REGION Network 80: IMMEDIATE STOP ALARMS
   RUNG wire#powerrail
      Contact( "M_ONE" )
      wire#w1
      I_Contact( #oALARM_POWDER_LINE_1_CLOGGED )
      I_Contact( #oALARM_GAS_FLOW_BELOW_LOW_LIMIT_LN_1 )
      I_Contact( #oALARM_DISK_SPEED_BELOW_LOW_LIMIT_LN_1 )
      I_Contact( #oALARM_STIRRER_SPEED_BELOW_LOW_LIMIT_LN_1 )
      I_Contact( #oALARM_GAS_FLOW_ABOVE_HIGH_LIMIT_LN_1 )
      I_Contact( #oALARM_CARRIER_GAS_INLET_PRESSURE_TOO_LOW_LN_1 )
      Not()
      Coil( #DATA.FAULT )
   END_RUNG
   RUNG wire#w1
      I_Contact( #DATA.FAULT )
      I_Contact( #oALARM_DISK_SPEED_ABOVE_HIGH_LIMIT_LN_1 )
      I_Contact( #oALARM_STIRRER_SPEED_ABOVE_HIGH_LIMIT_LN_1 )
      I_Contact( #oALARM_DISK_MOTOR_PLUGGED_IN_AND_READY_LN_1 )
      I_Contact( #oALARM_STIRRER_PLUGGED_IN_AND_READY_LN_1 )
      I_Contact( #oALARM_COMMUNICATION_RUNNING_LN_1 )
      I_Contact( #oALARM_FEEDER_NOT_READY_LN_1 )
      Not()
      Coil( #DATA.FAULT )
   END_RUNG
   RUNG wire#w1
      I_Contact( #DATA.FAULT )
      I_Contact( #oALARM_POWDER_LINE_2_CLOGGED )
      I_Contact( #oALARM_GAS_FLOW_BELOW_LOW_LIMIT_LN_2 )
      I_Contact( #oALARM_DISK_SPEED_BELOW_LOW_LIMIT_LN_2 )
      I_Contact( #oALARM_STIRRER_SPEED_BELOW_LOW_LIMIT_LN_2 )
      I_Contact( #oALARM_GAS_FLOW_ABOVE_HIGH_LIMIT_LN_2 )
      I_Contact( #oALARM_CARRIER_GAS_INLET_PRESSURE_TOO_LOW_LN_2 )
      Not()
      Coil( #DATA.FAULT )
   END_RUNG
   RUNG wire#w1
      I_Contact( #DATA.FAULT )
      I_Contact( #oALARM_DISK_SPEED_ABOVE_HIGH_LIMIT_LN_2 )
      I_Contact( #oALARM_STIRRER_SPEED_ABOVE_HIGH_LIMIT_LN_2 )
      I_Contact( #oALARM_DISK_MOTOR_PLUGGED_IN_AND_READY_LN_2 )
      I_Contact( #oALARM_STIRRER_PLUGGED_IN_AND_READY_LN_2 )
      I_Contact( #oALARM_COMMUNICATION_RUNNING_LN_2 )
      I_Contact( #oALARM_FEEDER_NOT_READY_LN_2 )
      Not()
      Move(in := #DB_NUMBER, out1 => "DB441_POWDER_FEEDERS_ALARM_DECODING".GLOBAL_ALARMS_MACHINE.ALARM_DECODING)
      wire#w2
      { S7_Templates := "SrcType := Int" } EQ_Contact(in1 := #INPUT_SETTINGS.UNIT_NUMBER, in2 := 1)
      S_Coil( "DB441_POWDER_FEEDERS_ALARM_DECODING".ALARMS_UNIT_01.POWDER_FEEDER[#INPUT_SETTINGS.FEEDER_NUMBER].IS_ALARMS )
   END_RUNG
   RUNG wire#w2
      { S7_Templates := "SrcType := Int" } EQ_Contact(in1 := #INPUT_SETTINGS.UNIT_NUMBER, in2 := 2)
      S_Coil( "DB441_POWDER_FEEDERS_ALARM_DECODING".ALARMS_UNIT_02.POWDER_FEEDER[#INPUT_SETTINGS.FEEDER_NUMBER].IS_ALARMS )
   END_RUNG
   // the same network as SCL:
   #DATA.FAULT := NOT ("M_ONE" AND NOT #oALARM_POWDER_LINE_1_CLOGGED AND NOT #oALARM_GAS_FLOW_BELOW_LOW_LIMIT_LN_1 AND NOT #oALARM_DISK_SPEED_BELOW_LOW_LIMIT_LN_1 AND NOT #oALARM_STIRRER_SPEED_BELOW_LOW_LIMIT_LN_1 AND NOT #oALARM_GAS_FLOW_ABOVE_HIGH_LIMIT_LN_1 AND NOT #oALARM_CARRIER_GAS_INLET_PRESSURE_TOO_LOW_LN_1);
   #DATA.FAULT := NOT ("M_ONE" AND NOT #DATA.FAULT AND NOT #oALARM_DISK_SPEED_ABOVE_HIGH_LIMIT_LN_1 AND NOT #oALARM_STIRRER_SPEED_ABOVE_HIGH_LIMIT_LN_1 AND NOT #oALARM_DISK_MOTOR_PLUGGED_IN_AND_READY_LN_1 AND NOT #oALARM_STIRRER_PLUGGED_IN_AND_READY_LN_1 AND NOT #oALARM_COMMUNICATION_RUNNING_LN_1 AND NOT #oALARM_FEEDER_NOT_READY_LN_1);
   #DATA.FAULT := NOT ("M_ONE" AND NOT #DATA.FAULT AND NOT #oALARM_POWDER_LINE_2_CLOGGED AND NOT #oALARM_GAS_FLOW_BELOW_LOW_LIMIT_LN_2 AND NOT #oALARM_DISK_SPEED_BELOW_LOW_LIMIT_LN_2 AND NOT #oALARM_STIRRER_SPEED_BELOW_LOW_LIMIT_LN_2 AND NOT #oALARM_GAS_FLOW_ABOVE_HIGH_LIMIT_LN_2 AND NOT #oALARM_CARRIER_GAS_INLET_PRESSURE_TOO_LOW_LN_2);
   #_w1 := NOT ("M_ONE" AND NOT #DATA.FAULT AND NOT #oALARM_DISK_SPEED_ABOVE_HIGH_LIMIT_LN_2 AND NOT #oALARM_STIRRER_SPEED_ABOVE_HIGH_LIMIT_LN_2 AND NOT #oALARM_DISK_MOTOR_PLUGGED_IN_AND_READY_LN_2 AND NOT #oALARM_STIRRER_PLUGGED_IN_AND_READY_LN_2 AND NOT #oALARM_COMMUNICATION_RUNNING_LN_2 AND NOT #oALARM_FEEDER_NOT_READY_LN_2);
   IF #_w1 THEN
       "DB441_POWDER_FEEDERS_ALARM_DECODING".GLOBAL_ALARMS_MACHINE.ALARM_DECODING := #DB_NUMBER;
   END_IF;
   IF #_w1 AND (#INPUT_SETTINGS.UNIT_NUMBER = 1) THEN
       "DB441_POWDER_FEEDERS_ALARM_DECODING".ALARMS_UNIT_01.POWDER_FEEDER[#INPUT_SETTINGS.FEEDER_NUMBER].IS_ALARMS := TRUE;
   END_IF;
   IF #_w1 AND (#INPUT_SETTINGS.UNIT_NUMBER = 2) THEN
       "DB441_POWDER_FEEDERS_ALARM_DECODING".ALARMS_UNIT_02.POWDER_FEEDER[#INPUT_SETTINGS.FEEDER_NUMBER].IS_ALARMS := TRUE;
   END_IF;
END_REGION

REGION Network 81: WARNINGS
   RUNG wire#powerrail
      Contact( "M_ONE" )
      wire#w1
      I_Contact( #oWARNING_GAS_FLOW_UNDER_LIMIT_LN_1 )
      I_Contact( #oWARNING_DISK_SPEED_UNDER_LIMIT_LN_1 )
      I_Contact( #oWARNING_STIRRER_SPEED_UNDER_LIMIT_LN_1 )
      I_Contact( #oWARNING_GAS_FLOW_OVER_LIMIT_LN_1 )
      I_Contact( #oWARNING_DISK_SPEED_OVER_LIMIT_LN_1 )
      I_Contact( #oWARNING_STIRRER_SPEED_OVER_LIMIT_LN_1 )
      Not()
      Coil( #oSTATION_WARNINGS )
   END_RUNG
   RUNG wire#w1
      I_Contact( #oSTATION_WARNINGS )
      I_Contact( #oWARNING_GAS_FLOW_UNDER_LIMIT_LN_2 )
      I_Contact( #oWARNING_DISK_SPEED_UNDER_LIMIT_LN_2 )
      I_Contact( #oWARNING_STIRRER_SPEED_UNDER_LIMIT_LN_2 )
      I_Contact( #oWARNING_GAS_FLOW_OVER_LIMIT_LN_2 )
      I_Contact( #oWARNING_DISK_SPEED_OVER_LIMIT_LN_2 )
      I_Contact( #oWARNING_STIRRER_SPEED_OVER_LIMIT_LN_2 )
      Not()
      Move(in := #DB_NUMBER, out1 => "DB441_POWDER_FEEDERS_ALARM_DECODING".GLOBAL_ALARMS_MACHINE.HELP_DECODING)
      wire#w2
      { S7_Templates := "SrcType := Int" } EQ_Contact(in1 := #INPUT_SETTINGS.UNIT_NUMBER, in2 := 1)
      S_Coil( "DB441_POWDER_FEEDERS_ALARM_DECODING".ALARMS_UNIT_01.POWDER_FEEDER[#INPUT_SETTINGS.FEEDER_NUMBER].WARNING )
   END_RUNG
   RUNG wire#w2
      { S7_Templates := "SrcType := Int" } EQ_Contact(in1 := #INPUT_SETTINGS.UNIT_NUMBER, in2 := 2)
      S_Coil( "DB441_POWDER_FEEDERS_ALARM_DECODING".ALARMS_UNIT_02.POWDER_FEEDER[#INPUT_SETTINGS.FEEDER_NUMBER].WARNING )
   END_RUNG
   // the same network as SCL:
   #oSTATION_WARNINGS := NOT ("M_ONE" AND NOT #oWARNING_GAS_FLOW_UNDER_LIMIT_LN_1 AND NOT #oWARNING_DISK_SPEED_UNDER_LIMIT_LN_1 AND NOT #oWARNING_STIRRER_SPEED_UNDER_LIMIT_LN_1 AND NOT #oWARNING_GAS_FLOW_OVER_LIMIT_LN_1 AND NOT #oWARNING_DISK_SPEED_OVER_LIMIT_LN_1 AND NOT #oWARNING_STIRRER_SPEED_OVER_LIMIT_LN_1);
   #_w1 := NOT ("M_ONE" AND NOT #oSTATION_WARNINGS AND NOT #oWARNING_GAS_FLOW_UNDER_LIMIT_LN_2 AND NOT #oWARNING_DISK_SPEED_UNDER_LIMIT_LN_2 AND NOT #oWARNING_STIRRER_SPEED_UNDER_LIMIT_LN_2 AND NOT #oWARNING_GAS_FLOW_OVER_LIMIT_LN_2 AND NOT #oWARNING_DISK_SPEED_OVER_LIMIT_LN_2 AND NOT #oWARNING_STIRRER_SPEED_OVER_LIMIT_LN_2);
   IF #_w1 THEN
       "DB441_POWDER_FEEDERS_ALARM_DECODING".GLOBAL_ALARMS_MACHINE.HELP_DECODING := #DB_NUMBER;
   END_IF;
   IF #_w1 AND (#INPUT_SETTINGS.UNIT_NUMBER = 1) THEN
       "DB441_POWDER_FEEDERS_ALARM_DECODING".ALARMS_UNIT_01.POWDER_FEEDER[#INPUT_SETTINGS.FEEDER_NUMBER].WARNING := TRUE;
   END_IF;
   IF #_w1 AND (#INPUT_SETTINGS.UNIT_NUMBER = 2) THEN
       "DB441_POWDER_FEEDERS_ALARM_DECODING".ALARMS_UNIT_02.POWDER_FEEDER[#INPUT_SETTINGS.FEEDER_NUMBER].WARNING := TRUE;
   END_IF;
END_REGION

REGION Network 82: FAULT RESET
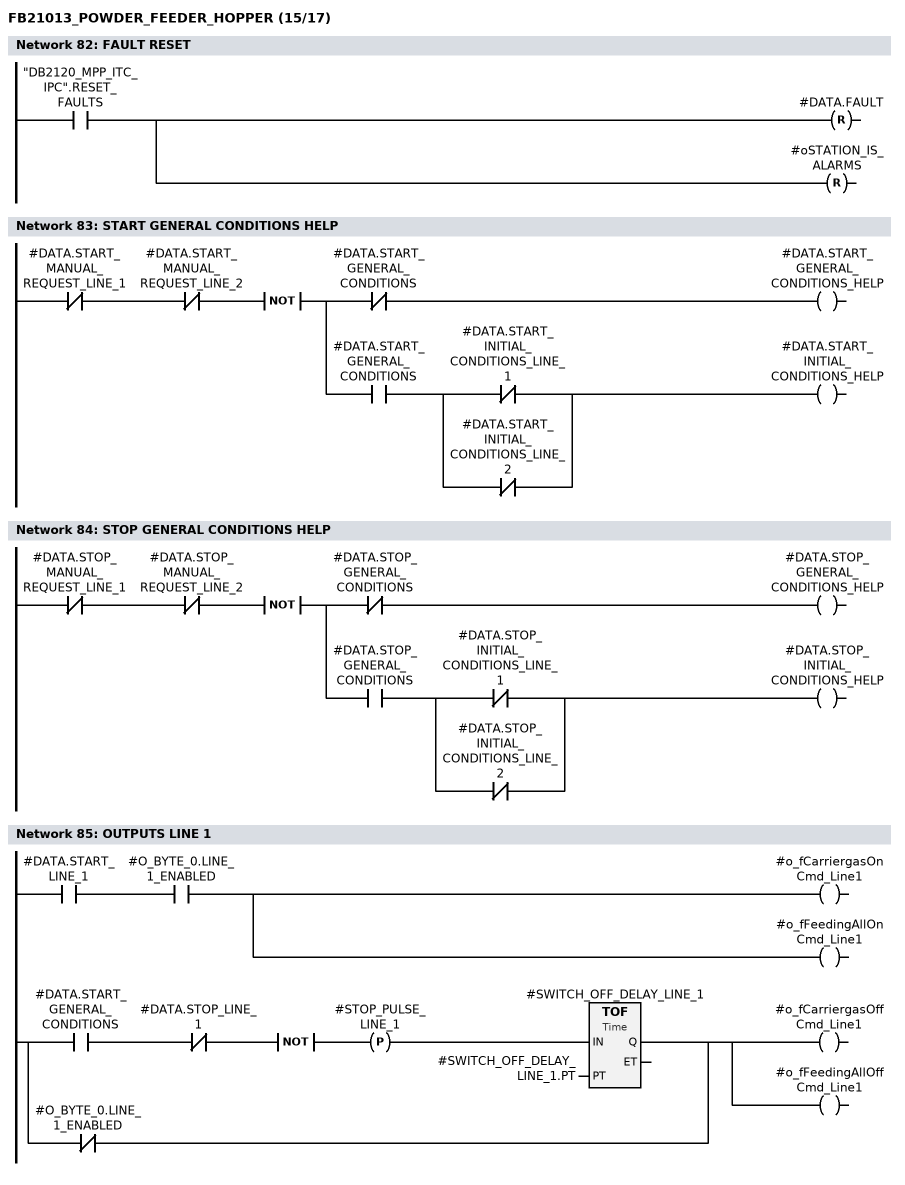
   RUNG wire#powerrail
      Contact( "DB2120_MPP_ITC_IPC".RESET_FAULTS )
      wire#w1
      R_Coil( #DATA.FAULT )
   END_RUNG
   RUNG wire#w1
      R_Coil( #oSTATION_IS_ALARMS )
   END_RUNG
   // the same network as SCL:
   IF "DB2120_MPP_ITC_IPC".RESET_FAULTS THEN
       #DATA.FAULT := FALSE;
       #oSTATION_IS_ALARMS := FALSE;
   END_IF;
END_REGION

REGION Network 83: START GENERAL CONDITIONS HELP
   RUNG wire#powerrail
      I_Contact( #DATA.START_MANUAL_REQUEST_LINE_1 )
      I_Contact( #DATA.START_MANUAL_REQUEST_LINE_2 )
      Not()
      wire#w1
      I_Contact( #DATA.START_GENERAL_CONDITIONS )
      Coil( #DATA.START_GENERAL_CONDITIONS_HELP )
   END_RUNG
   RUNG wire#w1
      Contact( #DATA.START_GENERAL_CONDITIONS )
      wire#w2
      I_Contact( #DATA.START_INITIAL_CONDITIONS_LINE_1 )
      wire#w3
      Coil( #DATA.START_INITIAL_CONDITIONS_HELP )
   END_RUNG
   RUNG wire#w2
      I_Contact( #DATA.START_INITIAL_CONDITIONS_LINE_2 )
   END_RUNG wire#w3
   // the same network as SCL:
   #_w1 := NOT (NOT #DATA.START_MANUAL_REQUEST_LINE_1 AND NOT #DATA.START_MANUAL_REQUEST_LINE_2);
   #DATA.START_GENERAL_CONDITIONS_HELP := #_w1 AND NOT #DATA.START_GENERAL_CONDITIONS;
   #DATA.START_INITIAL_CONDITIONS_HELP := #_w1 AND #DATA.START_GENERAL_CONDITIONS AND (NOT #DATA.START_INITIAL_CONDITIONS_LINE_1 OR NOT #DATA.START_INITIAL_CONDITIONS_LINE_2);
END_REGION

REGION Network 84: STOP GENERAL CONDITIONS HELP
   RUNG wire#powerrail
      I_Contact( #DATA.STOP_MANUAL_REQUEST_LINE_1 )
      I_Contact( #DATA.STOP_MANUAL_REQUEST_LINE_2 )
      Not()
      wire#w1
      I_Contact( #DATA.STOP_GENERAL_CONDITIONS )
      Coil( #DATA.STOP_GENERAL_CONDITIONS_HELP )
   END_RUNG
   RUNG wire#w1
      Contact( #DATA.STOP_GENERAL_CONDITIONS )
      wire#w2
      I_Contact( #DATA.STOP_INITIAL_CONDITIONS_LINE_1 )
      wire#w3
      Coil( #DATA.STOP_INITIAL_CONDITIONS_HELP )
   END_RUNG
   RUNG wire#w2
      I_Contact( #DATA.STOP_INITIAL_CONDITIONS_LINE_2 )
   END_RUNG wire#w3
   // the same network as SCL:
   #_w1 := NOT (NOT #DATA.STOP_MANUAL_REQUEST_LINE_1 AND NOT #DATA.STOP_MANUAL_REQUEST_LINE_2);
   #DATA.STOP_GENERAL_CONDITIONS_HELP := #_w1 AND NOT #DATA.STOP_GENERAL_CONDITIONS;
   #DATA.STOP_INITIAL_CONDITIONS_HELP := #_w1 AND #DATA.STOP_GENERAL_CONDITIONS AND (NOT #DATA.STOP_INITIAL_CONDITIONS_LINE_1 OR NOT #DATA.STOP_INITIAL_CONDITIONS_LINE_2);
END_REGION

REGION Network 85: OUTPUTS LINE 1
   RUNG wire#powerrail
      Contact( #DATA.START_LINE_1 )
      Contact( #O_BYTE_0.LINE_1_ENABLED )
      wire#w1
      Coil( #o_fCarriergasOnCmd_Line1 )
   END_RUNG
   RUNG wire#w1
      Coil( #o_fFeedingAllOnCmd_Line1 )
   END_RUNG
   RUNG wire#powerrail
      Contact( #DATA.START_GENERAL_CONDITIONS )
      I_Contact( #DATA.STOP_LINE_1 )
      Not()
      P_Trig( #STOP_PULSE_LINE_1 )
      { S7_Templates := "time_type := Time" } #SWITCH_OFF_DELAY_LINE_1.TOF(pt := #SWITCH_OFF_DELAY_LINE_1.PT, et =>)
      wire#w2
      Coil( #o_fCarriergasOffCmd_Line1 )
   END_RUNG
   RUNG wire#powerrail
      I_Contact( #O_BYTE_0.LINE_1_ENABLED )
   END_RUNG wire#w2
   RUNG wire#w2
      Coil( #o_fFeedingAllOffCmd_Line1 )
   END_RUNG
   // the same network as SCL:
   #o_fCarriergasOnCmd_Line1 := #DATA.START_LINE_1 AND #O_BYTE_0.LINE_1_ENABLED;
   #o_fFeedingAllOnCmd_Line1 := #o_fCarriergasOnCmd_Line1;
   #_w1 := NOT (#DATA.START_GENERAL_CONDITIONS AND NOT #DATA.STOP_LINE_1);
   #_w2 := #_w1 AND NOT #STOP_PULSE_LINE_1;   // rising edge
   #STOP_PULSE_LINE_1 := #_w1;
   #SWITCH_OFF_DELAY_LINE_1(IN := #_w2, PT := #SWITCH_OFF_DELAY_LINE_1.PT);   // TOF
   #o_fCarriergasOffCmd_Line1 := #SWITCH_OFF_DELAY_LINE_1.Q OR NOT #O_BYTE_0.LINE_1_ENABLED;
   #o_fFeedingAllOffCmd_Line1 := #o_fCarriergasOffCmd_Line1;
END_REGION

REGION Network 86: OUTPUTS LINE 2
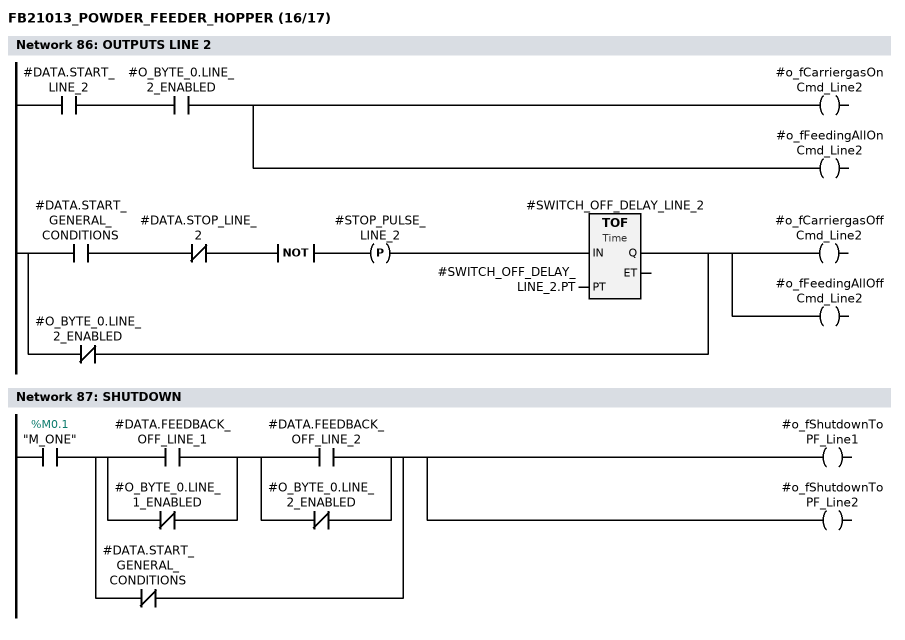
   RUNG wire#powerrail
      Contact( #DATA.START_LINE_2 )
      Contact( #O_BYTE_0.LINE_2_ENABLED )
      wire#w1
      Coil( #o_fCarriergasOnCmd_Line2 )
   END_RUNG
   RUNG wire#w1
      Coil( #o_fFeedingAllOnCmd_Line2 )
   END_RUNG
   RUNG wire#powerrail
      Contact( #DATA.START_GENERAL_CONDITIONS )
      I_Contact( #DATA.STOP_LINE_2 )
      Not()
      P_Trig( #STOP_PULSE_LINE_2 )
      { S7_Templates := "time_type := Time" } #SWITCH_OFF_DELAY_LINE_2.TOF(pt := #SWITCH_OFF_DELAY_LINE_2.PT, et =>)
      wire#w2
      Coil( #o_fCarriergasOffCmd_Line2 )
   END_RUNG
   RUNG wire#powerrail
      I_Contact( #O_BYTE_0.LINE_2_ENABLED )
   END_RUNG wire#w2
   RUNG wire#w2
      Coil( #o_fFeedingAllOffCmd_Line2 )
   END_RUNG
   // the same network as SCL:
   #o_fCarriergasOnCmd_Line2 := #DATA.START_LINE_2 AND #O_BYTE_0.LINE_2_ENABLED;
   #o_fFeedingAllOnCmd_Line2 := #o_fCarriergasOnCmd_Line2;
   #_w1 := NOT (#DATA.START_GENERAL_CONDITIONS AND NOT #DATA.STOP_LINE_2);
   #_w2 := #_w1 AND NOT #STOP_PULSE_LINE_2;   // rising edge
   #STOP_PULSE_LINE_2 := #_w1;
   #SWITCH_OFF_DELAY_LINE_2(IN := #_w2, PT := #SWITCH_OFF_DELAY_LINE_2.PT);   // TOF
   #o_fCarriergasOffCmd_Line2 := #SWITCH_OFF_DELAY_LINE_2.Q OR NOT #O_BYTE_0.LINE_2_ENABLED;
   #o_fFeedingAllOffCmd_Line2 := #o_fCarriergasOffCmd_Line2;
END_REGION

REGION Network 87: SHUTDOWN
   RUNG wire#powerrail
      Contact( "M_ONE" )
      wire#w1
      Contact( #DATA.FEEDBACK_OFF_LINE_1 )
      wire#w2
      Contact( #DATA.FEEDBACK_OFF_LINE_2 )
      wire#w3
      Coil( #o_fShutdownToPF_Line1 )
   END_RUNG
   RUNG wire#w1
      I_Contact( #O_BYTE_0.LINE_1_ENABLED )
   END_RUNG wire#w2
   RUNG wire#w2
      I_Contact( #O_BYTE_0.LINE_2_ENABLED )
   END_RUNG wire#w3
   RUNG wire#w1
      I_Contact( #DATA.START_GENERAL_CONDITIONS )
   END_RUNG wire#w3
   RUNG wire#w3
      Coil( #o_fShutdownToPF_Line2 )
   END_RUNG
   // the same network as SCL:
   #o_fShutdownToPF_Line1 := "M_ONE" AND (((#DATA.FEEDBACK_OFF_LINE_1 OR NOT #O_BYTE_0.LINE_1_ENABLED) AND (#DATA.FEEDBACK_OFF_LINE_2 OR NOT #O_BYTE_0.LINE_2_ENABLED)) OR NOT #DATA.START_GENERAL_CONDITIONS);
   #o_fShutdownToPF_Line2 := #o_fShutdownToPF_Line1;
END_REGION

REGION Network 88: HOPPER STATUS
   // STATUS:
   // 0: OFF WITH NO CONDITIONS
   // 1: ON
   // 2: OFF WITH CONDITIONS TO SWITCH ON
   // 3: SWITCH ON SEQUENCE RUNNING
   // 4: SWITCH OFF SEQUENCE RUNNING
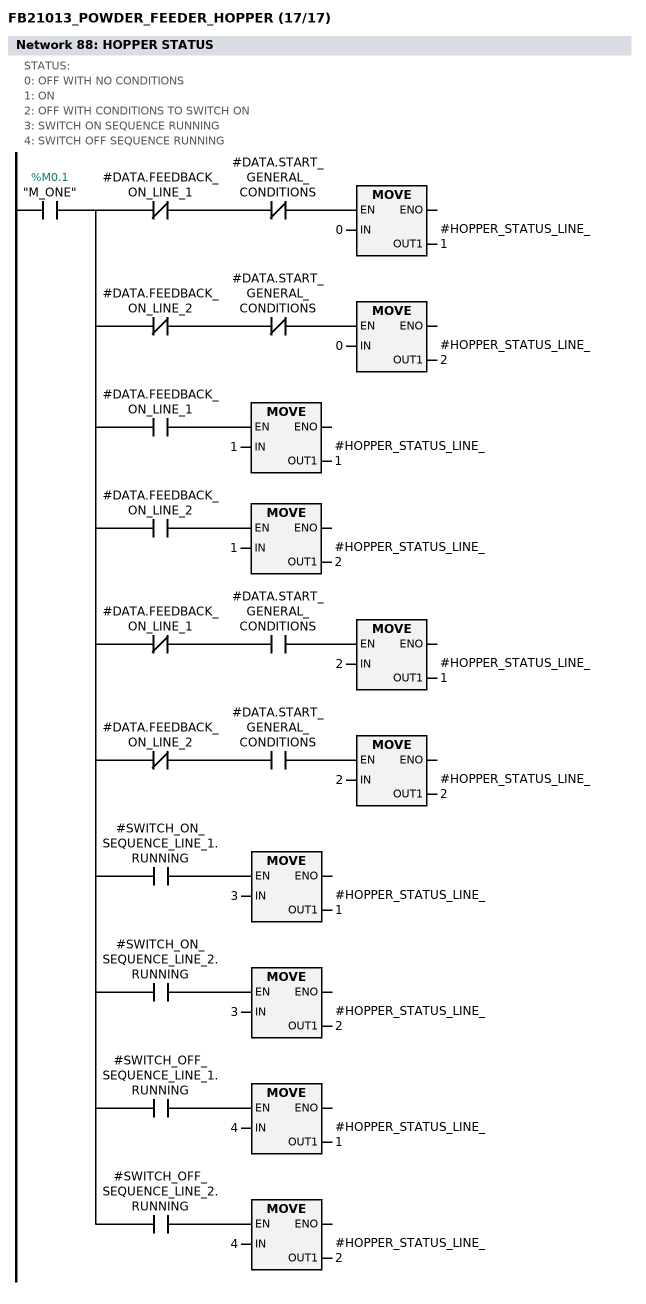
   RUNG wire#powerrail
      Contact( "M_ONE" )
      wire#w1
      I_Contact( #DATA.FEEDBACK_ON_LINE_1 )
      I_Contact( #DATA.START_GENERAL_CONDITIONS )
      Move(in := 0, out1 => #HOPPER_STATUS_LINE_1)
   END_RUNG
   RUNG wire#w1
      I_Contact( #DATA.FEEDBACK_ON_LINE_2 )
      I_Contact( #DATA.START_GENERAL_CONDITIONS )
      Move(in := 0, out1 => #HOPPER_STATUS_LINE_2)
   END_RUNG
   RUNG wire#w1
      Contact( #DATA.FEEDBACK_ON_LINE_1 )
      Move(in := 1, out1 => #HOPPER_STATUS_LINE_1)
   END_RUNG
   RUNG wire#w1
      Contact( #DATA.FEEDBACK_ON_LINE_2 )
      Move(in := 1, out1 => #HOPPER_STATUS_LINE_2)
   END_RUNG
   RUNG wire#w1
      I_Contact( #DATA.FEEDBACK_ON_LINE_1 )
      Contact( #DATA.START_GENERAL_CONDITIONS )
      Move(in := 2, out1 => #HOPPER_STATUS_LINE_1)
   END_RUNG
   RUNG wire#w1
      I_Contact( #DATA.FEEDBACK_ON_LINE_2 )
      Contact( #DATA.START_GENERAL_CONDITIONS )
      Move(in := 2, out1 => #HOPPER_STATUS_LINE_2)
   END_RUNG
   RUNG wire#w1
      Contact( #SWITCH_ON_SEQUENCE_LINE_1.RUNNING )
      Move(in := 3, out1 => #HOPPER_STATUS_LINE_1)
   END_RUNG
   RUNG wire#w1
      Contact( #SWITCH_ON_SEQUENCE_LINE_2.RUNNING )
      Move(in := 3, out1 => #HOPPER_STATUS_LINE_2)
   END_RUNG
   RUNG wire#w1
      Contact( #SWITCH_OFF_SEQUENCE_LINE_1.RUNNING )
      Move(in := 4, out1 => #HOPPER_STATUS_LINE_1)
   END_RUNG
   RUNG wire#w1
      Contact( #SWITCH_OFF_SEQUENCE_LINE_2.RUNNING )
      Move(in := 4, out1 => #HOPPER_STATUS_LINE_2)
   END_RUNG
   // the same network as SCL:
   IF "M_ONE" AND NOT #DATA.FEEDBACK_ON_LINE_1 AND NOT #DATA.START_GENERAL_CONDITIONS THEN
       #HOPPER_STATUS_LINE_1 := 0;
   END_IF;
   IF "M_ONE" AND NOT #DATA.FEEDBACK_ON_LINE_2 AND NOT #DATA.START_GENERAL_CONDITIONS THEN
       #HOPPER_STATUS_LINE_2 := 0;
   END_IF;
   IF "M_ONE" AND #DATA.FEEDBACK_ON_LINE_1 THEN #HOPPER_STATUS_LINE_1 := 1; END_IF;
   IF "M_ONE" AND #DATA.FEEDBACK_ON_LINE_2 THEN #HOPPER_STATUS_LINE_2 := 1; END_IF;
   IF "M_ONE" AND NOT #DATA.FEEDBACK_ON_LINE_1 AND #DATA.START_GENERAL_CONDITIONS THEN
       #HOPPER_STATUS_LINE_1 := 2;
   END_IF;
   IF "M_ONE" AND NOT #DATA.FEEDBACK_ON_LINE_2 AND #DATA.START_GENERAL_CONDITIONS THEN
       #HOPPER_STATUS_LINE_2 := 2;
   END_IF;
   IF "M_ONE" AND #SWITCH_ON_SEQUENCE_LINE_1.RUNNING THEN #HOPPER_STATUS_LINE_1 := 3; END_IF;
   IF "M_ONE" AND #SWITCH_ON_SEQUENCE_LINE_2.RUNNING THEN #HOPPER_STATUS_LINE_2 := 3; END_IF;
   IF "M_ONE" AND #SWITCH_OFF_SEQUENCE_LINE_1.RUNNING THEN #HOPPER_STATUS_LINE_1 := 4; END_IF;
   IF "M_ONE" AND #SWITCH_OFF_SEQUENCE_LINE_2.RUNNING THEN #HOPPER_STATUS_LINE_2 := 4; END_IF;
END_REGION
END_FUNCTION_BLOCK

FUNCTION_BLOCK "FB21250_POWDER_ON_OFF_SEQUENCE"   // FB21250, LAD
{ S7_Optimized_Access := 'FALSE' }
VERSION : 0.1
// stored: AutoNumber false, IsIECCheckEnabled false, SetENOAutomatically false, UDAEnableTagReadback false
   VAR_INPUT
      OPTIONS_0 : Byte := 2#0000_0000;   // OPTIONS 0
      REQUEST_INPUT : Bool;   // REQUEST
      GENERAL_CONDITIONS_INPUT : Bool;   // GENERAL CONDITIONS INPUT
      INITIAL_CONDITIONS_INPUT : Bool;   // INITIAL CONDITIONS INPUT
      GAS_FLOW_ACTUAL : Real;   // GAS FLOW ACTUAL
      DISK_SPEED_ACTUAL : Real;   // DISK SPEED ACTUAL
      GAS_SETPOINT : Real;   // GAS SETPOINT
      DISK_SETPOINT : Real;   // DISK SETPOINT
   END_VAR
   VAR_OUTPUT
      DONE : Bool;   // SEQUENCE DONE
   END_VAR
   VAR DB_SPECIFIC
      GENERAL_CONDITIONS : Bool;   // GENERAL CONDITIONS
      INITIAL_CONDITIONS : Bool;   // INITIAL CONDITIONS
      REQUEST_START : Bool;   // REQUEST START
      START_COMMAND : Bool;   // START COMMAND
      RUNNING : Bool := false;   // SEQUENCE RUNNING
      ACTUAL_STEP_GAS : Int := 1;   // ACTUAL STEP GAS
      ACTUAL_STEP_DISK : Int := 1;   // ACTUAL STEP DISK
      MAX_STEPS_GAS : Int := 10;   // MAXIMUM NUMBER OF STEPS FOR GAS
      MAX_STEPS_DISK { ExternalAccessible := 'False'; ExternalVisible := 'False'; ExternalWritable := 'False'} : Int := 10;   // MAXIMUM NUMBER OF STEPS FOR DISK
      GAS_WAIT_STEP : Int;   // GAS PAUSE STEP
      GAS_FLOW_OFFSET { ExternalAccessible := 'False'; ExternalVisible := 'False'; ExternalWritable := 'False'} : Real := 10.0;   // GAS FLOW STEP OFFSET
      DISK_SPEED_OFFSET { ExternalAccessible := 'False'; ExternalVisible := 'False'; ExternalWritable := 'False'} : Real := 10.0;   // DISK SPEED STEP OFFSET
      START_GAS_FLOW { ExternalAccessible := 'False'; ExternalVisible := 'False'; ExternalWritable := 'False'} : Real := 0.0;   // START GAS FLOW
      START_DISK_SPEED : Real := 0.0;   // START DISK SPEED
      GAS_FLOW_MIN : Real := 0.0;   // GAS FLOW MIN
      GAS_FLOW_MAX : Real := 0.0;   // GAS FLOW MAX
      DISK_SPEED_MIN : Real := 0.0;   // DISK SPEED MIN
      DISK_SPEED_MAX : Real := 0.0;   // DISK SPEED MAX
      AUX_SETPOINT_VALUES : Struct
         GAS_FLOW_SETPOINT : Real;   // GAS FLOW SETPOINT
         DISK_SPEED_SETPOINT : Real;   // DISK SPEED SETPOINT
      END_STRUCT;
      STEP_CHANGE_DELAY_GAS : TON_TIME;
      STEP_CHANGE_DELAY_DISK : TON_TIME;
      DONE_DELAY : TON_TIME;
      AUX_1 : Bool;   // AUX PULSE
      AUX_2 : Bool;   // AUX PULSE
      AUX_3 : Bool;   // AUX PULSE
      AUX_4 : Bool;   // AUX PULSE
      AUX_5 : Bool;   // AUX PULSE
   END_VAR
   VAR_TEMP
      DB_NUMBER : DInt;   // DB NUMBER FOR ALARM DECODING
      INPUTS_MASK : Byte;   // INPUTS MASK
      O_BYTE_0 : Struct   // OPTIONS BYTE 0
         ON_SEQUENCE : Bool;   // ON SEQUENCE OPTION
         OFF_SEQUENCE : Bool;   // OFF SEQUENCE OPTION
         SPARE_2 : Bool;
         SPARE_3 : Bool;
         SPARE_4 : Bool;
         SPARE_5 : Bool;
         SPARE_6 : Bool;
         SPARE_7 : Bool;
      END_STRUCT;
   END_VAR
   // STEP_CHANGE_DELAY_GAS.PT := T#200ms;
   // STEP_CHANGE_DELAY_DISK.PT := T#200ms;
   // DONE_DELAY.PT := T#2s;
   VAR_TEMP   // added for the SCL form of the ladder/FBD networks
      _w1 : Bool;
   END_VAR
BEGIN

NETWORK
TITLE = READ INSTANCE DB
      L     DINO;
      +     10#800000;
      T     #DB_NUMBER;


REGION Network 2: OPTIONS
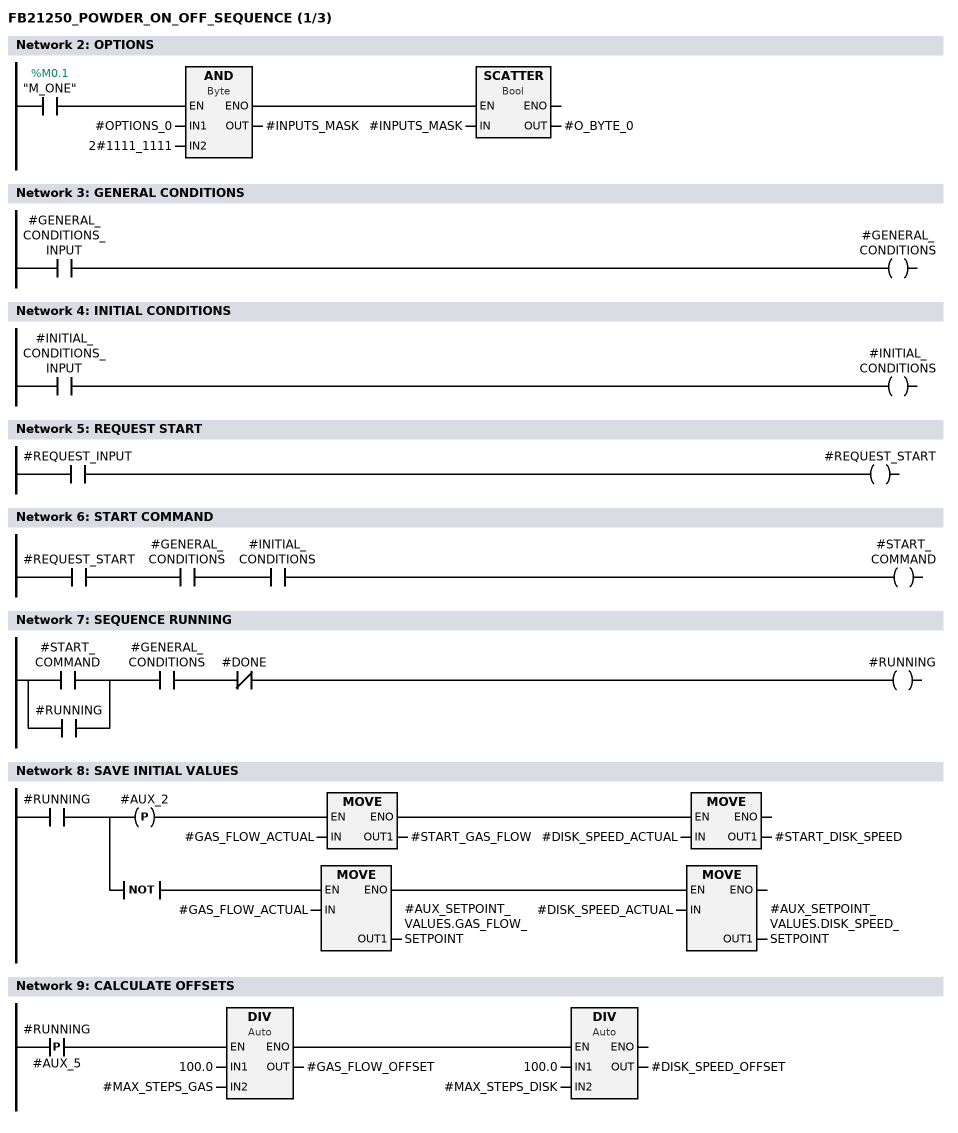
   RUNG wire#powerrail
      Contact( "M_ONE" )
      { S7_Templates := "SrcType := Byte"; S7_GenerateENO := "TRUE" } And(in1 := #OPTIONS_0, in2 := 2#1111_1111, out => #INPUTS_MASK)
      { S7_Templates := "[dest_type := Bool, src_type := Byte]" } SCATTER(IN := #INPUTS_MASK, OUT => #O_BYTE_0)
   END_RUNG
   // the same network as SCL:
   IF "M_ONE" THEN
       #INPUTS_MASK := #OPTIONS_0 AND 2#1111_1111;
       SCATTER(IN := #INPUTS_MASK, OUT => #O_BYTE_0);
   END_IF;
END_REGION

REGION Network 3: GENERAL CONDITIONS
   RUNG wire#powerrail
      Contact( #GENERAL_CONDITIONS_INPUT )
      Coil( #GENERAL_CONDITIONS )
   END_RUNG
   // the same network as SCL:
   #GENERAL_CONDITIONS := #GENERAL_CONDITIONS_INPUT;
END_REGION

REGION Network 4: INITIAL CONDITIONS
   RUNG wire#powerrail
      Contact( #INITIAL_CONDITIONS_INPUT )
      Coil( #INITIAL_CONDITIONS )
   END_RUNG
   // the same network as SCL:
   #INITIAL_CONDITIONS := #INITIAL_CONDITIONS_INPUT;
END_REGION

REGION Network 5: REQUEST START
   RUNG wire#powerrail
      Contact( #REQUEST_INPUT )
      Coil( #REQUEST_START )
   END_RUNG
   // the same network as SCL:
   #REQUEST_START := #REQUEST_INPUT;
END_REGION

REGION Network 6: START COMMAND
   RUNG wire#powerrail
      Contact( #REQUEST_START )
      Contact( #GENERAL_CONDITIONS )
      Contact( #INITIAL_CONDITIONS )
      Coil( #START_COMMAND )
   END_RUNG
   // the same network as SCL:
   #START_COMMAND := #REQUEST_START AND #GENERAL_CONDITIONS AND #INITIAL_CONDITIONS;
END_REGION

REGION Network 7: SEQUENCE RUNNING
   RUNG wire#powerrail
      Contact( #START_COMMAND )
      wire#w1
      Contact( #GENERAL_CONDITIONS )
      I_Contact( #DONE )
      Coil( #RUNNING )
   END_RUNG
   RUNG wire#powerrail
      Contact( #RUNNING )
   END_RUNG wire#w1
   // the same network as SCL:
   #RUNNING := (#START_COMMAND OR #RUNNING) AND #GENERAL_CONDITIONS AND NOT #DONE;
END_REGION

REGION Network 8: SAVE INITIAL VALUES
   RUNG wire#powerrail
      Contact( #RUNNING )
      wire#w1
      P_Trig( #AUX_2 )
      Move(in := #GAS_FLOW_ACTUAL, out1 => #START_GAS_FLOW)
      Move(in := #DISK_SPEED_ACTUAL, out1 => #START_DISK_SPEED)
   END_RUNG
   RUNG wire#w1
      Not()
      Move(in := #GAS_FLOW_ACTUAL, out1 => #AUX_SETPOINT_VALUES.GAS_FLOW_SETPOINT)
      Move(in := #DISK_SPEED_ACTUAL, out1 => #AUX_SETPOINT_VALUES.DISK_SPEED_SETPOINT)
   END_RUNG
   // the same network as SCL:
   #_w1 := #RUNNING AND NOT #AUX_2;   // rising edge
   #AUX_2 := #RUNNING;
   IF #_w1 THEN
       #START_GAS_FLOW := #GAS_FLOW_ACTUAL;
       #START_DISK_SPEED := #DISK_SPEED_ACTUAL;
   END_IF;
   IF NOT #RUNNING THEN
       #AUX_SETPOINT_VALUES.GAS_FLOW_SETPOINT := #GAS_FLOW_ACTUAL;
       #AUX_SETPOINT_VALUES.DISK_SPEED_SETPOINT := #DISK_SPEED_ACTUAL;
   END_IF;
END_REGION

REGION Network 9: CALCULATE OFFSETS
   RUNG wire#powerrail
      P_Contact(operand := #RUNNING, bit := #AUX_5)
      Div(in1 := 100.0, in2 := #MAX_STEPS_GAS, out => #GAS_FLOW_OFFSET)
      Div(in1 := 100.0, in2 := #MAX_STEPS_DISK, out => #DISK_SPEED_OFFSET)
   END_RUNG
   // the same network as SCL:
   #_w1 := #RUNNING AND NOT #AUX_5;   // rising edge of #RUNNING
   #AUX_5 := #RUNNING;
   IF #_w1 THEN
       #GAS_FLOW_OFFSET := 100.0 / #MAX_STEPS_GAS;
       #DISK_SPEED_OFFSET := 100.0 / #MAX_STEPS_DISK;
   END_IF;
END_REGION

REGION Network 10: CALCULATE VALUES DISK
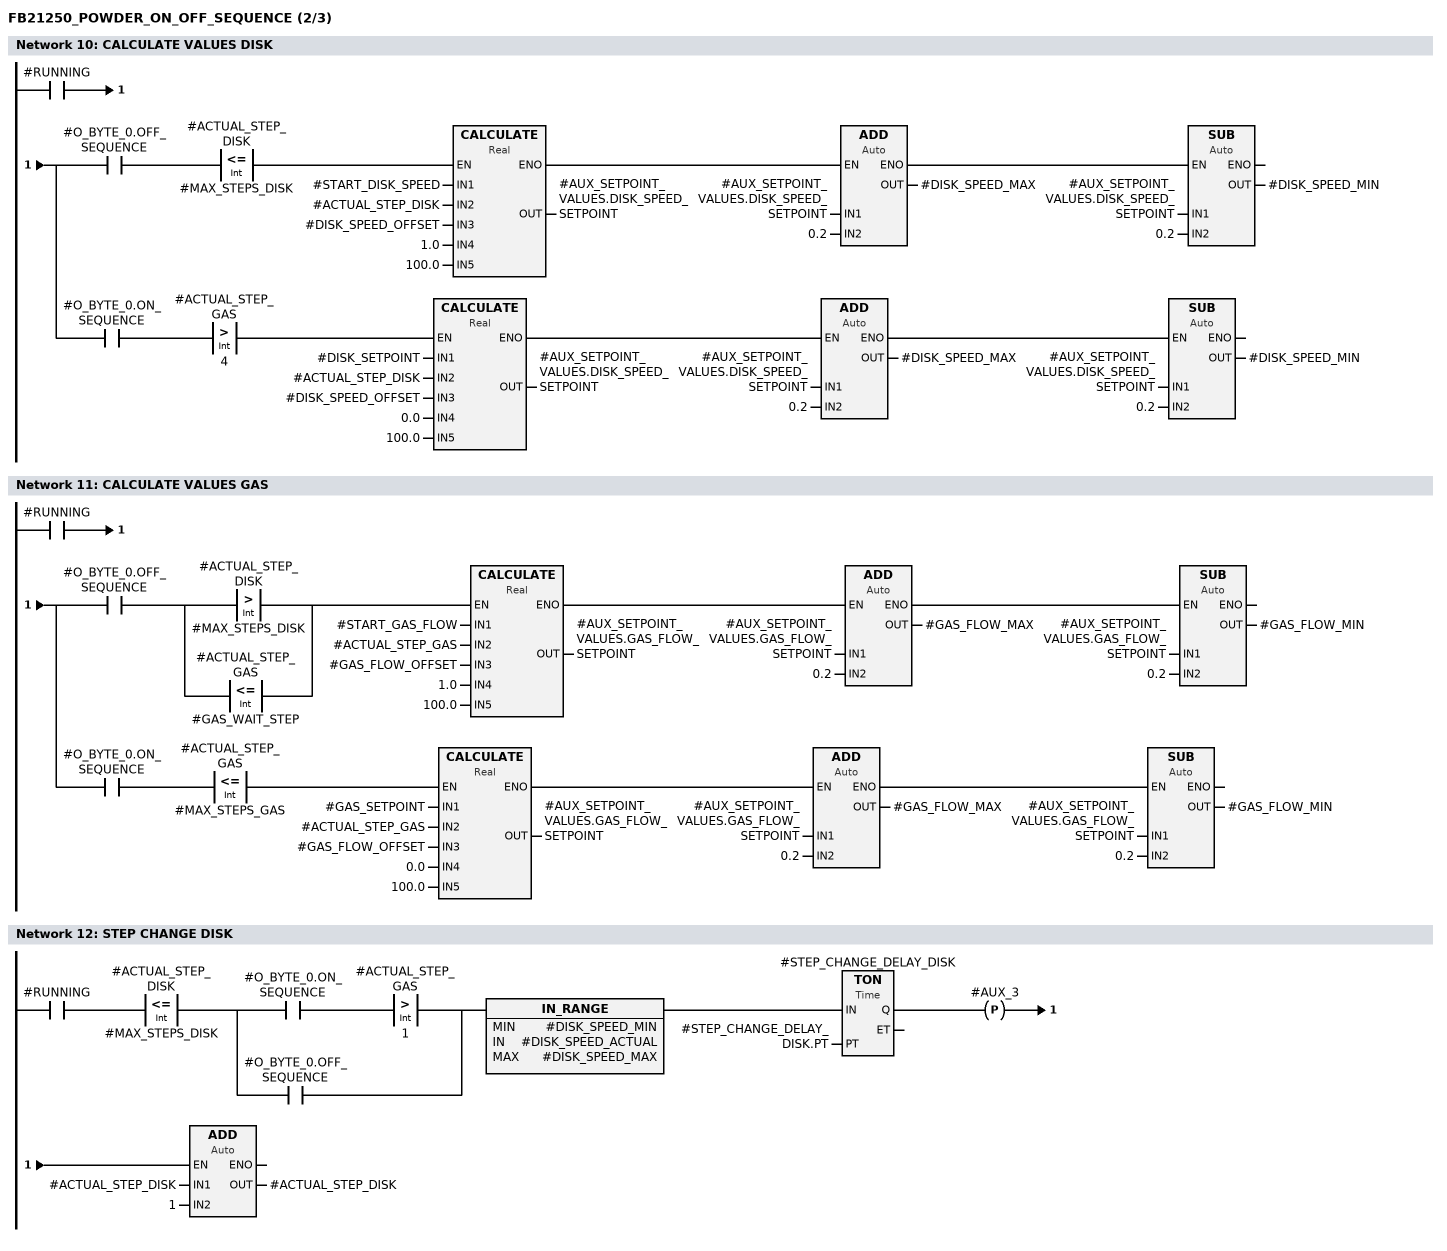
   RUNG wire#powerrail
      Contact( #RUNNING )
      wire#w1
      Contact( #O_BYTE_0.OFF_SEQUENCE )
      { S7_Templates := "SrcType := Int" } LE_Contact(in1 := #ACTUAL_STEP_DISK, in2 := #MAX_STEPS_DISK)
      { S7_Templates := "SrcType := Real"; S7_Expression := "(IN1)*(IN4-(IN2*(IN3/IN5)))" } Calculate(in1 := #START_DISK_SPEED, in2 := #ACTUAL_STEP_DISK, in3 := #DISK_SPEED_OFFSET, in4 := 1.0, in5 := 100.0, out => #AUX_SETPOINT_VALUES.DISK_SPEED_SETPOINT)
      Add(in1 := #AUX_SETPOINT_VALUES.DISK_SPEED_SETPOINT, in2 := 0.2, out => #DISK_SPEED_MAX)
      Sub(in1 := #AUX_SETPOINT_VALUES.DISK_SPEED_SETPOINT, in2 := 0.2, out => #DISK_SPEED_MIN)
   END_RUNG
   RUNG wire#w1
      Contact( #O_BYTE_0.ON_SEQUENCE )
      { S7_Templates := "SrcType := Int" } GT_Contact(in1 := #ACTUAL_STEP_GAS, in2 := 4)
      { S7_Templates := "SrcType := Real"; S7_Expression := "(IN1)*(IN4+(IN2*(IN3/IN5)))" } Calculate(in1 := #DISK_SETPOINT, in2 := #ACTUAL_STEP_DISK, in3 := #DISK_SPEED_OFFSET, in4 := 0.0, in5 := 100.0, out => #AUX_SETPOINT_VALUES.DISK_SPEED_SETPOINT)
      Add(in1 := #AUX_SETPOINT_VALUES.DISK_SPEED_SETPOINT, in2 := 0.2, out => #DISK_SPEED_MAX)
      Sub(in1 := #AUX_SETPOINT_VALUES.DISK_SPEED_SETPOINT, in2 := 0.2, out => #DISK_SPEED_MIN)
   END_RUNG
   // the same network as SCL:
   IF #RUNNING AND #O_BYTE_0.OFF_SEQUENCE AND (#ACTUAL_STEP_DISK <= #MAX_STEPS_DISK) THEN
       #AUX_SETPOINT_VALUES.DISK_SPEED_SETPOINT := (#START_DISK_SPEED)*(1.0-(#ACTUAL_STEP_DISK*(#DISK_SPEED_OFFSET/100.0)));
       #DISK_SPEED_MAX := #AUX_SETPOINT_VALUES.DISK_SPEED_SETPOINT + 0.2;
       #DISK_SPEED_MIN := #AUX_SETPOINT_VALUES.DISK_SPEED_SETPOINT - 0.2;
   END_IF;
   IF #RUNNING AND #O_BYTE_0.ON_SEQUENCE AND (#ACTUAL_STEP_GAS > 4) THEN
       #AUX_SETPOINT_VALUES.DISK_SPEED_SETPOINT := (#DISK_SETPOINT)*(0.0+(#ACTUAL_STEP_DISK*(#DISK_SPEED_OFFSET/100.0)));
       #DISK_SPEED_MAX := #AUX_SETPOINT_VALUES.DISK_SPEED_SETPOINT + 0.2;
       #DISK_SPEED_MIN := #AUX_SETPOINT_VALUES.DISK_SPEED_SETPOINT - 0.2;
   END_IF;
END_REGION

REGION Network 11: CALCULATE VALUES GAS
   RUNG wire#powerrail
      Contact( #RUNNING )
      wire#w1
      Contact( #O_BYTE_0.OFF_SEQUENCE )
      wire#w2
      { S7_Templates := "SrcType := Int" } GT_Contact(in1 := #ACTUAL_STEP_DISK, in2 := #MAX_STEPS_DISK)
      wire#w3
      { S7_Templates := "SrcType := Real"; S7_Expression := "(IN1)*(IN4-(IN2*(IN3/IN5)))" } Calculate(in1 := #START_GAS_FLOW, in2 := #ACTUAL_STEP_GAS, in3 := #GAS_FLOW_OFFSET, in4 := 1.0, in5 := 100.0, out => #AUX_SETPOINT_VALUES.GAS_FLOW_SETPOINT)
      Add(in1 := #AUX_SETPOINT_VALUES.GAS_FLOW_SETPOINT, in2 := 0.2, out => #GAS_FLOW_MAX)
      Sub(in1 := #AUX_SETPOINT_VALUES.GAS_FLOW_SETPOINT, in2 := 0.2, out => #GAS_FLOW_MIN)
   END_RUNG
   RUNG wire#w2
      { S7_Templates := "SrcType := Int" } LE_Contact(in1 := #ACTUAL_STEP_GAS, in2 := #GAS_WAIT_STEP)
   END_RUNG wire#w3
   RUNG wire#w1
      Contact( #O_BYTE_0.ON_SEQUENCE )
      { S7_Templates := "SrcType := Int" } LE_Contact(in1 := #ACTUAL_STEP_GAS, in2 := #MAX_STEPS_GAS)
      { S7_Templates := "SrcType := Real"; S7_Expression := "(IN1)*(IN4+(IN2*(IN3/IN5)))" } Calculate(in1 := #GAS_SETPOINT, in2 := #ACTUAL_STEP_GAS, in3 := #GAS_FLOW_OFFSET, in4 := 0.0, in5 := 100.0, out => #AUX_SETPOINT_VALUES.GAS_FLOW_SETPOINT)
      Add(in1 := #AUX_SETPOINT_VALUES.GAS_FLOW_SETPOINT, in2 := 0.2, out => #GAS_FLOW_MAX)
      Sub(in1 := #AUX_SETPOINT_VALUES.GAS_FLOW_SETPOINT, in2 := 0.2, out => #GAS_FLOW_MIN)
   END_RUNG
   // the same network as SCL:
   IF #RUNNING AND #O_BYTE_0.OFF_SEQUENCE AND ((#ACTUAL_STEP_DISK > #MAX_STEPS_DISK) OR (#ACTUAL_STEP_GAS <= #GAS_WAIT_STEP)) THEN
       #AUX_SETPOINT_VALUES.GAS_FLOW_SETPOINT := (#START_GAS_FLOW)*(1.0-(#ACTUAL_STEP_GAS*(#GAS_FLOW_OFFSET/100.0)));
       #GAS_FLOW_MAX := #AUX_SETPOINT_VALUES.GAS_FLOW_SETPOINT + 0.2;
       #GAS_FLOW_MIN := #AUX_SETPOINT_VALUES.GAS_FLOW_SETPOINT - 0.2;
   END_IF;
   IF #RUNNING AND #O_BYTE_0.ON_SEQUENCE AND (#ACTUAL_STEP_GAS <= #MAX_STEPS_GAS) THEN
       #AUX_SETPOINT_VALUES.GAS_FLOW_SETPOINT := (#GAS_SETPOINT)*(0.0+(#ACTUAL_STEP_GAS*(#GAS_FLOW_OFFSET/100.0)));
       #GAS_FLOW_MAX := #AUX_SETPOINT_VALUES.GAS_FLOW_SETPOINT + 0.2;
       #GAS_FLOW_MIN := #AUX_SETPOINT_VALUES.GAS_FLOW_SETPOINT - 0.2;
   END_IF;
END_REGION

REGION Network 12: STEP CHANGE DISK
   RUNG wire#powerrail
      Contact( #RUNNING )
      { S7_Templates := "SrcType := Int" } LE_Contact(in1 := #ACTUAL_STEP_DISK, in2 := #MAX_STEPS_DISK)
      wire#w1
      Contact( #O_BYTE_0.ON_SEQUENCE )
      { S7_Templates := "SrcType := Int" } GT_Contact(in1 := #ACTUAL_STEP_GAS, in2 := 1)
      wire#w2
      { S7_Templates := "SrcType := Real" } InRange(min := #DISK_SPEED_MIN, in := #DISK_SPEED_ACTUAL, max := #DISK_SPEED_MAX)
      { S7_Templates := "time_type := Time" } #STEP_CHANGE_DELAY_DISK.TON(pt := #STEP_CHANGE_DELAY_DISK.PT, et =>)
      P_Trig( #AUX_3 )
      Add(in1 := #ACTUAL_STEP_DISK, in2 := 1, out => #ACTUAL_STEP_DISK)
   END_RUNG
   RUNG wire#w1
      Contact( #O_BYTE_0.OFF_SEQUENCE )
   END_RUNG wire#w2
   // the same network as SCL:
   #STEP_CHANGE_DELAY_DISK(IN := #RUNNING AND (#ACTUAL_STEP_DISK <= #MAX_STEPS_DISK) AND ((#O_BYTE_0.ON_SEQUENCE AND (#ACTUAL_STEP_GAS > 1)) OR #O_BYTE_0.OFF_SEQUENCE) AND (#DISK_SPEED_MIN <= #DISK_SPEED_ACTUAL) AND (#DISK_SPEED_ACTUAL <= #DISK_SPEED_MAX),   // TON
                           PT := #STEP_CHANGE_DELAY_DISK.PT);
   #_w1 := #STEP_CHANGE_DELAY_DISK.Q AND NOT #AUX_3;   // rising edge
   #AUX_3 := #STEP_CHANGE_DELAY_DISK.Q;
   IF #_w1 THEN #ACTUAL_STEP_DISK := #ACTUAL_STEP_DISK + 1; END_IF;
END_REGION

REGION Network 13: STEP CHANGE GAS
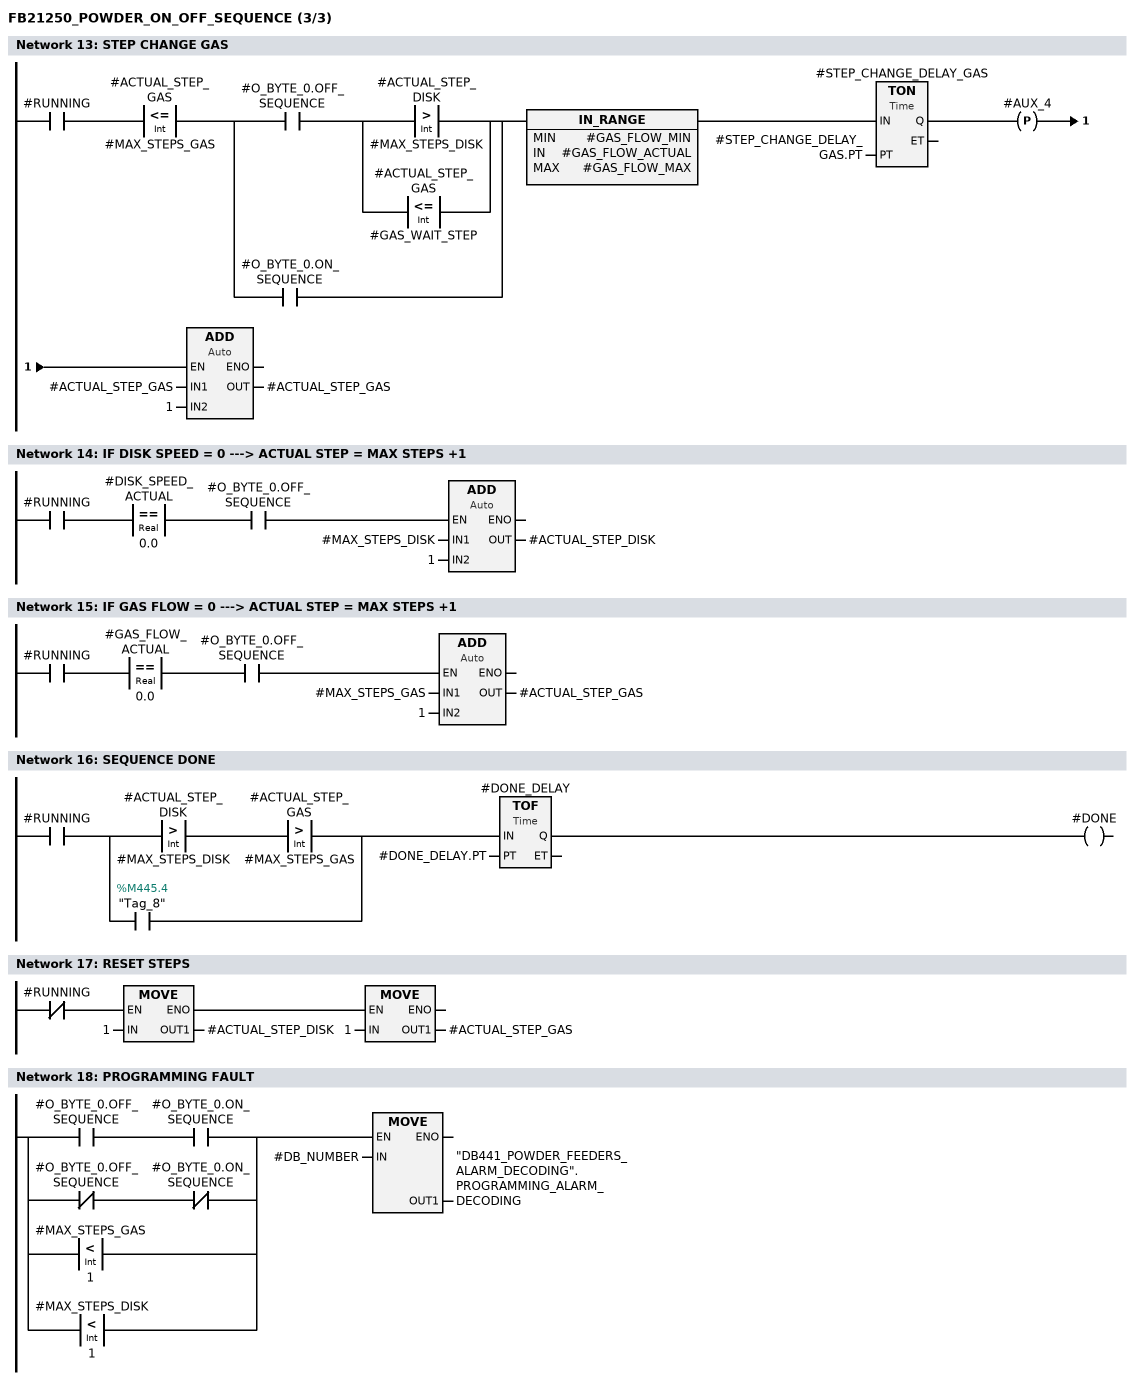
   RUNG wire#powerrail
      Contact( #RUNNING )
      { S7_Templates := "SrcType := Int" } LE_Contact(in1 := #ACTUAL_STEP_GAS, in2 := #MAX_STEPS_GAS)
      wire#w1
      Contact( #O_BYTE_0.OFF_SEQUENCE )
      wire#w2
      { S7_Templates := "SrcType := Int" } GT_Contact(in1 := #ACTUAL_STEP_DISK, in2 := #MAX_STEPS_DISK)
      wire#w3
      { S7_Templates := "SrcType := Real" } InRange(min := #GAS_FLOW_MIN, in := #GAS_FLOW_ACTUAL, max := #GAS_FLOW_MAX)
      { S7_Templates := "time_type := Time" } #STEP_CHANGE_DELAY_GAS.TON(pt := #STEP_CHANGE_DELAY_GAS.PT, et =>)
      P_Trig( #AUX_4 )
      Add(in1 := #ACTUAL_STEP_GAS, in2 := 1, out => #ACTUAL_STEP_GAS)
   END_RUNG
   RUNG wire#w2
      { S7_Templates := "SrcType := Int" } LE_Contact(in1 := #ACTUAL_STEP_GAS, in2 := #GAS_WAIT_STEP)
   END_RUNG wire#w3
   RUNG wire#w1
      Contact( #O_BYTE_0.ON_SEQUENCE )
   END_RUNG wire#w3
   // the same network as SCL:
   #STEP_CHANGE_DELAY_GAS(IN := #RUNNING AND (#ACTUAL_STEP_GAS <= #MAX_STEPS_GAS) AND ((#O_BYTE_0.OFF_SEQUENCE AND ((#ACTUAL_STEP_DISK > #MAX_STEPS_DISK) OR (#ACTUAL_STEP_GAS <= #GAS_WAIT_STEP))) OR #O_BYTE_0.ON_SEQUENCE) AND (#GAS_FLOW_MIN <= #GAS_FLOW_ACTUAL) AND (#GAS_FLOW_ACTUAL <= #GAS_FLOW_MAX),   // TON
                          PT := #STEP_CHANGE_DELAY_GAS.PT);
   #_w1 := #STEP_CHANGE_DELAY_GAS.Q AND NOT #AUX_4;   // rising edge
   #AUX_4 := #STEP_CHANGE_DELAY_GAS.Q;
   IF #_w1 THEN #ACTUAL_STEP_GAS := #ACTUAL_STEP_GAS + 1; END_IF;
END_REGION

REGION Network 14: IF DISK SPEED = 0 ---> ACTUAL STEP = MAX STEPS +1
   RUNG wire#powerrail
      Contact( #RUNNING )
      { S7_Templates := "SrcType := Real" } EQ_Contact(in1 := #DISK_SPEED_ACTUAL, in2 := 0.0)
      Contact( #O_BYTE_0.OFF_SEQUENCE )
      Add(in1 := #MAX_STEPS_DISK, in2 := 1, out => #ACTUAL_STEP_DISK)
   END_RUNG
   // the same network as SCL:
   IF #RUNNING AND (#DISK_SPEED_ACTUAL = 0.0) AND #O_BYTE_0.OFF_SEQUENCE THEN
       #ACTUAL_STEP_DISK := #MAX_STEPS_DISK + 1;
   END_IF;
END_REGION

REGION Network 15: IF GAS FLOW = 0 ---> ACTUAL STEP = MAX STEPS +1
   RUNG wire#powerrail
      Contact( #RUNNING )
      { S7_Templates := "SrcType := Real" } EQ_Contact(in1 := #GAS_FLOW_ACTUAL, in2 := 0.0)
      Contact( #O_BYTE_0.OFF_SEQUENCE )
      Add(in1 := #MAX_STEPS_GAS, in2 := 1, out => #ACTUAL_STEP_GAS)
   END_RUNG
   // the same network as SCL:
   IF #RUNNING AND (#GAS_FLOW_ACTUAL = 0.0) AND #O_BYTE_0.OFF_SEQUENCE THEN
       #ACTUAL_STEP_GAS := #MAX_STEPS_GAS + 1;
   END_IF;
END_REGION

REGION Network 16: SEQUENCE DONE
   RUNG wire#powerrail
      Contact( #RUNNING )
      wire#w1
      { S7_Templates := "SrcType := Int" } GT_Contact(in1 := #ACTUAL_STEP_DISK, in2 := #MAX_STEPS_DISK)
      { S7_Templates := "SrcType := Int" } GT_Contact(in1 := #ACTUAL_STEP_GAS, in2 := #MAX_STEPS_GAS)
      wire#w2
      { S7_Templates := "time_type := Time" } #DONE_DELAY.TOF(pt := #DONE_DELAY.PT, et =>)
      Coil( #DONE )
   END_RUNG
   RUNG wire#w1
      Contact( "Tag_8" )
   END_RUNG wire#w2
   // the same network as SCL:
   #DONE_DELAY(IN := #RUNNING AND (((#ACTUAL_STEP_DISK > #MAX_STEPS_DISK) AND (#ACTUAL_STEP_GAS > #MAX_STEPS_GAS)) OR "Tag_8"),   // TOF
               PT := #DONE_DELAY.PT);
   #DONE := #DONE_DELAY.Q;
END_REGION

REGION Network 17: RESET STEPS
   RUNG wire#powerrail
      I_Contact( #RUNNING )
      Move(in := 1, out1 => #ACTUAL_STEP_DISK)
      Move(in := 1, out1 => #ACTUAL_STEP_GAS)
   END_RUNG
   // the same network as SCL:
   IF NOT #RUNNING THEN
       #ACTUAL_STEP_DISK := 1;
       #ACTUAL_STEP_GAS := 1;
   END_IF;
END_REGION

REGION Network 18: PROGRAMMING FAULT
   RUNG wire#powerrail
      Contact( #O_BYTE_0.OFF_SEQUENCE )
      Contact( #O_BYTE_0.ON_SEQUENCE )
      wire#w1
      Move(in := #DB_NUMBER, out1 => "DB441_POWDER_FEEDERS_ALARM_DECODING".PROGRAMMING_ALARM_DECODING)
   END_RUNG
   RUNG wire#powerrail
      I_Contact( #O_BYTE_0.OFF_SEQUENCE )
      I_Contact( #O_BYTE_0.ON_SEQUENCE )
   END_RUNG wire#w1
   RUNG wire#powerrail
      { S7_Templates := "SrcType := Int" } LT_Contact(in1 := #MAX_STEPS_GAS, in2 := 1)
   END_RUNG wire#w1
   RUNG wire#powerrail
      { S7_Templates := "SrcType := Int" } LT_Contact(in1 := #MAX_STEPS_DISK, in2 := 1)
   END_RUNG wire#w1
   // the same network as SCL:
   IF (#O_BYTE_0.OFF_SEQUENCE AND #O_BYTE_0.ON_SEQUENCE) OR (NOT #O_BYTE_0.OFF_SEQUENCE AND NOT #O_BYTE_0.ON_SEQUENCE) OR (#MAX_STEPS_GAS < 1) OR (#MAX_STEPS_DISK < 1) THEN
       "DB441_POWDER_FEEDERS_ALARM_DECODING".PROGRAMMING_ALARM_DECODING := #DB_NUMBER;
   END_IF;
END_REGION
END_FUNCTION_BLOCK

FUNCTION "FC21014_POWDER_FEEDER_PROFINET" : Void   // FC21014, LAD
TITLE = FC21014 POWDER FEEDER PROFINET
{ S7_Optimized_Access := 'TRUE' }
VERSION : 0.1
// stored: AutoNumber false, IsIECCheckEnabled false, SetENOAutomatically false, UDAEnableTagReadback false
BEGIN

REGION Network 1: /////_UNIT_01_/////
END_REGION

REGION Network 2: CALL FB21014 POWDER FEEDER 1 PROFINET UNIT 01
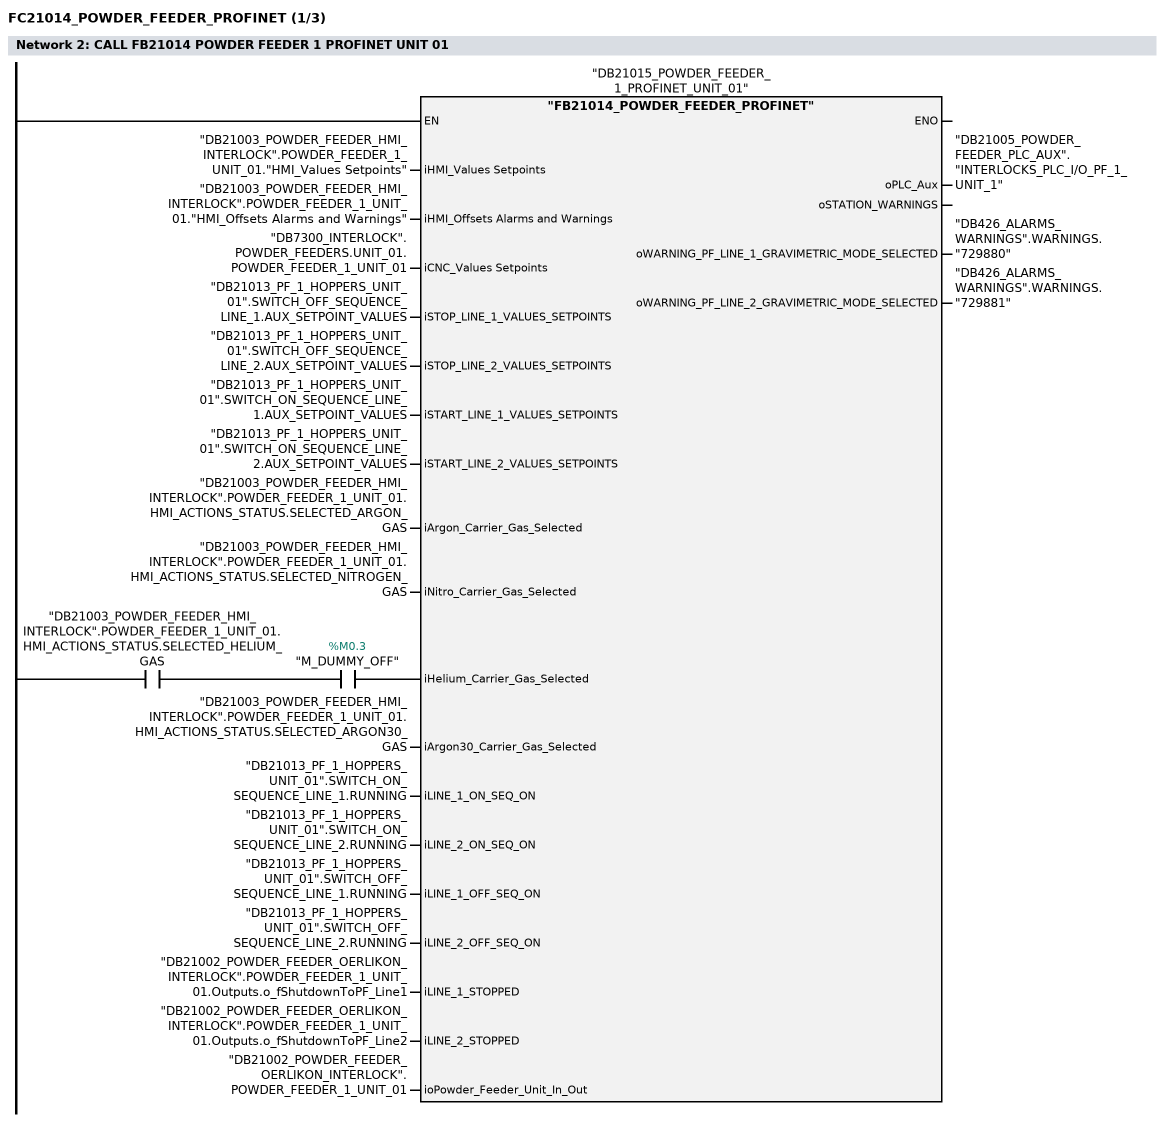
   RUNG wire#powerrail
      "DB21015_POWDER_FEEDER_1_PROFINET_UNIT_01"(iHelium_Carrier_Gas_Selected := wire#w1, "iHMI_Values Setpoints" := "DB21003_POWDER_FEEDER_HMI_INTERLOCK".POWDER_FEEDER_1_UNIT_01."HMI_Values Setpoints", "iHMI_Offsets Alarms and Warnings" := "DB21003_POWDER_FEEDER_HMI_INTERLOCK".POWDER_FEEDER_1_UNIT_01."HMI_Offsets Alarms and Warnings", "iCNC_Values Setpoints" := "DB7300_INTERLOCK".POWDER_FEEDERS.UNIT_01.POWDER_FEEDER_1_UNIT_01, iSTOP_LINE_1_VALUES_SETPOINTS := "DB21013_PF_1_HOPPERS_UNIT_01".SWITCH_OFF_SEQUENCE_LINE_1.AUX_SETPOINT_VALUES, iSTOP_LINE_2_VALUES_SETPOINTS := "DB21013_PF_1_HOPPERS_UNIT_01".SWITCH_OFF_SEQUENCE_LINE_2.AUX_SETPOINT_VALUES, iSTART_LINE_1_VALUES_SETPOINTS := "DB21013_PF_1_HOPPERS_UNIT_01".SWITCH_ON_SEQUENCE_LINE_1.AUX_SETPOINT_VALUES, iSTART_LINE_2_VALUES_SETPOINTS := "DB21013_PF_1_HOPPERS_UNIT_01".SWITCH_ON_SEQUENCE_LINE_2.AUX_SETPOINT_VALUES, iArgon_Carrier_Gas_Selected := "DB21003_POWDER_FEEDER_HMI_INTERLOCK".POWDER_FEEDER_1_UNIT_01.HMI_ACTIONS_STATUS.SELECTED_ARGON_GAS, iNitro_Carrier_Gas_Selected := "DB21003_POWDER_FEEDER_HMI_INTERLOCK".POWDER_FEEDER_1_UNIT_01.HMI_ACTIONS_STATUS.SELECTED_NITROGEN_GAS, iArgon30_Carrier_Gas_Selected := "DB21003_POWDER_FEEDER_HMI_INTERLOCK".POWDER_FEEDER_1_UNIT_01.HMI_ACTIONS_STATUS.SELECTED_ARGON30_GAS, iLINE_1_ON_SEQ_ON := "DB21013_PF_1_HOPPERS_UNIT_01".SWITCH_ON_SEQUENCE_LINE_1.RUNNING, iLINE_2_ON_SEQ_ON := "DB21013_PF_1_HOPPERS_UNIT_01".SWITCH_ON_SEQUENCE_LINE_2.RUNNING, iLINE_1_OFF_SEQ_ON := "DB21013_PF_1_HOPPERS_UNIT_01".SWITCH_OFF_SEQUENCE_LINE_1.RUNNING, iLINE_2_OFF_SEQ_ON := "DB21013_PF_1_HOPPERS_UNIT_01".SWITCH_OFF_SEQUENCE_LINE_2.RUNNING, iLINE_1_STOPPED := "DB21002_POWDER_FEEDER_OERLIKON_INTERLOCK".POWDER_FEEDER_1_UNIT_01.Outputs.o_fShutdownToPF_Line1, iLINE_2_STOPPED := "DB21002_POWDER_FEEDER_OERLIKON_INTERLOCK".POWDER_FEEDER_1_UNIT_01.Outputs.o_fShutdownToPF_Line2, ioPowder_Feeder_Unit_In_Out := "DB21002_POWDER_FEEDER_OERLIKON_INTERLOCK".POWDER_FEEDER_1_UNIT_01, oPLC_Aux => "DB21005_POWDER_FEEDER_PLC_AUX"."INTERLOCKS_PLC_I/O_PF_1_UNIT_1", oSTATION_WARNINGS =>, oWARNING_PF_LINE_1_GRAVIMETRIC_MODE_SELECTED => "DB426_ALARMS_WARNINGS".WARNINGS."729880", oWARNING_PF_LINE_2_GRAVIMETRIC_MODE_SELECTED => "DB426_ALARMS_WARNINGS".WARNINGS."729881")
   END_RUNG
   RUNG wire#powerrail
      Contact( "DB21003_POWDER_FEEDER_HMI_INTERLOCK".POWDER_FEEDER_1_UNIT_01.HMI_ACTIONS_STATUS.SELECTED_HELIUM_GAS )
      Contact( "M_DUMMY_OFF" )
   END_RUNG wire#w1
   // the same network as SCL:
   "DB21015_POWDER_FEEDER_1_PROFINET_UNIT_01"("iHMI_Values Setpoints" := "DB21003_POWDER_FEEDER_HMI_INTERLOCK".POWDER_FEEDER_1_UNIT_01."HMI_Values Setpoints",   // "FB21014_POWDER_FEEDER_PROFINET"
                           "iHMI_Offsets Alarms and Warnings" := "DB21003_POWDER_FEEDER_HMI_INTERLOCK".POWDER_FEEDER_1_UNIT_01."HMI_Offsets Alarms and Warnings",
                           "iCNC_Values Setpoints" := "DB7300_INTERLOCK".POWDER_FEEDERS.UNIT_01.POWDER_FEEDER_1_UNIT_01,
                           iSTOP_LINE_1_VALUES_SETPOINTS := "DB21013_PF_1_HOPPERS_UNIT_01".SWITCH_OFF_SEQUENCE_LINE_1.AUX_SETPOINT_VALUES,
                           iSTOP_LINE_2_VALUES_SETPOINTS := "DB21013_PF_1_HOPPERS_UNIT_01".SWITCH_OFF_SEQUENCE_LINE_2.AUX_SETPOINT_VALUES,
                           iSTART_LINE_1_VALUES_SETPOINTS := "DB21013_PF_1_HOPPERS_UNIT_01".SWITCH_ON_SEQUENCE_LINE_1.AUX_SETPOINT_VALUES,
                           iSTART_LINE_2_VALUES_SETPOINTS := "DB21013_PF_1_HOPPERS_UNIT_01".SWITCH_ON_SEQUENCE_LINE_2.AUX_SETPOINT_VALUES,
                           iArgon_Carrier_Gas_Selected := "DB21003_POWDER_FEEDER_HMI_INTERLOCK".POWDER_FEEDER_1_UNIT_01.HMI_ACTIONS_STATUS.SELECTED_ARGON_GAS,
                           iNitro_Carrier_Gas_Selected := "DB21003_POWDER_FEEDER_HMI_INTERLOCK".POWDER_FEEDER_1_UNIT_01.HMI_ACTIONS_STATUS.SELECTED_NITROGEN_GAS,
                           iHelium_Carrier_Gas_Selected := "DB21003_POWDER_FEEDER_HMI_INTERLOCK".POWDER_FEEDER_1_UNIT_01.HMI_ACTIONS_STATUS.SELECTED_HELIUM_GAS AND "M_DUMMY_OFF",
                           iArgon30_Carrier_Gas_Selected := "DB21003_POWDER_FEEDER_HMI_INTERLOCK".POWDER_FEEDER_1_UNIT_01.HMI_ACTIONS_STATUS.SELECTED_ARGON30_GAS,
                           iLINE_1_ON_SEQ_ON := "DB21013_PF_1_HOPPERS_UNIT_01".SWITCH_ON_SEQUENCE_LINE_1.RUNNING,
                           iLINE_2_ON_SEQ_ON := "DB21013_PF_1_HOPPERS_UNIT_01".SWITCH_ON_SEQUENCE_LINE_2.RUNNING,
                           iLINE_1_OFF_SEQ_ON := "DB21013_PF_1_HOPPERS_UNIT_01".SWITCH_OFF_SEQUENCE_LINE_1.RUNNING,
                           iLINE_2_OFF_SEQ_ON := "DB21013_PF_1_HOPPERS_UNIT_01".SWITCH_OFF_SEQUENCE_LINE_2.RUNNING,
                           iLINE_1_STOPPED := "DB21002_POWDER_FEEDER_OERLIKON_INTERLOCK".POWDER_FEEDER_1_UNIT_01.Outputs.o_fShutdownToPF_Line1,
                           iLINE_2_STOPPED := "DB21002_POWDER_FEEDER_OERLIKON_INTERLOCK".POWDER_FEEDER_1_UNIT_01.Outputs.o_fShutdownToPF_Line2,
                           ioPowder_Feeder_Unit_In_Out := "DB21002_POWDER_FEEDER_OERLIKON_INTERLOCK".POWDER_FEEDER_1_UNIT_01,
                           oPLC_Aux => "DB21005_POWDER_FEEDER_PLC_AUX"."INTERLOCKS_PLC_I/O_PF_1_UNIT_1",
                           oWARNING_PF_LINE_1_GRAVIMETRIC_MODE_SELECTED => "DB426_ALARMS_WARNINGS".WARNINGS."729880",
                           oWARNING_PF_LINE_2_GRAVIMETRIC_MODE_SELECTED => "DB426_ALARMS_WARNINGS".WARNINGS."729881");
END_REGION

REGION Network 3: /////_UNIT_02_/////
END_REGION

REGION Network 4: CALL FB21014 POWDER FEEDER 1 PROFINET UNIT 02
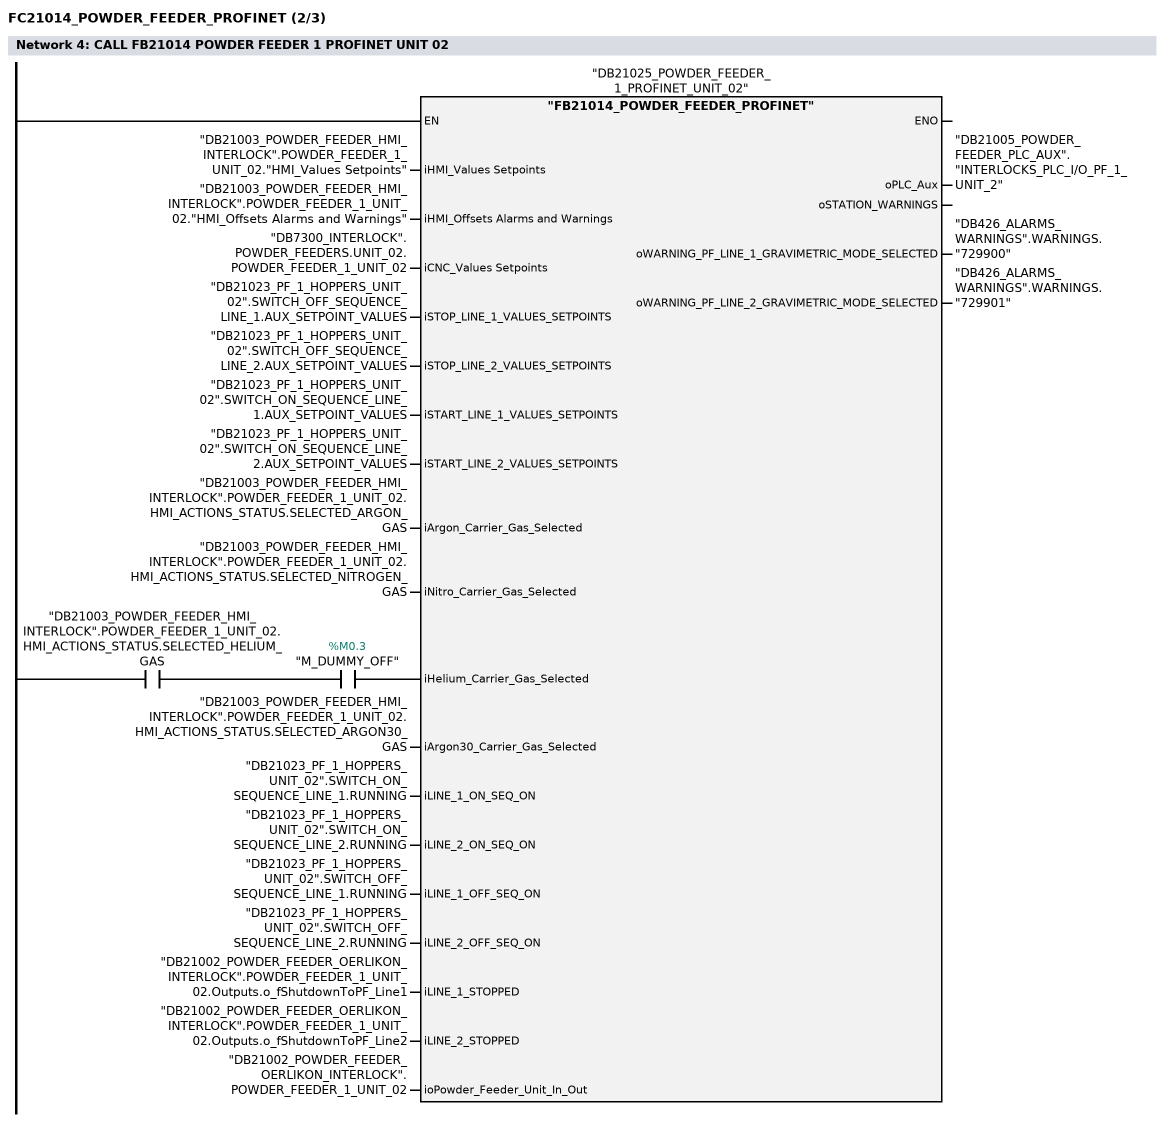
   RUNG wire#powerrail
      "DB21025_POWDER_FEEDER_1_PROFINET_UNIT_02"(iHelium_Carrier_Gas_Selected := wire#w1, "iHMI_Values Setpoints" := "DB21003_POWDER_FEEDER_HMI_INTERLOCK".POWDER_FEEDER_1_UNIT_02."HMI_Values Setpoints", "iHMI_Offsets Alarms and Warnings" := "DB21003_POWDER_FEEDER_HMI_INTERLOCK".POWDER_FEEDER_1_UNIT_02."HMI_Offsets Alarms and Warnings", "iCNC_Values Setpoints" := "DB7300_INTERLOCK".POWDER_FEEDERS.UNIT_02.POWDER_FEEDER_1_UNIT_02, iSTOP_LINE_1_VALUES_SETPOINTS := "DB21023_PF_1_HOPPERS_UNIT_02".SWITCH_OFF_SEQUENCE_LINE_1.AUX_SETPOINT_VALUES, iSTOP_LINE_2_VALUES_SETPOINTS := "DB21023_PF_1_HOPPERS_UNIT_02".SWITCH_OFF_SEQUENCE_LINE_2.AUX_SETPOINT_VALUES, iSTART_LINE_1_VALUES_SETPOINTS := "DB21023_PF_1_HOPPERS_UNIT_02".SWITCH_ON_SEQUENCE_LINE_1.AUX_SETPOINT_VALUES, iSTART_LINE_2_VALUES_SETPOINTS := "DB21023_PF_1_HOPPERS_UNIT_02".SWITCH_ON_SEQUENCE_LINE_2.AUX_SETPOINT_VALUES, iArgon_Carrier_Gas_Selected := "DB21003_POWDER_FEEDER_HMI_INTERLOCK".POWDER_FEEDER_1_UNIT_02.HMI_ACTIONS_STATUS.SELECTED_ARGON_GAS, iNitro_Carrier_Gas_Selected := "DB21003_POWDER_FEEDER_HMI_INTERLOCK".POWDER_FEEDER_1_UNIT_02.HMI_ACTIONS_STATUS.SELECTED_NITROGEN_GAS, iArgon30_Carrier_Gas_Selected := "DB21003_POWDER_FEEDER_HMI_INTERLOCK".POWDER_FEEDER_1_UNIT_02.HMI_ACTIONS_STATUS.SELECTED_ARGON30_GAS, iLINE_1_ON_SEQ_ON := "DB21023_PF_1_HOPPERS_UNIT_02".SWITCH_ON_SEQUENCE_LINE_1.RUNNING, iLINE_2_ON_SEQ_ON := "DB21023_PF_1_HOPPERS_UNIT_02".SWITCH_ON_SEQUENCE_LINE_2.RUNNING, iLINE_1_OFF_SEQ_ON := "DB21023_PF_1_HOPPERS_UNIT_02".SWITCH_OFF_SEQUENCE_LINE_1.RUNNING, iLINE_2_OFF_SEQ_ON := "DB21023_PF_1_HOPPERS_UNIT_02".SWITCH_OFF_SEQUENCE_LINE_2.RUNNING, iLINE_1_STOPPED := "DB21002_POWDER_FEEDER_OERLIKON_INTERLOCK".POWDER_FEEDER_1_UNIT_02.Outputs.o_fShutdownToPF_Line1, iLINE_2_STOPPED := "DB21002_POWDER_FEEDER_OERLIKON_INTERLOCK".POWDER_FEEDER_1_UNIT_02.Outputs.o_fShutdownToPF_Line2, ioPowder_Feeder_Unit_In_Out := "DB21002_POWDER_FEEDER_OERLIKON_INTERLOCK".POWDER_FEEDER_1_UNIT_02, oPLC_Aux => "DB21005_POWDER_FEEDER_PLC_AUX"."INTERLOCKS_PLC_I/O_PF_1_UNIT_2", oSTATION_WARNINGS =>, oWARNING_PF_LINE_1_GRAVIMETRIC_MODE_SELECTED => "DB426_ALARMS_WARNINGS".WARNINGS."729900", oWARNING_PF_LINE_2_GRAVIMETRIC_MODE_SELECTED => "DB426_ALARMS_WARNINGS".WARNINGS."729901")
   END_RUNG
   RUNG wire#powerrail
      Contact( "DB21003_POWDER_FEEDER_HMI_INTERLOCK".POWDER_FEEDER_1_UNIT_02.HMI_ACTIONS_STATUS.SELECTED_HELIUM_GAS )
      Contact( "M_DUMMY_OFF" )
   END_RUNG wire#w1
   // the same network as SCL:
   "DB21025_POWDER_FEEDER_1_PROFINET_UNIT_02"("iHMI_Values Setpoints" := "DB21003_POWDER_FEEDER_HMI_INTERLOCK".POWDER_FEEDER_1_UNIT_02."HMI_Values Setpoints",   // "FB21014_POWDER_FEEDER_PROFINET"
                           "iHMI_Offsets Alarms and Warnings" := "DB21003_POWDER_FEEDER_HMI_INTERLOCK".POWDER_FEEDER_1_UNIT_02."HMI_Offsets Alarms and Warnings",
                           "iCNC_Values Setpoints" := "DB7300_INTERLOCK".POWDER_FEEDERS.UNIT_02.POWDER_FEEDER_1_UNIT_02,
                           iSTOP_LINE_1_VALUES_SETPOINTS := "DB21023_PF_1_HOPPERS_UNIT_02".SWITCH_OFF_SEQUENCE_LINE_1.AUX_SETPOINT_VALUES,
                           iSTOP_LINE_2_VALUES_SETPOINTS := "DB21023_PF_1_HOPPERS_UNIT_02".SWITCH_OFF_SEQUENCE_LINE_2.AUX_SETPOINT_VALUES,
                           iSTART_LINE_1_VALUES_SETPOINTS := "DB21023_PF_1_HOPPERS_UNIT_02".SWITCH_ON_SEQUENCE_LINE_1.AUX_SETPOINT_VALUES,
                           iSTART_LINE_2_VALUES_SETPOINTS := "DB21023_PF_1_HOPPERS_UNIT_02".SWITCH_ON_SEQUENCE_LINE_2.AUX_SETPOINT_VALUES,
                           iArgon_Carrier_Gas_Selected := "DB21003_POWDER_FEEDER_HMI_INTERLOCK".POWDER_FEEDER_1_UNIT_02.HMI_ACTIONS_STATUS.SELECTED_ARGON_GAS,
                           iNitro_Carrier_Gas_Selected := "DB21003_POWDER_FEEDER_HMI_INTERLOCK".POWDER_FEEDER_1_UNIT_02.HMI_ACTIONS_STATUS.SELECTED_NITROGEN_GAS,
                           iHelium_Carrier_Gas_Selected := "DB21003_POWDER_FEEDER_HMI_INTERLOCK".POWDER_FEEDER_1_UNIT_02.HMI_ACTIONS_STATUS.SELECTED_HELIUM_GAS AND "M_DUMMY_OFF",
                           iArgon30_Carrier_Gas_Selected := "DB21003_POWDER_FEEDER_HMI_INTERLOCK".POWDER_FEEDER_1_UNIT_02.HMI_ACTIONS_STATUS.SELECTED_ARGON30_GAS,
                           iLINE_1_ON_SEQ_ON := "DB21023_PF_1_HOPPERS_UNIT_02".SWITCH_ON_SEQUENCE_LINE_1.RUNNING,
                           iLINE_2_ON_SEQ_ON := "DB21023_PF_1_HOPPERS_UNIT_02".SWITCH_ON_SEQUENCE_LINE_2.RUNNING,
                           iLINE_1_OFF_SEQ_ON := "DB21023_PF_1_HOPPERS_UNIT_02".SWITCH_OFF_SEQUENCE_LINE_1.RUNNING,
                           iLINE_2_OFF_SEQ_ON := "DB21023_PF_1_HOPPERS_UNIT_02".SWITCH_OFF_SEQUENCE_LINE_2.RUNNING,
                           iLINE_1_STOPPED := "DB21002_POWDER_FEEDER_OERLIKON_INTERLOCK".POWDER_FEEDER_1_UNIT_02.Outputs.o_fShutdownToPF_Line1,
                           iLINE_2_STOPPED := "DB21002_POWDER_FEEDER_OERLIKON_INTERLOCK".POWDER_FEEDER_1_UNIT_02.Outputs.o_fShutdownToPF_Line2,
                           ioPowder_Feeder_Unit_In_Out := "DB21002_POWDER_FEEDER_OERLIKON_INTERLOCK".POWDER_FEEDER_1_UNIT_02,
                           oPLC_Aux => "DB21005_POWDER_FEEDER_PLC_AUX"."INTERLOCKS_PLC_I/O_PF_1_UNIT_2",
                           oWARNING_PF_LINE_1_GRAVIMETRIC_MODE_SELECTED => "DB426_ALARMS_WARNINGS".WARNINGS."729900",
                           oWARNING_PF_LINE_2_GRAVIMETRIC_MODE_SELECTED => "DB426_ALARMS_WARNINGS".WARNINGS."729901");
END_REGION

REGION Network 5: CALL FB21014 POWDER FEEDER 2 PROFINET UNIT 02
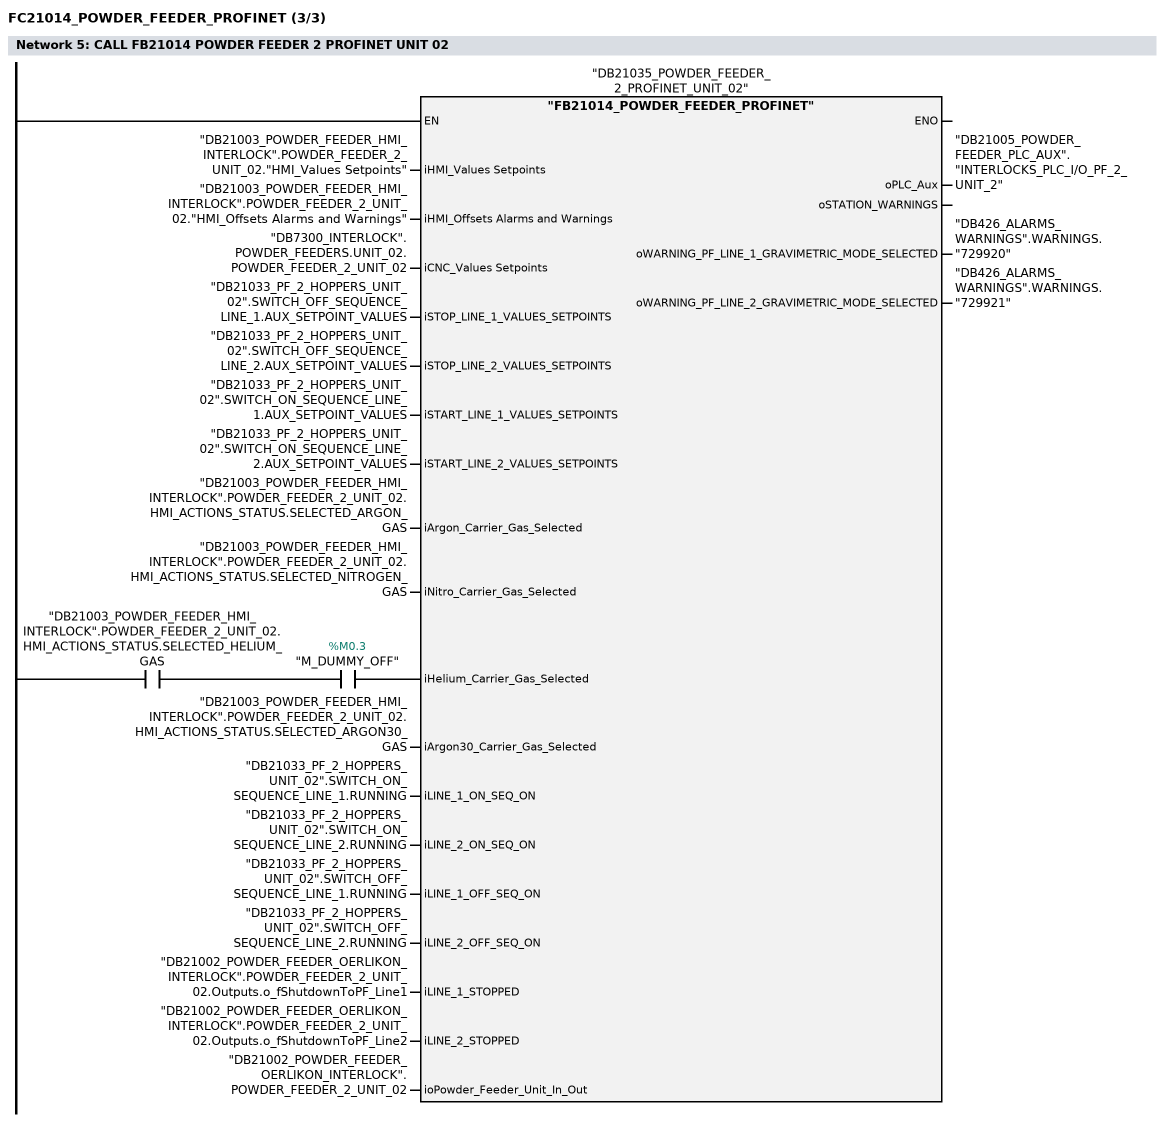
   RUNG wire#powerrail
      "DB21035_POWDER_FEEDER_2_PROFINET_UNIT_02"(iHelium_Carrier_Gas_Selected := wire#w1, "iHMI_Values Setpoints" := "DB21003_POWDER_FEEDER_HMI_INTERLOCK".POWDER_FEEDER_2_UNIT_02."HMI_Values Setpoints", "iHMI_Offsets Alarms and Warnings" := "DB21003_POWDER_FEEDER_HMI_INTERLOCK".POWDER_FEEDER_2_UNIT_02."HMI_Offsets Alarms and Warnings", "iCNC_Values Setpoints" := "DB7300_INTERLOCK".POWDER_FEEDERS.UNIT_02.POWDER_FEEDER_2_UNIT_02, iSTOP_LINE_1_VALUES_SETPOINTS := "DB21033_PF_2_HOPPERS_UNIT_02".SWITCH_OFF_SEQUENCE_LINE_1.AUX_SETPOINT_VALUES, iSTOP_LINE_2_VALUES_SETPOINTS := "DB21033_PF_2_HOPPERS_UNIT_02".SWITCH_OFF_SEQUENCE_LINE_2.AUX_SETPOINT_VALUES, iSTART_LINE_1_VALUES_SETPOINTS := "DB21033_PF_2_HOPPERS_UNIT_02".SWITCH_ON_SEQUENCE_LINE_1.AUX_SETPOINT_VALUES, iSTART_LINE_2_VALUES_SETPOINTS := "DB21033_PF_2_HOPPERS_UNIT_02".SWITCH_ON_SEQUENCE_LINE_2.AUX_SETPOINT_VALUES, iArgon_Carrier_Gas_Selected := "DB21003_POWDER_FEEDER_HMI_INTERLOCK".POWDER_FEEDER_2_UNIT_02.HMI_ACTIONS_STATUS.SELECTED_ARGON_GAS, iNitro_Carrier_Gas_Selected := "DB21003_POWDER_FEEDER_HMI_INTERLOCK".POWDER_FEEDER_2_UNIT_02.HMI_ACTIONS_STATUS.SELECTED_NITROGEN_GAS, iArgon30_Carrier_Gas_Selected := "DB21003_POWDER_FEEDER_HMI_INTERLOCK".POWDER_FEEDER_2_UNIT_02.HMI_ACTIONS_STATUS.SELECTED_ARGON30_GAS, iLINE_1_ON_SEQ_ON := "DB21033_PF_2_HOPPERS_UNIT_02".SWITCH_ON_SEQUENCE_LINE_1.RUNNING, iLINE_2_ON_SEQ_ON := "DB21033_PF_2_HOPPERS_UNIT_02".SWITCH_ON_SEQUENCE_LINE_2.RUNNING, iLINE_1_OFF_SEQ_ON := "DB21033_PF_2_HOPPERS_UNIT_02".SWITCH_OFF_SEQUENCE_LINE_1.RUNNING, iLINE_2_OFF_SEQ_ON := "DB21033_PF_2_HOPPERS_UNIT_02".SWITCH_OFF_SEQUENCE_LINE_2.RUNNING, iLINE_1_STOPPED := "DB21002_POWDER_FEEDER_OERLIKON_INTERLOCK".POWDER_FEEDER_2_UNIT_02.Outputs.o_fShutdownToPF_Line1, iLINE_2_STOPPED := "DB21002_POWDER_FEEDER_OERLIKON_INTERLOCK".POWDER_FEEDER_2_UNIT_02.Outputs.o_fShutdownToPF_Line2, ioPowder_Feeder_Unit_In_Out := "DB21002_POWDER_FEEDER_OERLIKON_INTERLOCK".POWDER_FEEDER_2_UNIT_02, oPLC_Aux => "DB21005_POWDER_FEEDER_PLC_AUX"."INTERLOCKS_PLC_I/O_PF_2_UNIT_2", oSTATION_WARNINGS =>, oWARNING_PF_LINE_1_GRAVIMETRIC_MODE_SELECTED => "DB426_ALARMS_WARNINGS".WARNINGS."729920", oWARNING_PF_LINE_2_GRAVIMETRIC_MODE_SELECTED => "DB426_ALARMS_WARNINGS".WARNINGS."729921")
   END_RUNG
   RUNG wire#powerrail
      Contact( "DB21003_POWDER_FEEDER_HMI_INTERLOCK".POWDER_FEEDER_2_UNIT_02.HMI_ACTIONS_STATUS.SELECTED_HELIUM_GAS )
      Contact( "M_DUMMY_OFF" )
   END_RUNG wire#w1
   // the same network as SCL:
   "DB21035_POWDER_FEEDER_2_PROFINET_UNIT_02"("iHMI_Values Setpoints" := "DB21003_POWDER_FEEDER_HMI_INTERLOCK".POWDER_FEEDER_2_UNIT_02."HMI_Values Setpoints",   // "FB21014_POWDER_FEEDER_PROFINET"
                           "iHMI_Offsets Alarms and Warnings" := "DB21003_POWDER_FEEDER_HMI_INTERLOCK".POWDER_FEEDER_2_UNIT_02."HMI_Offsets Alarms and Warnings",
                           "iCNC_Values Setpoints" := "DB7300_INTERLOCK".POWDER_FEEDERS.UNIT_02.POWDER_FEEDER_2_UNIT_02,
                           iSTOP_LINE_1_VALUES_SETPOINTS := "DB21033_PF_2_HOPPERS_UNIT_02".SWITCH_OFF_SEQUENCE_LINE_1.AUX_SETPOINT_VALUES,
                           iSTOP_LINE_2_VALUES_SETPOINTS := "DB21033_PF_2_HOPPERS_UNIT_02".SWITCH_OFF_SEQUENCE_LINE_2.AUX_SETPOINT_VALUES,
                           iSTART_LINE_1_VALUES_SETPOINTS := "DB21033_PF_2_HOPPERS_UNIT_02".SWITCH_ON_SEQUENCE_LINE_1.AUX_SETPOINT_VALUES,
                           iSTART_LINE_2_VALUES_SETPOINTS := "DB21033_PF_2_HOPPERS_UNIT_02".SWITCH_ON_SEQUENCE_LINE_2.AUX_SETPOINT_VALUES,
                           iArgon_Carrier_Gas_Selected := "DB21003_POWDER_FEEDER_HMI_INTERLOCK".POWDER_FEEDER_2_UNIT_02.HMI_ACTIONS_STATUS.SELECTED_ARGON_GAS,
                           iNitro_Carrier_Gas_Selected := "DB21003_POWDER_FEEDER_HMI_INTERLOCK".POWDER_FEEDER_2_UNIT_02.HMI_ACTIONS_STATUS.SELECTED_NITROGEN_GAS,
                           iHelium_Carrier_Gas_Selected := "DB21003_POWDER_FEEDER_HMI_INTERLOCK".POWDER_FEEDER_2_UNIT_02.HMI_ACTIONS_STATUS.SELECTED_HELIUM_GAS AND "M_DUMMY_OFF",
                           iArgon30_Carrier_Gas_Selected := "DB21003_POWDER_FEEDER_HMI_INTERLOCK".POWDER_FEEDER_2_UNIT_02.HMI_ACTIONS_STATUS.SELECTED_ARGON30_GAS,
                           iLINE_1_ON_SEQ_ON := "DB21033_PF_2_HOPPERS_UNIT_02".SWITCH_ON_SEQUENCE_LINE_1.RUNNING,
                           iLINE_2_ON_SEQ_ON := "DB21033_PF_2_HOPPERS_UNIT_02".SWITCH_ON_SEQUENCE_LINE_2.RUNNING,
                           iLINE_1_OFF_SEQ_ON := "DB21033_PF_2_HOPPERS_UNIT_02".SWITCH_OFF_SEQUENCE_LINE_1.RUNNING,
                           iLINE_2_OFF_SEQ_ON := "DB21033_PF_2_HOPPERS_UNIT_02".SWITCH_OFF_SEQUENCE_LINE_2.RUNNING,
                           iLINE_1_STOPPED := "DB21002_POWDER_FEEDER_OERLIKON_INTERLOCK".POWDER_FEEDER_2_UNIT_02.Outputs.o_fShutdownToPF_Line1,
                           iLINE_2_STOPPED := "DB21002_POWDER_FEEDER_OERLIKON_INTERLOCK".POWDER_FEEDER_2_UNIT_02.Outputs.o_fShutdownToPF_Line2,
                           ioPowder_Feeder_Unit_In_Out := "DB21002_POWDER_FEEDER_OERLIKON_INTERLOCK".POWDER_FEEDER_2_UNIT_02,
                           oPLC_Aux => "DB21005_POWDER_FEEDER_PLC_AUX"."INTERLOCKS_PLC_I/O_PF_2_UNIT_2",
                           oWARNING_PF_LINE_1_GRAVIMETRIC_MODE_SELECTED => "DB426_ALARMS_WARNINGS".WARNINGS."729920",
                           oWARNING_PF_LINE_2_GRAVIMETRIC_MODE_SELECTED => "DB426_ALARMS_WARNINGS".WARNINGS."729921");
END_REGION
END_FUNCTION

FUNCTION_BLOCK "FB21014_POWDER_FEEDER_PROFINET"   // FB21014, LAD
TITLE = FB21014 POWDER FEEDER PROFINET
{ S7_Optimized_Access := 'FALSE' }
VERSION : 0.1
// stored: AutoNumber false, IsIECCheckEnabled false, SetENOAutomatically false, UDAEnableTagReadback false
   VAR_INPUT
      "iHMI_Values Setpoints" : "POWDER FEEDER HMI VALUES SETPOINTS";
      "iHMI_Offsets Alarms and Warnings" : "POWDER FEEDER HMI OFFSETS ALARMS WARNINGS";
      "iCNC_Values Setpoints" : "POWDER FEEDER CNC VALUES SETPOINTS";
      iSTOP_LINE_1_VALUES_SETPOINTS : Struct
         LINE_1_GAS_FLOW : Real;   // LINE 1 GAS FLOW SETPOINT
         LINE_1_DISK_SPEED : Real;   // LINE 1 DISK SPEED SETPOINT
      END_STRUCT;
      iSTOP_LINE_2_VALUES_SETPOINTS : Struct
         LINE_2_GAS_FLOW : Real;   // LINE 2 GAS FLOW SETPOINT
         LINE_2_DISK_SPEED : Real;   // LINE 2 DISK SPEED SETPOINT
      END_STRUCT;
      iSTART_LINE_1_VALUES_SETPOINTS : Struct
         LINE_1_GAS_FLOW : Real;   // LINE 1 GAS FLOW SETPOINT
         LINE_1_DISK_SPEED : Real;   // LINE 1 DISK SPEED SETPOINT
      END_STRUCT;
      iSTART_LINE_2_VALUES_SETPOINTS : Struct
         LINE_2_GAS_FLOW : Real;   // LINE 2 GAS FLOW SETPOINT
         LINE_2_DISK_SPEED : Real;   // LINE 2 DISK SPEED SETPOINT
      END_STRUCT;
      iArgon_Carrier_Gas_Selected : Bool;
      iNitro_Carrier_Gas_Selected : Bool;
      iHelium_Carrier_Gas_Selected : Bool;
      iArgon30_Carrier_Gas_Selected : Bool;
      iLINE_1_ON_SEQ_ON : Bool;
      iLINE_2_ON_SEQ_ON : Bool;
      iLINE_1_OFF_SEQ_ON : Bool;
      iLINE_2_OFF_SEQ_ON : Bool;
      iLINE_1_STOPPED : Bool;   // HOPPER LINE 1 STOPPPED
      iLINE_2_STOPPED : Bool;   // HOPPER LINE 2 STOPPPED
   END_VAR
   VAR_OUTPUT
      oPLC_Aux : "POWDER FEEDER PLC AUXILIAR";
      oSTATION_WARNINGS : Bool;
      oWARNING_PF_LINE_1_GRAVIMETRIC_MODE_SELECTED : Bool;
      oWARNING_PF_LINE_2_GRAVIMETRIC_MODE_SELECTED : Bool;
   END_VAR
   VAR_IN_OUT
      ioPowder_Feeder_Unit_In_Out : "POWDER FEEDER OERLIKON";
   END_VAR
   VAR DB_SPECIFIC
      INPUT_SETTINGS : Struct
         UNIT_NUMBER : Int;
         FEEDER_NUMBER : Int;
      END_STRUCT;
      AUX_MANUAL_GAS_LINE_1 : Bool;   // AUX MANUAL GAS LINE 1
      AUX_MANUAL_GAS_LINE_2 : Bool;   // AUX MANUAL GAS LINE 2
      AUX_MANUAL_DISK_LINE_1 : Bool;   // AUX MANUAL DISK LINE 1
      AUX_MANUAL_DISK_LINE_2 : Bool;   // AUX MANUAL DISK LINE 2
      swapped : Word;
   END_VAR
   VAR_TEMP
      HMI_INPUT_MAN_MODE : Bool;
      OPTIONS_ON : Bool;
      OPTIONS_OFF : Bool;
      "VOLUMETRIC/GRAVIMETRIC" : Bool;
      "¿SUSTITUIR_VAR_CNC?" : Real;
      Retval_Fill_R : Real;
      DB_NUMBER : DInt;
   END_VAR
   VAR_TEMP   // added for the SCL form of the ladder/FBD networks
      _w1 : Bool;
   END_VAR
BEGIN

NETWORK
TITLE = READ INSTANCE DB NUMBER
      L     DINO;
      +     10#800000;
      T     #DB_NUMBER;

REGION Network 2: HMI INPUT
   // With Hmi Input we allow for user manipulation of feeder operating parameters. If not, they get overriden by robot interlock.
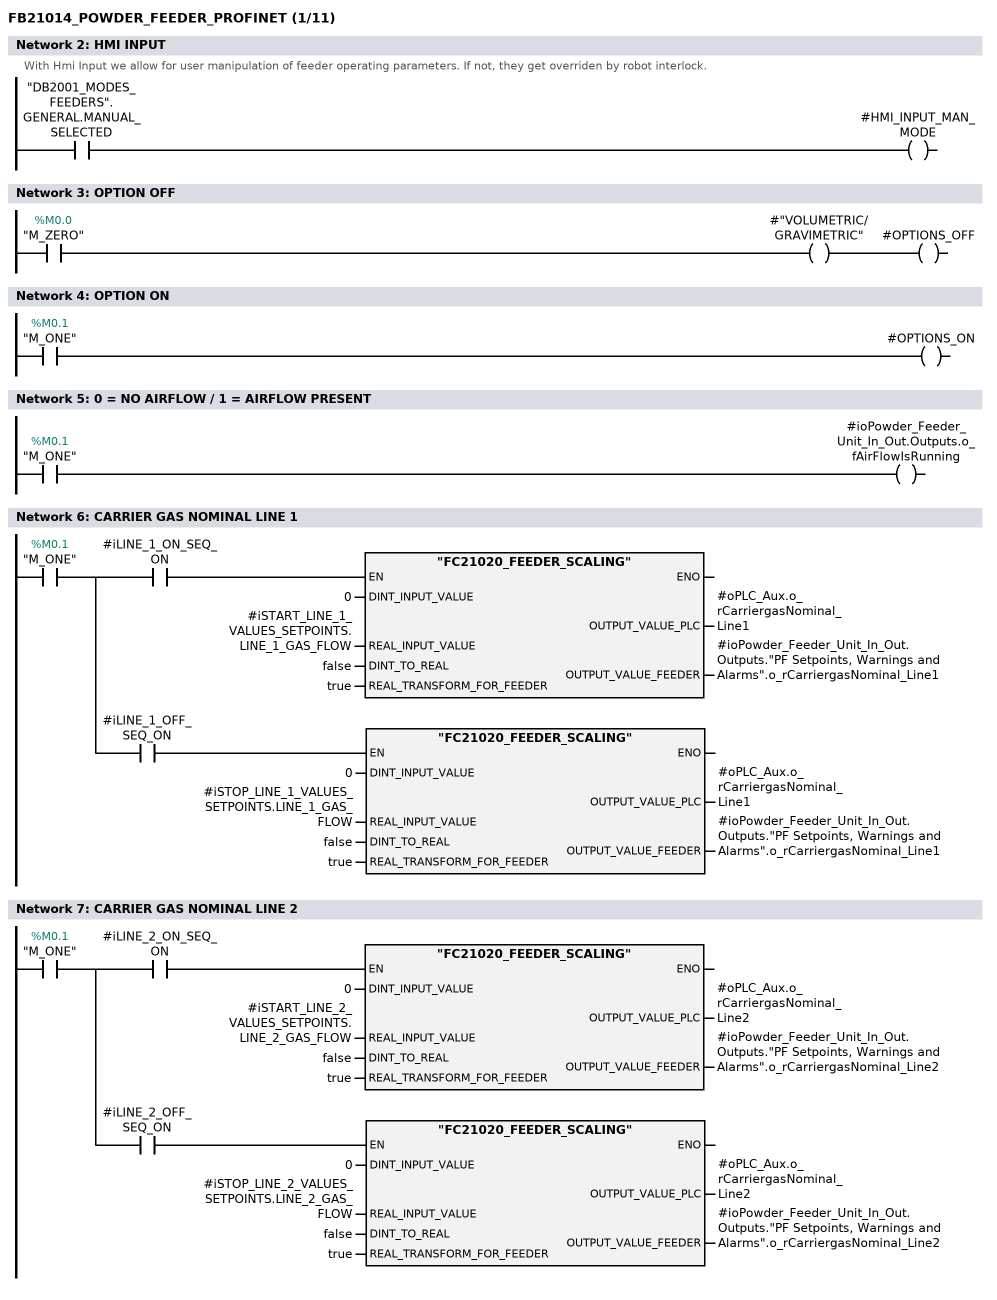
   RUNG wire#powerrail
      Contact( "DB2001_MODES_FEEDERS".GENERAL.MANUAL_SELECTED )
      Coil( #HMI_INPUT_MAN_MODE )
   END_RUNG
   // the same network as SCL:
   #HMI_INPUT_MAN_MODE := "DB2001_MODES_FEEDERS".GENERAL.MANUAL_SELECTED;
END_REGION

REGION Network 3: OPTION OFF
   RUNG wire#powerrail
      Contact( "M_ZERO" )
      Coil( #"VOLUMETRIC/GRAVIMETRIC" )
      Coil( #OPTIONS_OFF )
   END_RUNG
   // the same network as SCL:
   #"VOLUMETRIC/GRAVIMETRIC" := "M_ZERO";
   #OPTIONS_OFF := "M_ZERO";
END_REGION

REGION Network 4: OPTION ON
   RUNG wire#powerrail
      Contact( "M_ONE" )
      Coil( #OPTIONS_ON )
   END_RUNG
   // the same network as SCL:
   #OPTIONS_ON := "M_ONE";
END_REGION

REGION Network 5: 0 = NO AIRFLOW / 1 = AIRFLOW PRESENT
   RUNG wire#powerrail
      Contact( "M_ONE" )
      Coil( #ioPowder_Feeder_Unit_In_Out.Outputs.o_fAirFlowIsRunning )
   END_RUNG
   // the same network as SCL:
   #ioPowder_Feeder_Unit_In_Out.Outputs.o_fAirFlowIsRunning := "M_ONE";
END_REGION

REGION Network 6: CARRIER GAS NOMINAL LINE 1
   RUNG wire#powerrail
      Contact( "M_ONE" )
      wire#w1
      Contact( #iLINE_1_ON_SEQ_ON )
      "FC21020_FEEDER_SCALING"(DINT_INPUT_VALUE := 0, REAL_INPUT_VALUE := #iSTART_LINE_1_VALUES_SETPOINTS.LINE_1_GAS_FLOW, DINT_TO_REAL := false, REAL_TRANSFORM_FOR_FEEDER := true, OUTPUT_VALUE_PLC => #oPLC_Aux.o_rCarriergasNominal_Line1, OUTPUT_VALUE_FEEDER => #ioPowder_Feeder_Unit_In_Out.Outputs."PF Setpoints, Warnings and Alarms".o_rCarriergasNominal_Line1)
   END_RUNG
   RUNG wire#w1
      Contact( #iLINE_1_OFF_SEQ_ON )
      "FC21020_FEEDER_SCALING"(DINT_INPUT_VALUE := 0, REAL_INPUT_VALUE := #iSTOP_LINE_1_VALUES_SETPOINTS.LINE_1_GAS_FLOW, DINT_TO_REAL := false, REAL_TRANSFORM_FOR_FEEDER := true, OUTPUT_VALUE_PLC => #oPLC_Aux.o_rCarriergasNominal_Line1, OUTPUT_VALUE_FEEDER => #ioPowder_Feeder_Unit_In_Out.Outputs."PF Setpoints, Warnings and Alarms".o_rCarriergasNominal_Line1)
   END_RUNG
   // the same network as SCL:
   #_w1 := "M_ONE";
   IF "M_ONE" AND #iLINE_1_ON_SEQ_ON THEN
       "FC21020_FEEDER_SCALING"(DINT_INPUT_VALUE := 0,
                               REAL_INPUT_VALUE := #iSTART_LINE_1_VALUES_SETPOINTS.LINE_1_GAS_FLOW,
                               DINT_TO_REAL := false,
                               REAL_TRANSFORM_FOR_FEEDER := true,
                               OUTPUT_VALUE_PLC => #oPLC_Aux.o_rCarriergasNominal_Line1,
                               OUTPUT_VALUE_FEEDER => #ioPowder_Feeder_Unit_In_Out.Outputs."PF Setpoints, Warnings and Alarms".o_rCarriergasNominal_Line1);
   END_IF;
   IF #_w1 AND #iLINE_1_OFF_SEQ_ON THEN
       "FC21020_FEEDER_SCALING"(DINT_INPUT_VALUE := 0,
                               REAL_INPUT_VALUE := #iSTOP_LINE_1_VALUES_SETPOINTS.LINE_1_GAS_FLOW,
                               DINT_TO_REAL := false,
                               REAL_TRANSFORM_FOR_FEEDER := true,
                               OUTPUT_VALUE_PLC => #oPLC_Aux.o_rCarriergasNominal_Line1,
                               OUTPUT_VALUE_FEEDER => #ioPowder_Feeder_Unit_In_Out.Outputs."PF Setpoints, Warnings and Alarms".o_rCarriergasNominal_Line1);
   END_IF;
END_REGION

REGION Network 7: CARRIER GAS NOMINAL LINE 2
   RUNG wire#powerrail
      Contact( "M_ONE" )
      wire#w1
      Contact( #iLINE_2_ON_SEQ_ON )
      "FC21020_FEEDER_SCALING"(DINT_INPUT_VALUE := 0, REAL_INPUT_VALUE := #iSTART_LINE_2_VALUES_SETPOINTS.LINE_2_GAS_FLOW, DINT_TO_REAL := false, REAL_TRANSFORM_FOR_FEEDER := true, OUTPUT_VALUE_PLC => #oPLC_Aux.o_rCarriergasNominal_Line2, OUTPUT_VALUE_FEEDER => #ioPowder_Feeder_Unit_In_Out.Outputs."PF Setpoints, Warnings and Alarms".o_rCarriergasNominal_Line2)
   END_RUNG
   RUNG wire#w1
      Contact( #iLINE_2_OFF_SEQ_ON )
      "FC21020_FEEDER_SCALING"(DINT_INPUT_VALUE := 0, REAL_INPUT_VALUE := #iSTOP_LINE_2_VALUES_SETPOINTS.LINE_2_GAS_FLOW, DINT_TO_REAL := false, REAL_TRANSFORM_FOR_FEEDER := true, OUTPUT_VALUE_PLC => #oPLC_Aux.o_rCarriergasNominal_Line2, OUTPUT_VALUE_FEEDER => #ioPowder_Feeder_Unit_In_Out.Outputs."PF Setpoints, Warnings and Alarms".o_rCarriergasNominal_Line2)
   END_RUNG
   // the same network as SCL:
   #_w1 := "M_ONE";
   IF "M_ONE" AND #iLINE_2_ON_SEQ_ON THEN
       "FC21020_FEEDER_SCALING"(DINT_INPUT_VALUE := 0,
                               REAL_INPUT_VALUE := #iSTART_LINE_2_VALUES_SETPOINTS.LINE_2_GAS_FLOW,
                               DINT_TO_REAL := false,
                               REAL_TRANSFORM_FOR_FEEDER := true,
                               OUTPUT_VALUE_PLC => #oPLC_Aux.o_rCarriergasNominal_Line2,
                               OUTPUT_VALUE_FEEDER => #ioPowder_Feeder_Unit_In_Out.Outputs."PF Setpoints, Warnings and Alarms".o_rCarriergasNominal_Line2);
   END_IF;
   IF #_w1 AND #iLINE_2_OFF_SEQ_ON THEN
       "FC21020_FEEDER_SCALING"(DINT_INPUT_VALUE := 0,
                               REAL_INPUT_VALUE := #iSTOP_LINE_2_VALUES_SETPOINTS.LINE_2_GAS_FLOW,
                               DINT_TO_REAL := false,
                               REAL_TRANSFORM_FOR_FEEDER := true,
                               OUTPUT_VALUE_PLC => #oPLC_Aux.o_rCarriergasNominal_Line2,
                               OUTPUT_VALUE_FEEDER => #ioPowder_Feeder_Unit_In_Out.Outputs."PF Setpoints, Warnings and Alarms".o_rCarriergasNominal_Line2);
   END_IF;
END_REGION

REGION Network 8: DISK SPEED NOMINAL LINE 1
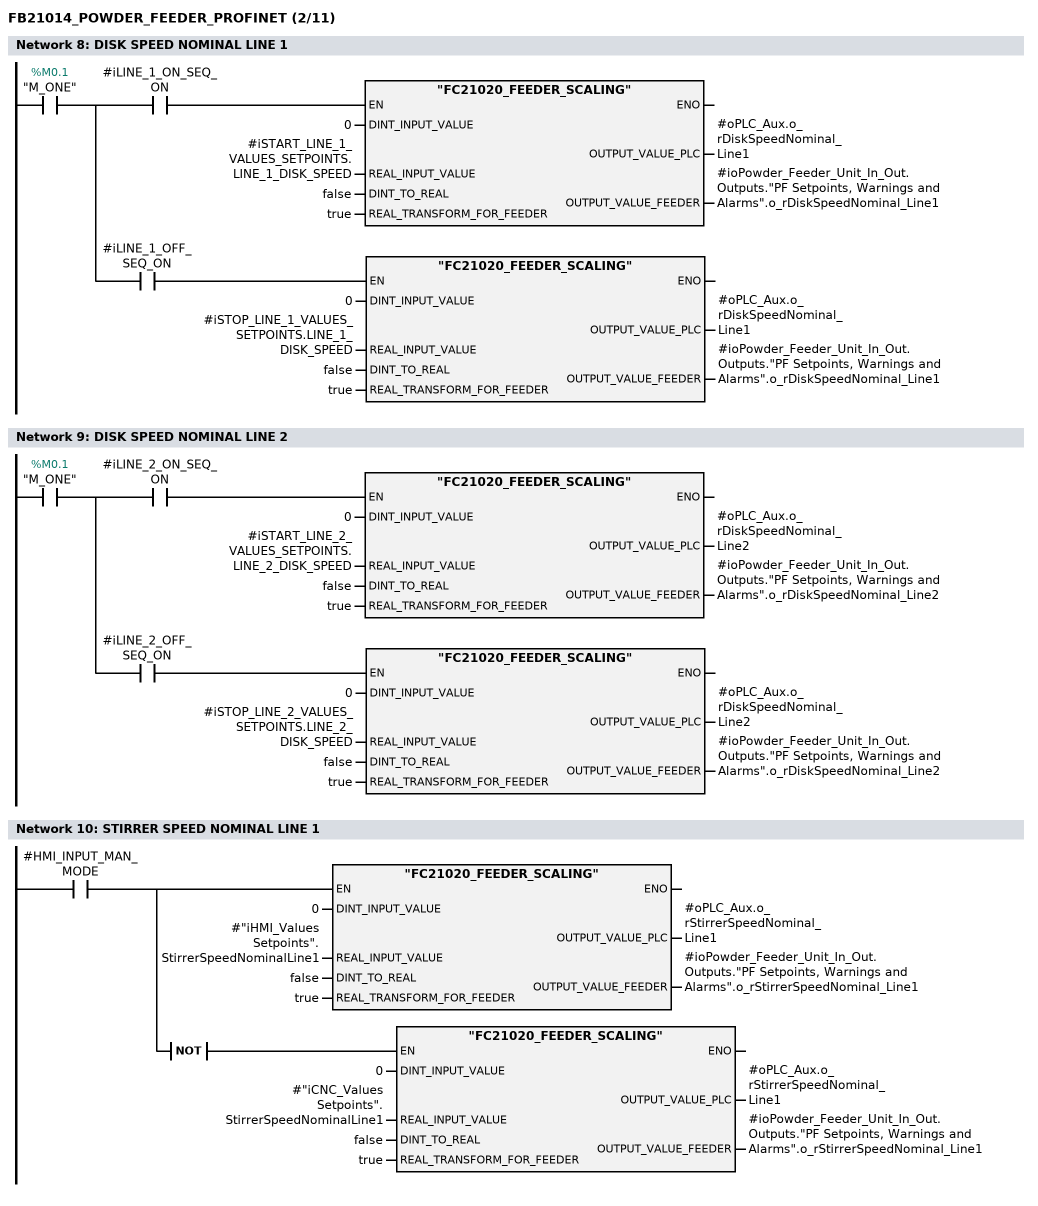
   RUNG wire#powerrail
      Contact( "M_ONE" )
      wire#w1
      Contact( #iLINE_1_ON_SEQ_ON )
      "FC21020_FEEDER_SCALING"(DINT_INPUT_VALUE := 0, REAL_INPUT_VALUE := #iSTART_LINE_1_VALUES_SETPOINTS.LINE_1_DISK_SPEED, DINT_TO_REAL := false, REAL_TRANSFORM_FOR_FEEDER := true, OUTPUT_VALUE_PLC => #oPLC_Aux.o_rDiskSpeedNominal_Line1, OUTPUT_VALUE_FEEDER => #ioPowder_Feeder_Unit_In_Out.Outputs."PF Setpoints, Warnings and Alarms".o_rDiskSpeedNominal_Line1)
   END_RUNG
   RUNG wire#w1
      Contact( #iLINE_1_OFF_SEQ_ON )
      "FC21020_FEEDER_SCALING"(DINT_INPUT_VALUE := 0, REAL_INPUT_VALUE := #iSTOP_LINE_1_VALUES_SETPOINTS.LINE_1_DISK_SPEED, DINT_TO_REAL := false, REAL_TRANSFORM_FOR_FEEDER := true, OUTPUT_VALUE_PLC => #oPLC_Aux.o_rDiskSpeedNominal_Line1, OUTPUT_VALUE_FEEDER => #ioPowder_Feeder_Unit_In_Out.Outputs."PF Setpoints, Warnings and Alarms".o_rDiskSpeedNominal_Line1)
   END_RUNG
   // the same network as SCL:
   #_w1 := "M_ONE";
   IF "M_ONE" AND #iLINE_1_ON_SEQ_ON THEN
       "FC21020_FEEDER_SCALING"(DINT_INPUT_VALUE := 0,
                               REAL_INPUT_VALUE := #iSTART_LINE_1_VALUES_SETPOINTS.LINE_1_DISK_SPEED,
                               DINT_TO_REAL := false,
                               REAL_TRANSFORM_FOR_FEEDER := true,
                               OUTPUT_VALUE_PLC => #oPLC_Aux.o_rDiskSpeedNominal_Line1,
                               OUTPUT_VALUE_FEEDER => #ioPowder_Feeder_Unit_In_Out.Outputs."PF Setpoints, Warnings and Alarms".o_rDiskSpeedNominal_Line1);
   END_IF;
   IF #_w1 AND #iLINE_1_OFF_SEQ_ON THEN
       "FC21020_FEEDER_SCALING"(DINT_INPUT_VALUE := 0,
                               REAL_INPUT_VALUE := #iSTOP_LINE_1_VALUES_SETPOINTS.LINE_1_DISK_SPEED,
                               DINT_TO_REAL := false,
                               REAL_TRANSFORM_FOR_FEEDER := true,
                               OUTPUT_VALUE_PLC => #oPLC_Aux.o_rDiskSpeedNominal_Line1,
                               OUTPUT_VALUE_FEEDER => #ioPowder_Feeder_Unit_In_Out.Outputs."PF Setpoints, Warnings and Alarms".o_rDiskSpeedNominal_Line1);
   END_IF;
END_REGION

REGION Network 9: DISK SPEED NOMINAL LINE 2
   RUNG wire#powerrail
      Contact( "M_ONE" )
      wire#w1
      Contact( #iLINE_2_ON_SEQ_ON )
      "FC21020_FEEDER_SCALING"(DINT_INPUT_VALUE := 0, REAL_INPUT_VALUE := #iSTART_LINE_2_VALUES_SETPOINTS.LINE_2_DISK_SPEED, DINT_TO_REAL := false, REAL_TRANSFORM_FOR_FEEDER := true, OUTPUT_VALUE_PLC => #oPLC_Aux.o_rDiskSpeedNominal_Line2, OUTPUT_VALUE_FEEDER => #ioPowder_Feeder_Unit_In_Out.Outputs."PF Setpoints, Warnings and Alarms".o_rDiskSpeedNominal_Line2)
   END_RUNG
   RUNG wire#w1
      Contact( #iLINE_2_OFF_SEQ_ON )
      "FC21020_FEEDER_SCALING"(DINT_INPUT_VALUE := 0, REAL_INPUT_VALUE := #iSTOP_LINE_2_VALUES_SETPOINTS.LINE_2_DISK_SPEED, DINT_TO_REAL := false, REAL_TRANSFORM_FOR_FEEDER := true, OUTPUT_VALUE_PLC => #oPLC_Aux.o_rDiskSpeedNominal_Line2, OUTPUT_VALUE_FEEDER => #ioPowder_Feeder_Unit_In_Out.Outputs."PF Setpoints, Warnings and Alarms".o_rDiskSpeedNominal_Line2)
   END_RUNG
   // the same network as SCL:
   #_w1 := "M_ONE";
   IF "M_ONE" AND #iLINE_2_ON_SEQ_ON THEN
       "FC21020_FEEDER_SCALING"(DINT_INPUT_VALUE := 0,
                               REAL_INPUT_VALUE := #iSTART_LINE_2_VALUES_SETPOINTS.LINE_2_DISK_SPEED,
                               DINT_TO_REAL := false,
                               REAL_TRANSFORM_FOR_FEEDER := true,
                               OUTPUT_VALUE_PLC => #oPLC_Aux.o_rDiskSpeedNominal_Line2,
                               OUTPUT_VALUE_FEEDER => #ioPowder_Feeder_Unit_In_Out.Outputs."PF Setpoints, Warnings and Alarms".o_rDiskSpeedNominal_Line2);
   END_IF;
   IF #_w1 AND #iLINE_2_OFF_SEQ_ON THEN
       "FC21020_FEEDER_SCALING"(DINT_INPUT_VALUE := 0,
                               REAL_INPUT_VALUE := #iSTOP_LINE_2_VALUES_SETPOINTS.LINE_2_DISK_SPEED,
                               DINT_TO_REAL := false,
                               REAL_TRANSFORM_FOR_FEEDER := true,
                               OUTPUT_VALUE_PLC => #oPLC_Aux.o_rDiskSpeedNominal_Line2,
                               OUTPUT_VALUE_FEEDER => #ioPowder_Feeder_Unit_In_Out.Outputs."PF Setpoints, Warnings and Alarms".o_rDiskSpeedNominal_Line2);
   END_IF;
END_REGION

REGION Network 10: STIRRER SPEED NOMINAL LINE 1
   RUNG wire#powerrail
      Contact( #HMI_INPUT_MAN_MODE )
      wire#w1
      "FC21020_FEEDER_SCALING"(DINT_INPUT_VALUE := 0, REAL_INPUT_VALUE := #"iHMI_Values Setpoints".StirrerSpeedNominalLine1, DINT_TO_REAL := false, REAL_TRANSFORM_FOR_FEEDER := true, OUTPUT_VALUE_PLC => #oPLC_Aux.o_rStirrerSpeedNominal_Line1, OUTPUT_VALUE_FEEDER => #ioPowder_Feeder_Unit_In_Out.Outputs."PF Setpoints, Warnings and Alarms".o_rStirrerSpeedNominal_Line1)
   END_RUNG
   RUNG wire#w1
      Not()
      "FC21020_FEEDER_SCALING"(DINT_INPUT_VALUE := 0, REAL_INPUT_VALUE := #"iCNC_Values Setpoints".StirrerSpeedNominalLine1, DINT_TO_REAL := false, REAL_TRANSFORM_FOR_FEEDER := true, OUTPUT_VALUE_PLC => #oPLC_Aux.o_rStirrerSpeedNominal_Line1, OUTPUT_VALUE_FEEDER => #ioPowder_Feeder_Unit_In_Out.Outputs."PF Setpoints, Warnings and Alarms".o_rStirrerSpeedNominal_Line1)
   END_RUNG
   // the same network as SCL:
   IF #HMI_INPUT_MAN_MODE THEN
       "FC21020_FEEDER_SCALING"(DINT_INPUT_VALUE := 0,
                               REAL_INPUT_VALUE := #"iHMI_Values Setpoints".StirrerSpeedNominalLine1,
                               DINT_TO_REAL := false,
                               REAL_TRANSFORM_FOR_FEEDER := true,
                               OUTPUT_VALUE_PLC => #oPLC_Aux.o_rStirrerSpeedNominal_Line1,
                               OUTPUT_VALUE_FEEDER => #ioPowder_Feeder_Unit_In_Out.Outputs."PF Setpoints, Warnings and Alarms".o_rStirrerSpeedNominal_Line1);
   END_IF;
   IF NOT #HMI_INPUT_MAN_MODE THEN
       "FC21020_FEEDER_SCALING"(DINT_INPUT_VALUE := 0,
                               REAL_INPUT_VALUE := #"iCNC_Values Setpoints".StirrerSpeedNominalLine1,
                               DINT_TO_REAL := false,
                               REAL_TRANSFORM_FOR_FEEDER := true,
                               OUTPUT_VALUE_PLC => #oPLC_Aux.o_rStirrerSpeedNominal_Line1,
                               OUTPUT_VALUE_FEEDER => #ioPowder_Feeder_Unit_In_Out.Outputs."PF Setpoints, Warnings and Alarms".o_rStirrerSpeedNominal_Line1);
   END_IF;
END_REGION

REGION Network 11: STIRRER SPEED NOMINAL LINE 2
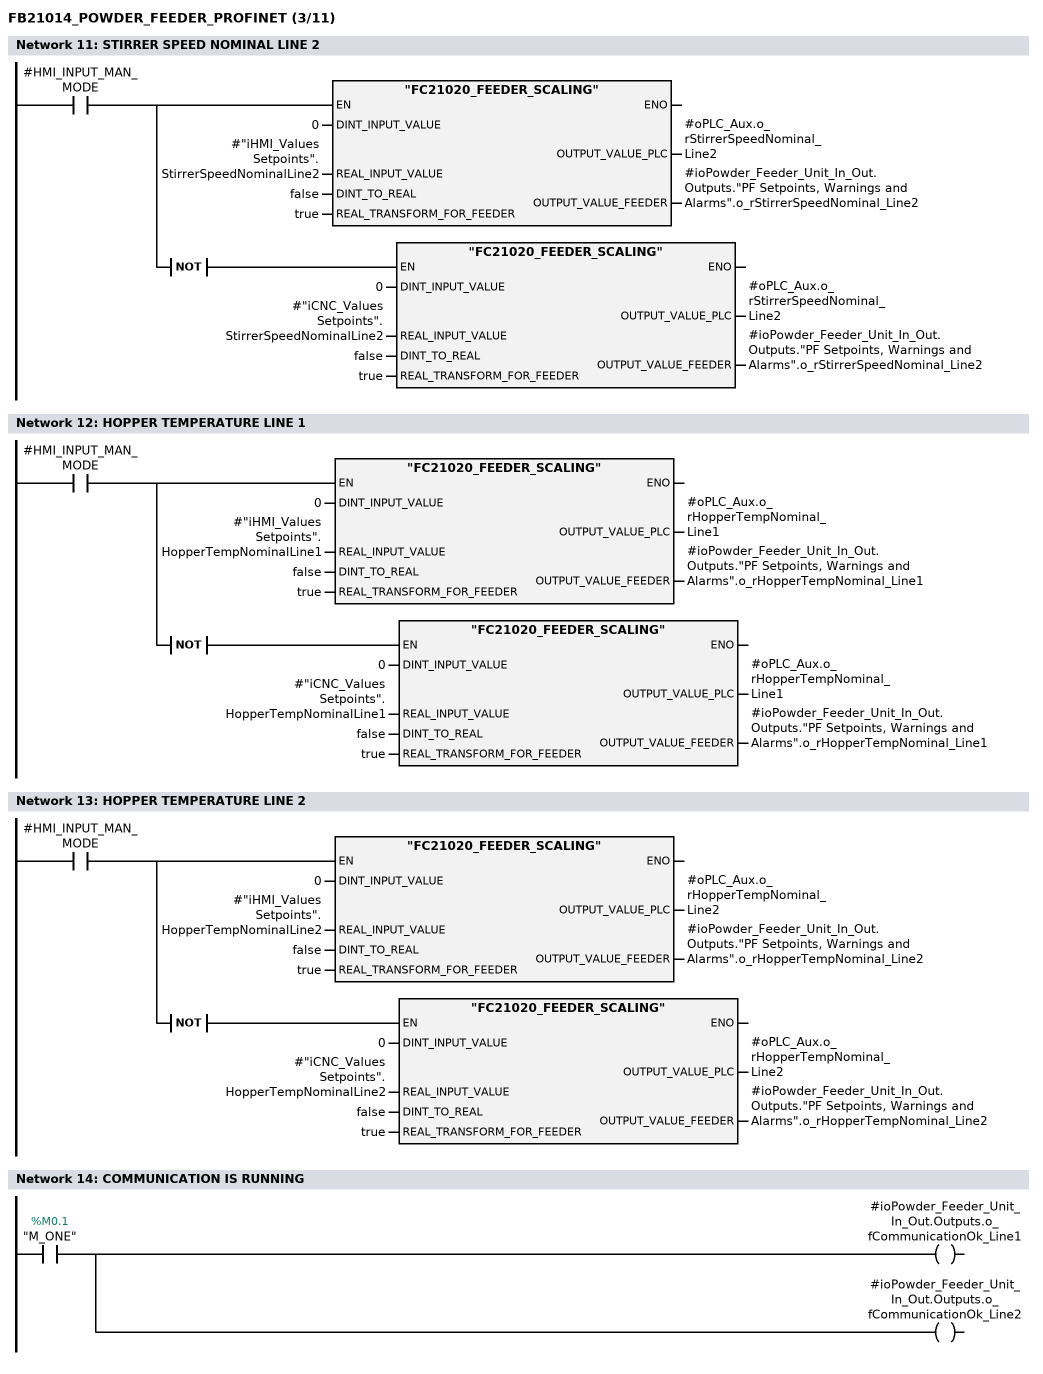
   RUNG wire#powerrail
      Contact( #HMI_INPUT_MAN_MODE )
      wire#w1
      "FC21020_FEEDER_SCALING"(DINT_INPUT_VALUE := 0, REAL_INPUT_VALUE := #"iHMI_Values Setpoints".StirrerSpeedNominalLine2, DINT_TO_REAL := false, REAL_TRANSFORM_FOR_FEEDER := true, OUTPUT_VALUE_PLC => #oPLC_Aux.o_rStirrerSpeedNominal_Line2, OUTPUT_VALUE_FEEDER => #ioPowder_Feeder_Unit_In_Out.Outputs."PF Setpoints, Warnings and Alarms".o_rStirrerSpeedNominal_Line2)
   END_RUNG
   RUNG wire#w1
      Not()
      "FC21020_FEEDER_SCALING"(DINT_INPUT_VALUE := 0, REAL_INPUT_VALUE := #"iCNC_Values Setpoints".StirrerSpeedNominalLine2, DINT_TO_REAL := false, REAL_TRANSFORM_FOR_FEEDER := true, OUTPUT_VALUE_PLC => #oPLC_Aux.o_rStirrerSpeedNominal_Line2, OUTPUT_VALUE_FEEDER => #ioPowder_Feeder_Unit_In_Out.Outputs."PF Setpoints, Warnings and Alarms".o_rStirrerSpeedNominal_Line2)
   END_RUNG
   // the same network as SCL:
   IF #HMI_INPUT_MAN_MODE THEN
       "FC21020_FEEDER_SCALING"(DINT_INPUT_VALUE := 0,
                               REAL_INPUT_VALUE := #"iHMI_Values Setpoints".StirrerSpeedNominalLine2,
                               DINT_TO_REAL := false,
                               REAL_TRANSFORM_FOR_FEEDER := true,
                               OUTPUT_VALUE_PLC => #oPLC_Aux.o_rStirrerSpeedNominal_Line2,
                               OUTPUT_VALUE_FEEDER => #ioPowder_Feeder_Unit_In_Out.Outputs."PF Setpoints, Warnings and Alarms".o_rStirrerSpeedNominal_Line2);
   END_IF;
   IF NOT #HMI_INPUT_MAN_MODE THEN
       "FC21020_FEEDER_SCALING"(DINT_INPUT_VALUE := 0,
                               REAL_INPUT_VALUE := #"iCNC_Values Setpoints".StirrerSpeedNominalLine2,
                               DINT_TO_REAL := false,
                               REAL_TRANSFORM_FOR_FEEDER := true,
                               OUTPUT_VALUE_PLC => #oPLC_Aux.o_rStirrerSpeedNominal_Line2,
                               OUTPUT_VALUE_FEEDER => #ioPowder_Feeder_Unit_In_Out.Outputs."PF Setpoints, Warnings and Alarms".o_rStirrerSpeedNominal_Line2);
   END_IF;
END_REGION

REGION Network 12: HOPPER TEMPERATURE LINE 1
   RUNG wire#powerrail
      Contact( #HMI_INPUT_MAN_MODE )
      wire#w1
      "FC21020_FEEDER_SCALING"(DINT_INPUT_VALUE := 0, REAL_INPUT_VALUE := #"iHMI_Values Setpoints".HopperTempNominalLine1, DINT_TO_REAL := false, REAL_TRANSFORM_FOR_FEEDER := true, OUTPUT_VALUE_PLC => #oPLC_Aux.o_rHopperTempNominal_Line1, OUTPUT_VALUE_FEEDER => #ioPowder_Feeder_Unit_In_Out.Outputs."PF Setpoints, Warnings and Alarms".o_rHopperTempNominal_Line1)
   END_RUNG
   RUNG wire#w1
      Not()
      "FC21020_FEEDER_SCALING"(DINT_INPUT_VALUE := 0, REAL_INPUT_VALUE := #"iCNC_Values Setpoints".HopperTempNominalLine1, DINT_TO_REAL := false, REAL_TRANSFORM_FOR_FEEDER := true, OUTPUT_VALUE_PLC => #oPLC_Aux.o_rHopperTempNominal_Line1, OUTPUT_VALUE_FEEDER => #ioPowder_Feeder_Unit_In_Out.Outputs."PF Setpoints, Warnings and Alarms".o_rHopperTempNominal_Line1)
   END_RUNG
   // the same network as SCL:
   IF #HMI_INPUT_MAN_MODE THEN
       "FC21020_FEEDER_SCALING"(DINT_INPUT_VALUE := 0,
                               REAL_INPUT_VALUE := #"iHMI_Values Setpoints".HopperTempNominalLine1,
                               DINT_TO_REAL := false,
                               REAL_TRANSFORM_FOR_FEEDER := true,
                               OUTPUT_VALUE_PLC => #oPLC_Aux.o_rHopperTempNominal_Line1,
                               OUTPUT_VALUE_FEEDER => #ioPowder_Feeder_Unit_In_Out.Outputs."PF Setpoints, Warnings and Alarms".o_rHopperTempNominal_Line1);
   END_IF;
   IF NOT #HMI_INPUT_MAN_MODE THEN
       "FC21020_FEEDER_SCALING"(DINT_INPUT_VALUE := 0,
                               REAL_INPUT_VALUE := #"iCNC_Values Setpoints".HopperTempNominalLine1,
                               DINT_TO_REAL := false,
                               REAL_TRANSFORM_FOR_FEEDER := true,
                               OUTPUT_VALUE_PLC => #oPLC_Aux.o_rHopperTempNominal_Line1,
                               OUTPUT_VALUE_FEEDER => #ioPowder_Feeder_Unit_In_Out.Outputs."PF Setpoints, Warnings and Alarms".o_rHopperTempNominal_Line1);
   END_IF;
END_REGION

REGION Network 13: HOPPER TEMPERATURE LINE 2
   RUNG wire#powerrail
      Contact( #HMI_INPUT_MAN_MODE )
      wire#w1
      "FC21020_FEEDER_SCALING"(DINT_INPUT_VALUE := 0, REAL_INPUT_VALUE := #"iHMI_Values Setpoints".HopperTempNominalLine2, DINT_TO_REAL := false, REAL_TRANSFORM_FOR_FEEDER := true, OUTPUT_VALUE_PLC => #oPLC_Aux.o_rHopperTempNominal_Line2, OUTPUT_VALUE_FEEDER => #ioPowder_Feeder_Unit_In_Out.Outputs."PF Setpoints, Warnings and Alarms".o_rHopperTempNominal_Line2)
   END_RUNG
   RUNG wire#w1
      Not()
      "FC21020_FEEDER_SCALING"(DINT_INPUT_VALUE := 0, REAL_INPUT_VALUE := #"iCNC_Values Setpoints".HopperTempNominalLine2, DINT_TO_REAL := false, REAL_TRANSFORM_FOR_FEEDER := true, OUTPUT_VALUE_PLC => #oPLC_Aux.o_rHopperTempNominal_Line2, OUTPUT_VALUE_FEEDER => #ioPowder_Feeder_Unit_In_Out.Outputs."PF Setpoints, Warnings and Alarms".o_rHopperTempNominal_Line2)
   END_RUNG
   // the same network as SCL:
   IF #HMI_INPUT_MAN_MODE THEN
       "FC21020_FEEDER_SCALING"(DINT_INPUT_VALUE := 0,
                               REAL_INPUT_VALUE := #"iHMI_Values Setpoints".HopperTempNominalLine2,
                               DINT_TO_REAL := false,
                               REAL_TRANSFORM_FOR_FEEDER := true,
                               OUTPUT_VALUE_PLC => #oPLC_Aux.o_rHopperTempNominal_Line2,
                               OUTPUT_VALUE_FEEDER => #ioPowder_Feeder_Unit_In_Out.Outputs."PF Setpoints, Warnings and Alarms".o_rHopperTempNominal_Line2);
   END_IF;
   IF NOT #HMI_INPUT_MAN_MODE THEN
       "FC21020_FEEDER_SCALING"(DINT_INPUT_VALUE := 0,
                               REAL_INPUT_VALUE := #"iCNC_Values Setpoints".HopperTempNominalLine2,
                               DINT_TO_REAL := false,
                               REAL_TRANSFORM_FOR_FEEDER := true,
                               OUTPUT_VALUE_PLC => #oPLC_Aux.o_rHopperTempNominal_Line2,
                               OUTPUT_VALUE_FEEDER => #ioPowder_Feeder_Unit_In_Out.Outputs."PF Setpoints, Warnings and Alarms".o_rHopperTempNominal_Line2);
   END_IF;
END_REGION

REGION Network 14: COMMUNICATION IS RUNNING
   RUNG wire#powerrail
      Contact( "M_ONE" )
      wire#w1
      Coil( #ioPowder_Feeder_Unit_In_Out.Outputs.o_fCommunicationOk_Line1 )
   END_RUNG
   RUNG wire#w1
      Coil( #ioPowder_Feeder_Unit_In_Out.Outputs.o_fCommunicationOk_Line2 )
   END_RUNG
   // the same network as SCL:
   #ioPowder_Feeder_Unit_In_Out.Outputs.o_fCommunicationOk_Line1 := "M_ONE";
   #ioPowder_Feeder_Unit_In_Out.Outputs.o_fCommunicationOk_Line2 := "M_ONE";
END_REGION

REGION Network 15: VOLUMETRIC MODE ON
   // Volumetric Mode On = 1 for Twin 150
   // Gravimetric Mode - n/a for Twin 150
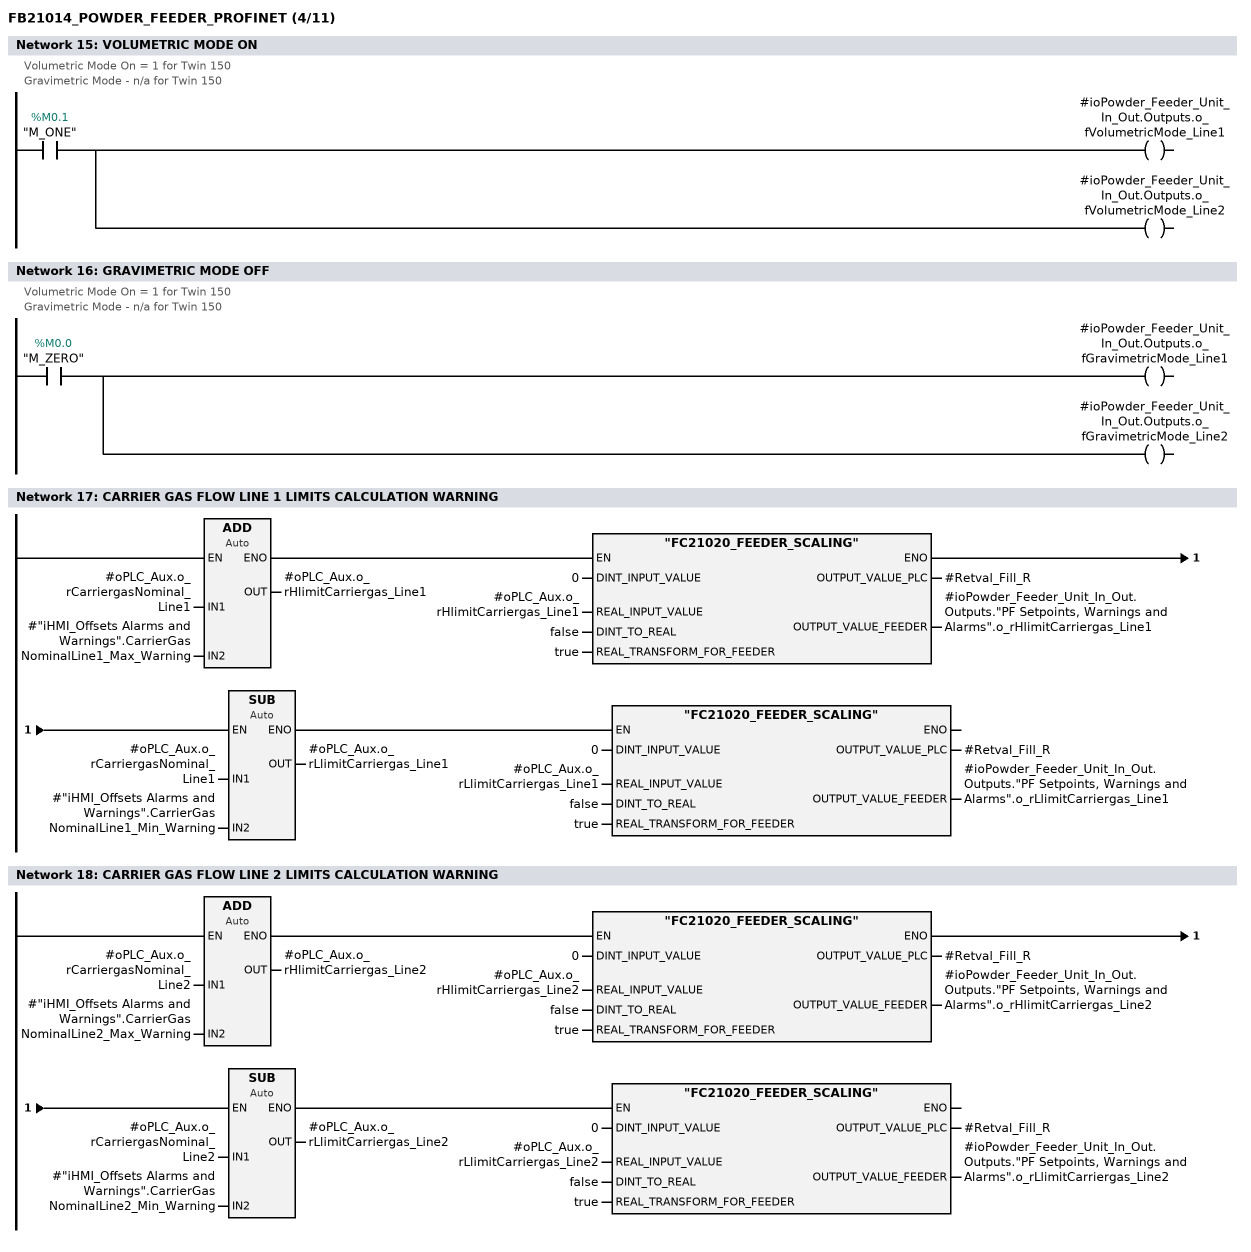
   RUNG wire#powerrail
      Contact( "M_ONE" )
      wire#w1
      Coil( #ioPowder_Feeder_Unit_In_Out.Outputs.o_fVolumetricMode_Line1 )
   END_RUNG
   RUNG wire#w1
      Coil( #ioPowder_Feeder_Unit_In_Out.Outputs.o_fVolumetricMode_Line2 )
   END_RUNG
   // the same network as SCL:
   #ioPowder_Feeder_Unit_In_Out.Outputs.o_fVolumetricMode_Line1 := "M_ONE";
   #ioPowder_Feeder_Unit_In_Out.Outputs.o_fVolumetricMode_Line2 := "M_ONE";
END_REGION

REGION Network 16: GRAVIMETRIC MODE OFF
   // Volumetric Mode On = 1 for Twin 150
   // Gravimetric Mode - n/a for Twin 150
   RUNG wire#powerrail
      Contact( "M_ZERO" )
      wire#w1
      Coil( #ioPowder_Feeder_Unit_In_Out.Outputs.o_fGravimetricMode_Line1 )
   END_RUNG
   RUNG wire#w1
      Coil( #ioPowder_Feeder_Unit_In_Out.Outputs.o_fGravimetricMode_Line2 )
   END_RUNG
   // the same network as SCL:
   #ioPowder_Feeder_Unit_In_Out.Outputs.o_fGravimetricMode_Line1 := "M_ZERO";
   #ioPowder_Feeder_Unit_In_Out.Outputs.o_fGravimetricMode_Line2 := "M_ZERO";
END_REGION

REGION Network 17: CARRIER GAS FLOW LINE 1 LIMITS CALCULATION WARNING
   RUNG wire#powerrail
      Add(in1 := #oPLC_Aux.o_rCarriergasNominal_Line1, in2 := #"iHMI_Offsets Alarms and Warnings".CarrierGasNominalLine1_Max_Warning, out => #oPLC_Aux.o_rHlimitCarriergas_Line1)
      "FC21020_FEEDER_SCALING"(DINT_INPUT_VALUE := 0, REAL_INPUT_VALUE := #oPLC_Aux.o_rHlimitCarriergas_Line1, DINT_TO_REAL := false, REAL_TRANSFORM_FOR_FEEDER := true, OUTPUT_VALUE_PLC => #Retval_Fill_R, OUTPUT_VALUE_FEEDER => #ioPowder_Feeder_Unit_In_Out.Outputs."PF Setpoints, Warnings and Alarms".o_rHlimitCarriergas_Line1)
      Sub(in1 := #oPLC_Aux.o_rCarriergasNominal_Line1, in2 := #"iHMI_Offsets Alarms and Warnings".CarrierGasNominalLine1_Min_Warning, out => #oPLC_Aux.o_rLlimitCarriergas_Line1)
      "FC21020_FEEDER_SCALING"(DINT_INPUT_VALUE := 0, REAL_INPUT_VALUE := #oPLC_Aux.o_rLlimitCarriergas_Line1, DINT_TO_REAL := false, REAL_TRANSFORM_FOR_FEEDER := true, OUTPUT_VALUE_PLC => #Retval_Fill_R, OUTPUT_VALUE_FEEDER => #ioPowder_Feeder_Unit_In_Out.Outputs."PF Setpoints, Warnings and Alarms".o_rLlimitCarriergas_Line1)
   END_RUNG
   // the same network as SCL:
   #oPLC_Aux.o_rHlimitCarriergas_Line1 := #oPLC_Aux.o_rCarriergasNominal_Line1 + #"iHMI_Offsets Alarms and Warnings".CarrierGasNominalLine1_Max_Warning;
   "FC21020_FEEDER_SCALING"(DINT_INPUT_VALUE := 0,
                           REAL_INPUT_VALUE := #oPLC_Aux.o_rHlimitCarriergas_Line1,
                           DINT_TO_REAL := false,
                           REAL_TRANSFORM_FOR_FEEDER := true,
                           OUTPUT_VALUE_PLC => #Retval_Fill_R,
                           OUTPUT_VALUE_FEEDER => #ioPowder_Feeder_Unit_In_Out.Outputs."PF Setpoints, Warnings and Alarms".o_rHlimitCarriergas_Line1,
                           ENO => #_w1);
   IF #_w1 THEN
       #oPLC_Aux.o_rLlimitCarriergas_Line1 := #oPLC_Aux.o_rCarriergasNominal_Line1 - #"iHMI_Offsets Alarms and Warnings".CarrierGasNominalLine1_Min_Warning;
       "FC21020_FEEDER_SCALING"(DINT_INPUT_VALUE := 0,
                               REAL_INPUT_VALUE := #oPLC_Aux.o_rLlimitCarriergas_Line1,
                               DINT_TO_REAL := false,
                               REAL_TRANSFORM_FOR_FEEDER := true,
                               OUTPUT_VALUE_PLC => #Retval_Fill_R,
                               OUTPUT_VALUE_FEEDER => #ioPowder_Feeder_Unit_In_Out.Outputs."PF Setpoints, Warnings and Alarms".o_rLlimitCarriergas_Line1);
   END_IF;
END_REGION

REGION Network 18: CARRIER GAS FLOW LINE 2 LIMITS CALCULATION WARNING
   RUNG wire#powerrail
      Add(in1 := #oPLC_Aux.o_rCarriergasNominal_Line2, in2 := #"iHMI_Offsets Alarms and Warnings".CarrierGasNominalLine2_Max_Warning, out => #oPLC_Aux.o_rHlimitCarriergas_Line2)
      "FC21020_FEEDER_SCALING"(DINT_INPUT_VALUE := 0, REAL_INPUT_VALUE := #oPLC_Aux.o_rHlimitCarriergas_Line2, DINT_TO_REAL := false, REAL_TRANSFORM_FOR_FEEDER := true, OUTPUT_VALUE_PLC => #Retval_Fill_R, OUTPUT_VALUE_FEEDER => #ioPowder_Feeder_Unit_In_Out.Outputs."PF Setpoints, Warnings and Alarms".o_rHlimitCarriergas_Line2)
      Sub(in1 := #oPLC_Aux.o_rCarriergasNominal_Line2, in2 := #"iHMI_Offsets Alarms and Warnings".CarrierGasNominalLine2_Min_Warning, out => #oPLC_Aux.o_rLlimitCarriergas_Line2)
      "FC21020_FEEDER_SCALING"(DINT_INPUT_VALUE := 0, REAL_INPUT_VALUE := #oPLC_Aux.o_rLlimitCarriergas_Line2, DINT_TO_REAL := false, REAL_TRANSFORM_FOR_FEEDER := true, OUTPUT_VALUE_PLC => #Retval_Fill_R, OUTPUT_VALUE_FEEDER => #ioPowder_Feeder_Unit_In_Out.Outputs."PF Setpoints, Warnings and Alarms".o_rLlimitCarriergas_Line2)
   END_RUNG
   // the same network as SCL:
   #oPLC_Aux.o_rHlimitCarriergas_Line2 := #oPLC_Aux.o_rCarriergasNominal_Line2 + #"iHMI_Offsets Alarms and Warnings".CarrierGasNominalLine2_Max_Warning;
   "FC21020_FEEDER_SCALING"(DINT_INPUT_VALUE := 0,
                           REAL_INPUT_VALUE := #oPLC_Aux.o_rHlimitCarriergas_Line2,
                           DINT_TO_REAL := false,
                           REAL_TRANSFORM_FOR_FEEDER := true,
                           OUTPUT_VALUE_PLC => #Retval_Fill_R,
                           OUTPUT_VALUE_FEEDER => #ioPowder_Feeder_Unit_In_Out.Outputs."PF Setpoints, Warnings and Alarms".o_rHlimitCarriergas_Line2,
                           ENO => #_w1);
   IF #_w1 THEN
       #oPLC_Aux.o_rLlimitCarriergas_Line2 := #oPLC_Aux.o_rCarriergasNominal_Line2 - #"iHMI_Offsets Alarms and Warnings".CarrierGasNominalLine2_Min_Warning;
       "FC21020_FEEDER_SCALING"(DINT_INPUT_VALUE := 0,
                               REAL_INPUT_VALUE := #oPLC_Aux.o_rLlimitCarriergas_Line2,
                               DINT_TO_REAL := false,
                               REAL_TRANSFORM_FOR_FEEDER := true,
                               OUTPUT_VALUE_PLC => #Retval_Fill_R,
                               OUTPUT_VALUE_FEEDER => #ioPowder_Feeder_Unit_In_Out.Outputs."PF Setpoints, Warnings and Alarms".o_rLlimitCarriergas_Line2);
   END_IF;
END_REGION

REGION Network 19: CARRIER GAS FLOW LINE 1 LIMITS CALCULATION ALARM
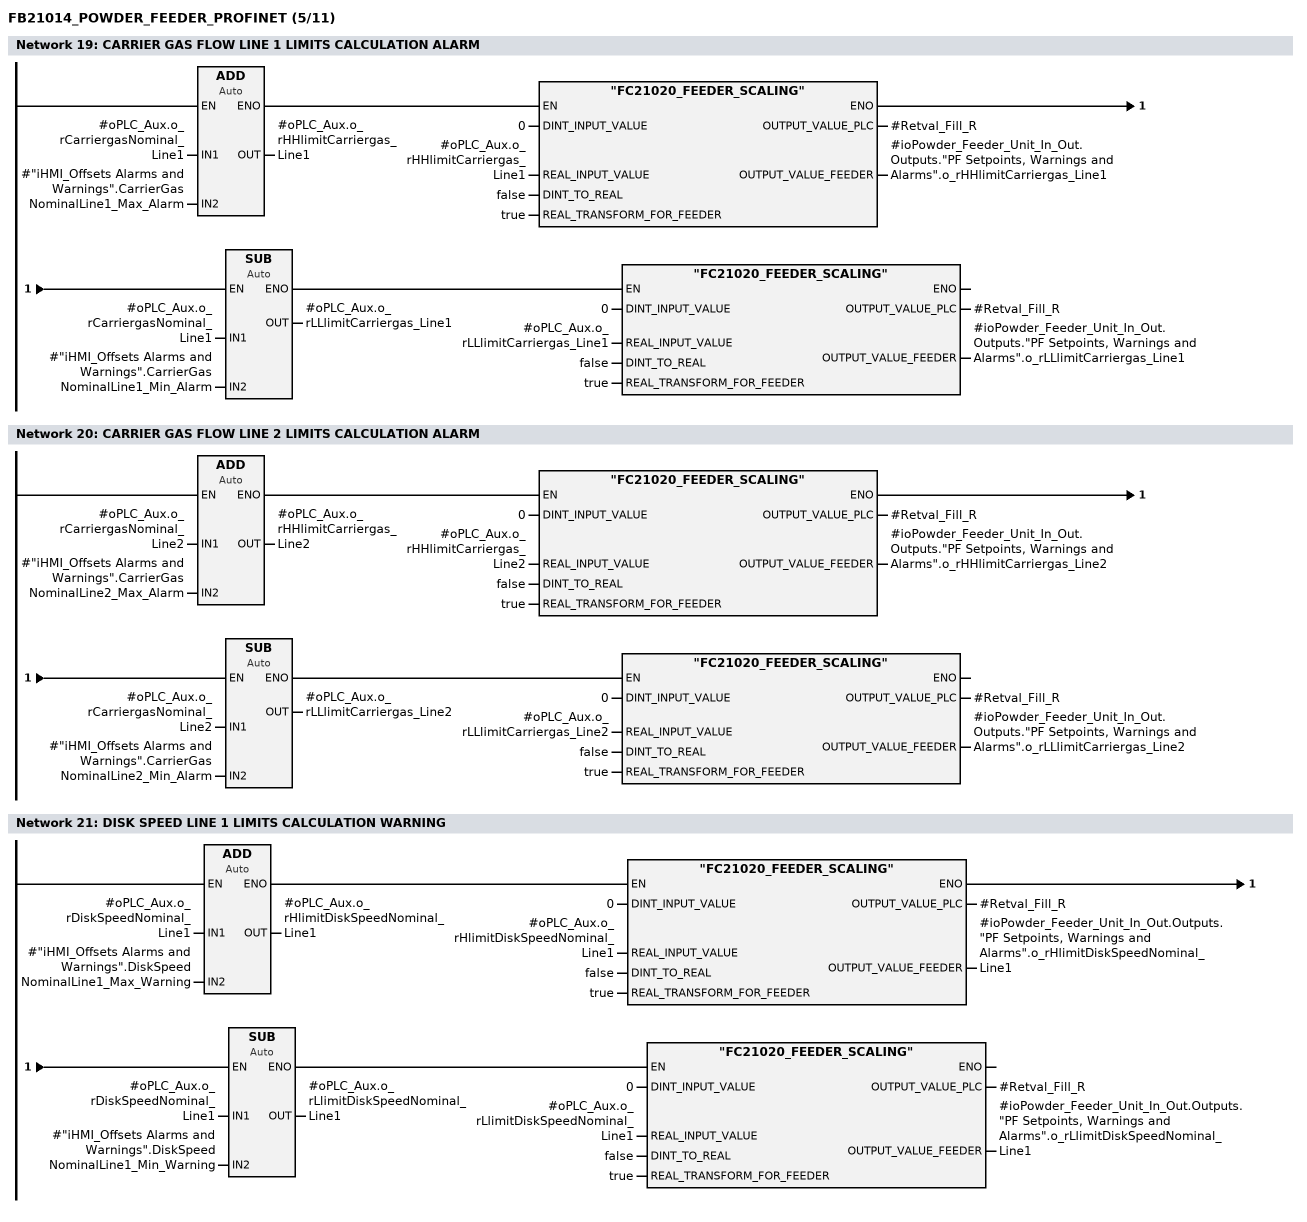
   RUNG wire#powerrail
      Add(in1 := #oPLC_Aux.o_rCarriergasNominal_Line1, in2 := #"iHMI_Offsets Alarms and Warnings".CarrierGasNominalLine1_Max_Alarm, out => #oPLC_Aux.o_rHHlimitCarriergas_Line1)
      "FC21020_FEEDER_SCALING"(DINT_INPUT_VALUE := 0, REAL_INPUT_VALUE := #oPLC_Aux.o_rHHlimitCarriergas_Line1, DINT_TO_REAL := false, REAL_TRANSFORM_FOR_FEEDER := true, OUTPUT_VALUE_PLC => #Retval_Fill_R, OUTPUT_VALUE_FEEDER => #ioPowder_Feeder_Unit_In_Out.Outputs."PF Setpoints, Warnings and Alarms".o_rHHlimitCarriergas_Line1)
      Sub(in1 := #oPLC_Aux.o_rCarriergasNominal_Line1, in2 := #"iHMI_Offsets Alarms and Warnings".CarrierGasNominalLine1_Min_Alarm, out => #oPLC_Aux.o_rLLlimitCarriergas_Line1)
      "FC21020_FEEDER_SCALING"(DINT_INPUT_VALUE := 0, REAL_INPUT_VALUE := #oPLC_Aux.o_rLLlimitCarriergas_Line1, DINT_TO_REAL := false, REAL_TRANSFORM_FOR_FEEDER := true, OUTPUT_VALUE_PLC => #Retval_Fill_R, OUTPUT_VALUE_FEEDER => #ioPowder_Feeder_Unit_In_Out.Outputs."PF Setpoints, Warnings and Alarms".o_rLLlimitCarriergas_Line1)
   END_RUNG
   // the same network as SCL:
   #oPLC_Aux.o_rHHlimitCarriergas_Line1 := #oPLC_Aux.o_rCarriergasNominal_Line1 + #"iHMI_Offsets Alarms and Warnings".CarrierGasNominalLine1_Max_Alarm;
   "FC21020_FEEDER_SCALING"(DINT_INPUT_VALUE := 0,
                           REAL_INPUT_VALUE := #oPLC_Aux.o_rHHlimitCarriergas_Line1,
                           DINT_TO_REAL := false,
                           REAL_TRANSFORM_FOR_FEEDER := true,
                           OUTPUT_VALUE_PLC => #Retval_Fill_R,
                           OUTPUT_VALUE_FEEDER => #ioPowder_Feeder_Unit_In_Out.Outputs."PF Setpoints, Warnings and Alarms".o_rHHlimitCarriergas_Line1,
                           ENO => #_w1);
   IF #_w1 THEN
       #oPLC_Aux.o_rLLlimitCarriergas_Line1 := #oPLC_Aux.o_rCarriergasNominal_Line1 - #"iHMI_Offsets Alarms and Warnings".CarrierGasNominalLine1_Min_Alarm;
       "FC21020_FEEDER_SCALING"(DINT_INPUT_VALUE := 0,
                               REAL_INPUT_VALUE := #oPLC_Aux.o_rLLlimitCarriergas_Line1,
                               DINT_TO_REAL := false,
                               REAL_TRANSFORM_FOR_FEEDER := true,
                               OUTPUT_VALUE_PLC => #Retval_Fill_R,
                               OUTPUT_VALUE_FEEDER => #ioPowder_Feeder_Unit_In_Out.Outputs."PF Setpoints, Warnings and Alarms".o_rLLlimitCarriergas_Line1);
   END_IF;
END_REGION

REGION Network 20: CARRIER GAS FLOW LINE 2 LIMITS CALCULATION ALARM
   RUNG wire#powerrail
      Add(in1 := #oPLC_Aux.o_rCarriergasNominal_Line2, in2 := #"iHMI_Offsets Alarms and Warnings".CarrierGasNominalLine2_Max_Alarm, out => #oPLC_Aux.o_rHHlimitCarriergas_Line2)
      "FC21020_FEEDER_SCALING"(DINT_INPUT_VALUE := 0, REAL_INPUT_VALUE := #oPLC_Aux.o_rHHlimitCarriergas_Line2, DINT_TO_REAL := false, REAL_TRANSFORM_FOR_FEEDER := true, OUTPUT_VALUE_PLC => #Retval_Fill_R, OUTPUT_VALUE_FEEDER => #ioPowder_Feeder_Unit_In_Out.Outputs."PF Setpoints, Warnings and Alarms".o_rHHlimitCarriergas_Line2)
      Sub(in1 := #oPLC_Aux.o_rCarriergasNominal_Line2, in2 := #"iHMI_Offsets Alarms and Warnings".CarrierGasNominalLine2_Min_Alarm, out => #oPLC_Aux.o_rLLlimitCarriergas_Line2)
      "FC21020_FEEDER_SCALING"(DINT_INPUT_VALUE := 0, REAL_INPUT_VALUE := #oPLC_Aux.o_rLLlimitCarriergas_Line2, DINT_TO_REAL := false, REAL_TRANSFORM_FOR_FEEDER := true, OUTPUT_VALUE_PLC => #Retval_Fill_R, OUTPUT_VALUE_FEEDER => #ioPowder_Feeder_Unit_In_Out.Outputs."PF Setpoints, Warnings and Alarms".o_rLLlimitCarriergas_Line2)
   END_RUNG
   // the same network as SCL:
   #oPLC_Aux.o_rHHlimitCarriergas_Line2 := #oPLC_Aux.o_rCarriergasNominal_Line2 + #"iHMI_Offsets Alarms and Warnings".CarrierGasNominalLine2_Max_Alarm;
   "FC21020_FEEDER_SCALING"(DINT_INPUT_VALUE := 0,
                           REAL_INPUT_VALUE := #oPLC_Aux.o_rHHlimitCarriergas_Line2,
                           DINT_TO_REAL := false,
                           REAL_TRANSFORM_FOR_FEEDER := true,
                           OUTPUT_VALUE_PLC => #Retval_Fill_R,
                           OUTPUT_VALUE_FEEDER => #ioPowder_Feeder_Unit_In_Out.Outputs."PF Setpoints, Warnings and Alarms".o_rHHlimitCarriergas_Line2,
                           ENO => #_w1);
   IF #_w1 THEN
       #oPLC_Aux.o_rLLlimitCarriergas_Line2 := #oPLC_Aux.o_rCarriergasNominal_Line2 - #"iHMI_Offsets Alarms and Warnings".CarrierGasNominalLine2_Min_Alarm;
       "FC21020_FEEDER_SCALING"(DINT_INPUT_VALUE := 0,
                               REAL_INPUT_VALUE := #oPLC_Aux.o_rLLlimitCarriergas_Line2,
                               DINT_TO_REAL := false,
                               REAL_TRANSFORM_FOR_FEEDER := true,
                               OUTPUT_VALUE_PLC => #Retval_Fill_R,
                               OUTPUT_VALUE_FEEDER => #ioPowder_Feeder_Unit_In_Out.Outputs."PF Setpoints, Warnings and Alarms".o_rLLlimitCarriergas_Line2);
   END_IF;
END_REGION

REGION Network 21: DISK SPEED LINE 1 LIMITS CALCULATION WARNING
   RUNG wire#powerrail
      Add(in1 := #oPLC_Aux.o_rDiskSpeedNominal_Line1, in2 := #"iHMI_Offsets Alarms and Warnings".DiskSpeedNominalLine1_Max_Warning, out => #oPLC_Aux.o_rHlimitDiskSpeedNominal_Line1)
      "FC21020_FEEDER_SCALING"(DINT_INPUT_VALUE := 0, REAL_INPUT_VALUE := #oPLC_Aux.o_rHlimitDiskSpeedNominal_Line1, DINT_TO_REAL := false, REAL_TRANSFORM_FOR_FEEDER := true, OUTPUT_VALUE_PLC => #Retval_Fill_R, OUTPUT_VALUE_FEEDER => #ioPowder_Feeder_Unit_In_Out.Outputs."PF Setpoints, Warnings and Alarms".o_rHlimitDiskSpeedNominal_Line1)
      Sub(in1 := #oPLC_Aux.o_rDiskSpeedNominal_Line1, in2 := #"iHMI_Offsets Alarms and Warnings".DiskSpeedNominalLine1_Min_Warning, out => #oPLC_Aux.o_rLlimitDiskSpeedNominal_Line1)
      "FC21020_FEEDER_SCALING"(DINT_INPUT_VALUE := 0, REAL_INPUT_VALUE := #oPLC_Aux.o_rLlimitDiskSpeedNominal_Line1, DINT_TO_REAL := false, REAL_TRANSFORM_FOR_FEEDER := true, OUTPUT_VALUE_PLC => #Retval_Fill_R, OUTPUT_VALUE_FEEDER => #ioPowder_Feeder_Unit_In_Out.Outputs."PF Setpoints, Warnings and Alarms".o_rLlimitDiskSpeedNominal_Line1)
   END_RUNG
   // the same network as SCL:
   #oPLC_Aux.o_rHlimitDiskSpeedNominal_Line1 := #oPLC_Aux.o_rDiskSpeedNominal_Line1 + #"iHMI_Offsets Alarms and Warnings".DiskSpeedNominalLine1_Max_Warning;
   "FC21020_FEEDER_SCALING"(DINT_INPUT_VALUE := 0,
                           REAL_INPUT_VALUE := #oPLC_Aux.o_rHlimitDiskSpeedNominal_Line1,
                           DINT_TO_REAL := false,
                           REAL_TRANSFORM_FOR_FEEDER := true,
                           OUTPUT_VALUE_PLC => #Retval_Fill_R,
                           OUTPUT_VALUE_FEEDER => #ioPowder_Feeder_Unit_In_Out.Outputs."PF Setpoints, Warnings and Alarms".o_rHlimitDiskSpeedNominal_Line1,
                           ENO => #_w1);
   IF #_w1 THEN
       #oPLC_Aux.o_rLlimitDiskSpeedNominal_Line1 := #oPLC_Aux.o_rDiskSpeedNominal_Line1 - #"iHMI_Offsets Alarms and Warnings".DiskSpeedNominalLine1_Min_Warning;
       "FC21020_FEEDER_SCALING"(DINT_INPUT_VALUE := 0,
                               REAL_INPUT_VALUE := #oPLC_Aux.o_rLlimitDiskSpeedNominal_Line1,
                               DINT_TO_REAL := false,
                               REAL_TRANSFORM_FOR_FEEDER := true,
                               OUTPUT_VALUE_PLC => #Retval_Fill_R,
                               OUTPUT_VALUE_FEEDER => #ioPowder_Feeder_Unit_In_Out.Outputs."PF Setpoints, Warnings and Alarms".o_rLlimitDiskSpeedNominal_Line1);
   END_IF;
END_REGION

REGION Network 22: DISK SPEED LINE 2 LIMITS CALCULATION WARNING
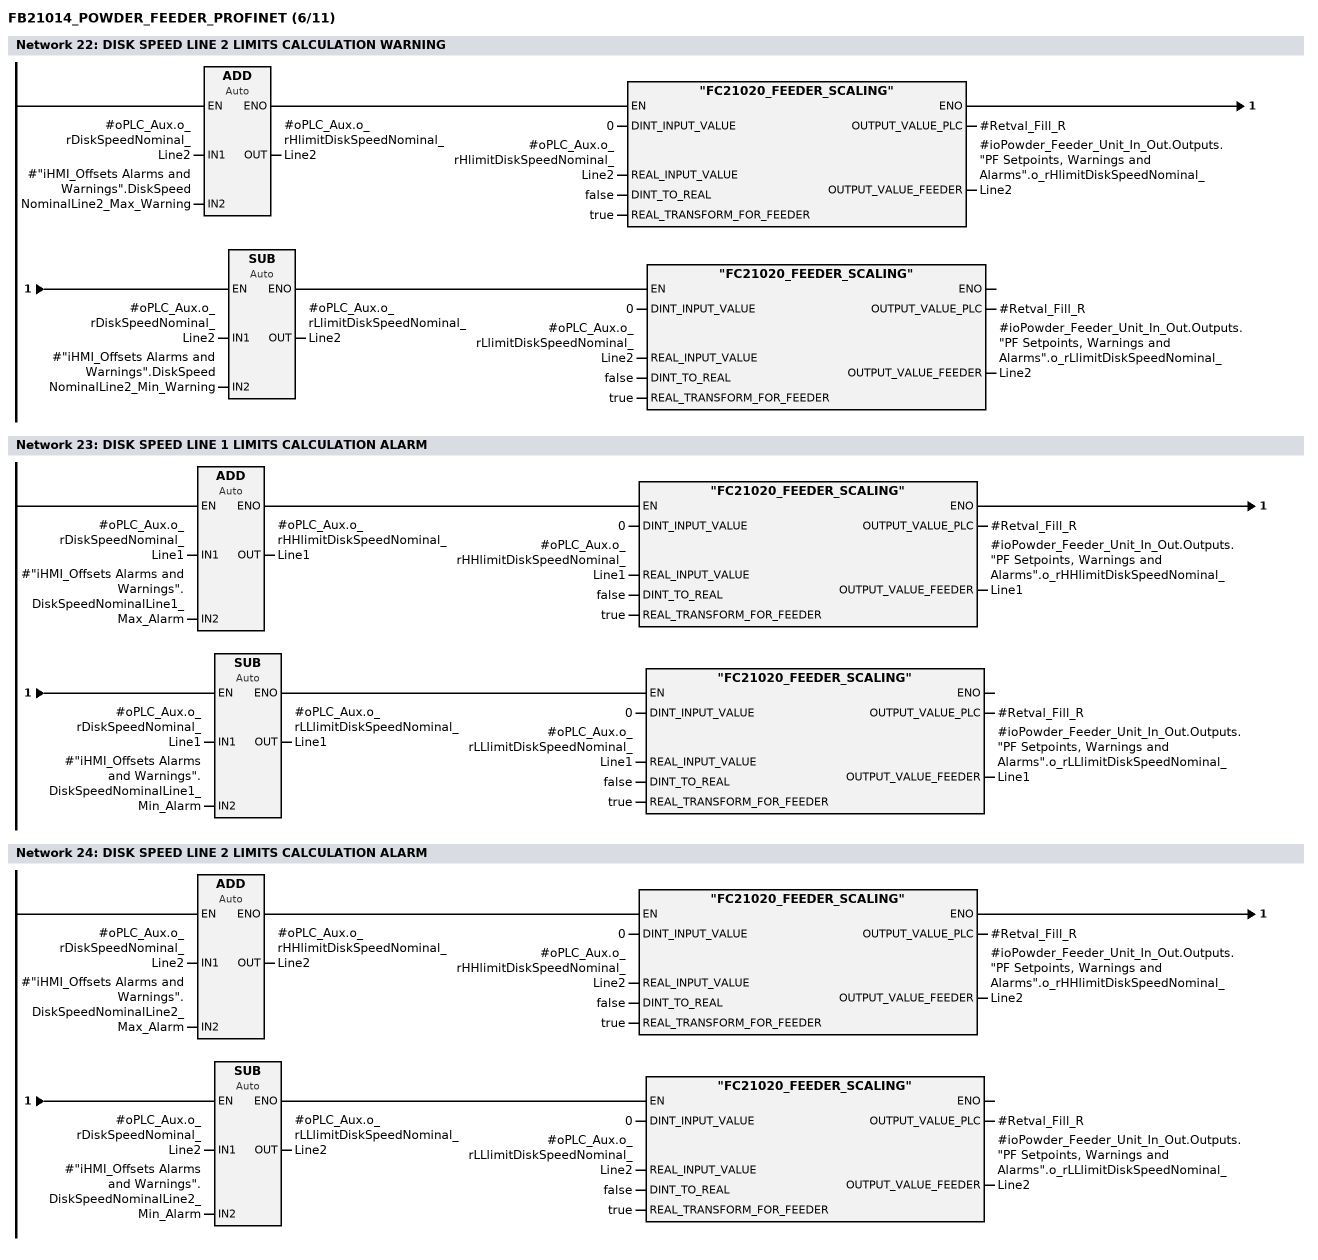
   RUNG wire#powerrail
      Add(in1 := #oPLC_Aux.o_rDiskSpeedNominal_Line2, in2 := #"iHMI_Offsets Alarms and Warnings".DiskSpeedNominalLine2_Max_Warning, out => #oPLC_Aux.o_rHlimitDiskSpeedNominal_Line2)
      "FC21020_FEEDER_SCALING"(DINT_INPUT_VALUE := 0, REAL_INPUT_VALUE := #oPLC_Aux.o_rHlimitDiskSpeedNominal_Line2, DINT_TO_REAL := false, REAL_TRANSFORM_FOR_FEEDER := true, OUTPUT_VALUE_PLC => #Retval_Fill_R, OUTPUT_VALUE_FEEDER => #ioPowder_Feeder_Unit_In_Out.Outputs."PF Setpoints, Warnings and Alarms".o_rHlimitDiskSpeedNominal_Line2)
      Sub(in1 := #oPLC_Aux.o_rDiskSpeedNominal_Line2, in2 := #"iHMI_Offsets Alarms and Warnings".DiskSpeedNominalLine2_Min_Warning, out => #oPLC_Aux.o_rLlimitDiskSpeedNominal_Line2)
      "FC21020_FEEDER_SCALING"(DINT_INPUT_VALUE := 0, REAL_INPUT_VALUE := #oPLC_Aux.o_rLlimitDiskSpeedNominal_Line2, DINT_TO_REAL := false, REAL_TRANSFORM_FOR_FEEDER := true, OUTPUT_VALUE_PLC => #Retval_Fill_R, OUTPUT_VALUE_FEEDER => #ioPowder_Feeder_Unit_In_Out.Outputs."PF Setpoints, Warnings and Alarms".o_rLlimitDiskSpeedNominal_Line2)
   END_RUNG
   // the same network as SCL:
   #oPLC_Aux.o_rHlimitDiskSpeedNominal_Line2 := #oPLC_Aux.o_rDiskSpeedNominal_Line2 + #"iHMI_Offsets Alarms and Warnings".DiskSpeedNominalLine2_Max_Warning;
   "FC21020_FEEDER_SCALING"(DINT_INPUT_VALUE := 0,
                           REAL_INPUT_VALUE := #oPLC_Aux.o_rHlimitDiskSpeedNominal_Line2,
                           DINT_TO_REAL := false,
                           REAL_TRANSFORM_FOR_FEEDER := true,
                           OUTPUT_VALUE_PLC => #Retval_Fill_R,
                           OUTPUT_VALUE_FEEDER => #ioPowder_Feeder_Unit_In_Out.Outputs."PF Setpoints, Warnings and Alarms".o_rHlimitDiskSpeedNominal_Line2,
                           ENO => #_w1);
   IF #_w1 THEN
       #oPLC_Aux.o_rLlimitDiskSpeedNominal_Line2 := #oPLC_Aux.o_rDiskSpeedNominal_Line2 - #"iHMI_Offsets Alarms and Warnings".DiskSpeedNominalLine2_Min_Warning;
       "FC21020_FEEDER_SCALING"(DINT_INPUT_VALUE := 0,
                               REAL_INPUT_VALUE := #oPLC_Aux.o_rLlimitDiskSpeedNominal_Line2,
                               DINT_TO_REAL := false,
                               REAL_TRANSFORM_FOR_FEEDER := true,
                               OUTPUT_VALUE_PLC => #Retval_Fill_R,
                               OUTPUT_VALUE_FEEDER => #ioPowder_Feeder_Unit_In_Out.Outputs."PF Setpoints, Warnings and Alarms".o_rLlimitDiskSpeedNominal_Line2);
   END_IF;
END_REGION

REGION Network 23: DISK SPEED LINE 1 LIMITS CALCULATION ALARM
   RUNG wire#powerrail
      Add(in1 := #oPLC_Aux.o_rDiskSpeedNominal_Line1, in2 := #"iHMI_Offsets Alarms and Warnings".DiskSpeedNominalLine1_Max_Alarm, out => #oPLC_Aux.o_rHHlimitDiskSpeedNominal_Line1)
      "FC21020_FEEDER_SCALING"(DINT_INPUT_VALUE := 0, REAL_INPUT_VALUE := #oPLC_Aux.o_rHHlimitDiskSpeedNominal_Line1, DINT_TO_REAL := false, REAL_TRANSFORM_FOR_FEEDER := true, OUTPUT_VALUE_PLC => #Retval_Fill_R, OUTPUT_VALUE_FEEDER => #ioPowder_Feeder_Unit_In_Out.Outputs."PF Setpoints, Warnings and Alarms".o_rHHlimitDiskSpeedNominal_Line1)
      Sub(in1 := #oPLC_Aux.o_rDiskSpeedNominal_Line1, in2 := #"iHMI_Offsets Alarms and Warnings".DiskSpeedNominalLine1_Min_Alarm, out => #oPLC_Aux.o_rLLlimitDiskSpeedNominal_Line1)
      "FC21020_FEEDER_SCALING"(DINT_INPUT_VALUE := 0, REAL_INPUT_VALUE := #oPLC_Aux.o_rLLlimitDiskSpeedNominal_Line1, DINT_TO_REAL := false, REAL_TRANSFORM_FOR_FEEDER := true, OUTPUT_VALUE_PLC => #Retval_Fill_R, OUTPUT_VALUE_FEEDER => #ioPowder_Feeder_Unit_In_Out.Outputs."PF Setpoints, Warnings and Alarms".o_rLLlimitDiskSpeedNominal_Line1)
   END_RUNG
   // the same network as SCL:
   #oPLC_Aux.o_rHHlimitDiskSpeedNominal_Line1 := #oPLC_Aux.o_rDiskSpeedNominal_Line1 + #"iHMI_Offsets Alarms and Warnings".DiskSpeedNominalLine1_Max_Alarm;
   "FC21020_FEEDER_SCALING"(DINT_INPUT_VALUE := 0,
                           REAL_INPUT_VALUE := #oPLC_Aux.o_rHHlimitDiskSpeedNominal_Line1,
                           DINT_TO_REAL := false,
                           REAL_TRANSFORM_FOR_FEEDER := true,
                           OUTPUT_VALUE_PLC => #Retval_Fill_R,
                           OUTPUT_VALUE_FEEDER => #ioPowder_Feeder_Unit_In_Out.Outputs."PF Setpoints, Warnings and Alarms".o_rHHlimitDiskSpeedNominal_Line1,
                           ENO => #_w1);
   IF #_w1 THEN
       #oPLC_Aux.o_rLLlimitDiskSpeedNominal_Line1 := #oPLC_Aux.o_rDiskSpeedNominal_Line1 - #"iHMI_Offsets Alarms and Warnings".DiskSpeedNominalLine1_Min_Alarm;
       "FC21020_FEEDER_SCALING"(DINT_INPUT_VALUE := 0,
                               REAL_INPUT_VALUE := #oPLC_Aux.o_rLLlimitDiskSpeedNominal_Line1,
                               DINT_TO_REAL := false,
                               REAL_TRANSFORM_FOR_FEEDER := true,
                               OUTPUT_VALUE_PLC => #Retval_Fill_R,
                               OUTPUT_VALUE_FEEDER => #ioPowder_Feeder_Unit_In_Out.Outputs."PF Setpoints, Warnings and Alarms".o_rLLlimitDiskSpeedNominal_Line1);
   END_IF;
END_REGION

REGION Network 24: DISK SPEED LINE 2 LIMITS CALCULATION ALARM
   RUNG wire#powerrail
      Add(in1 := #oPLC_Aux.o_rDiskSpeedNominal_Line2, in2 := #"iHMI_Offsets Alarms and Warnings".DiskSpeedNominalLine2_Max_Alarm, out => #oPLC_Aux.o_rHHlimitDiskSpeedNominal_Line2)
      "FC21020_FEEDER_SCALING"(DINT_INPUT_VALUE := 0, REAL_INPUT_VALUE := #oPLC_Aux.o_rHHlimitDiskSpeedNominal_Line2, DINT_TO_REAL := false, REAL_TRANSFORM_FOR_FEEDER := true, OUTPUT_VALUE_PLC => #Retval_Fill_R, OUTPUT_VALUE_FEEDER => #ioPowder_Feeder_Unit_In_Out.Outputs."PF Setpoints, Warnings and Alarms".o_rHHlimitDiskSpeedNominal_Line2)
      Sub(in1 := #oPLC_Aux.o_rDiskSpeedNominal_Line2, in2 := #"iHMI_Offsets Alarms and Warnings".DiskSpeedNominalLine2_Min_Alarm, out => #oPLC_Aux.o_rLLlimitDiskSpeedNominal_Line2)
      "FC21020_FEEDER_SCALING"(DINT_INPUT_VALUE := 0, REAL_INPUT_VALUE := #oPLC_Aux.o_rLLlimitDiskSpeedNominal_Line2, DINT_TO_REAL := false, REAL_TRANSFORM_FOR_FEEDER := true, OUTPUT_VALUE_PLC => #Retval_Fill_R, OUTPUT_VALUE_FEEDER => #ioPowder_Feeder_Unit_In_Out.Outputs."PF Setpoints, Warnings and Alarms".o_rLLlimitDiskSpeedNominal_Line2)
   END_RUNG
   // the same network as SCL:
   #oPLC_Aux.o_rHHlimitDiskSpeedNominal_Line2 := #oPLC_Aux.o_rDiskSpeedNominal_Line2 + #"iHMI_Offsets Alarms and Warnings".DiskSpeedNominalLine2_Max_Alarm;
   "FC21020_FEEDER_SCALING"(DINT_INPUT_VALUE := 0,
                           REAL_INPUT_VALUE := #oPLC_Aux.o_rHHlimitDiskSpeedNominal_Line2,
                           DINT_TO_REAL := false,
                           REAL_TRANSFORM_FOR_FEEDER := true,
                           OUTPUT_VALUE_PLC => #Retval_Fill_R,
                           OUTPUT_VALUE_FEEDER => #ioPowder_Feeder_Unit_In_Out.Outputs."PF Setpoints, Warnings and Alarms".o_rHHlimitDiskSpeedNominal_Line2,
                           ENO => #_w1);
   IF #_w1 THEN
       #oPLC_Aux.o_rLLlimitDiskSpeedNominal_Line2 := #oPLC_Aux.o_rDiskSpeedNominal_Line2 - #"iHMI_Offsets Alarms and Warnings".DiskSpeedNominalLine2_Min_Alarm;
       "FC21020_FEEDER_SCALING"(DINT_INPUT_VALUE := 0,
                               REAL_INPUT_VALUE := #oPLC_Aux.o_rLLlimitDiskSpeedNominal_Line2,
                               DINT_TO_REAL := false,
                               REAL_TRANSFORM_FOR_FEEDER := true,
                               OUTPUT_VALUE_PLC => #Retval_Fill_R,
                               OUTPUT_VALUE_FEEDER => #ioPowder_Feeder_Unit_In_Out.Outputs."PF Setpoints, Warnings and Alarms".o_rLLlimitDiskSpeedNominal_Line2);
   END_IF;
END_REGION

REGION Network 25: STIRRER SPEED LINE 1 LIMITS CALCULATION WARNING
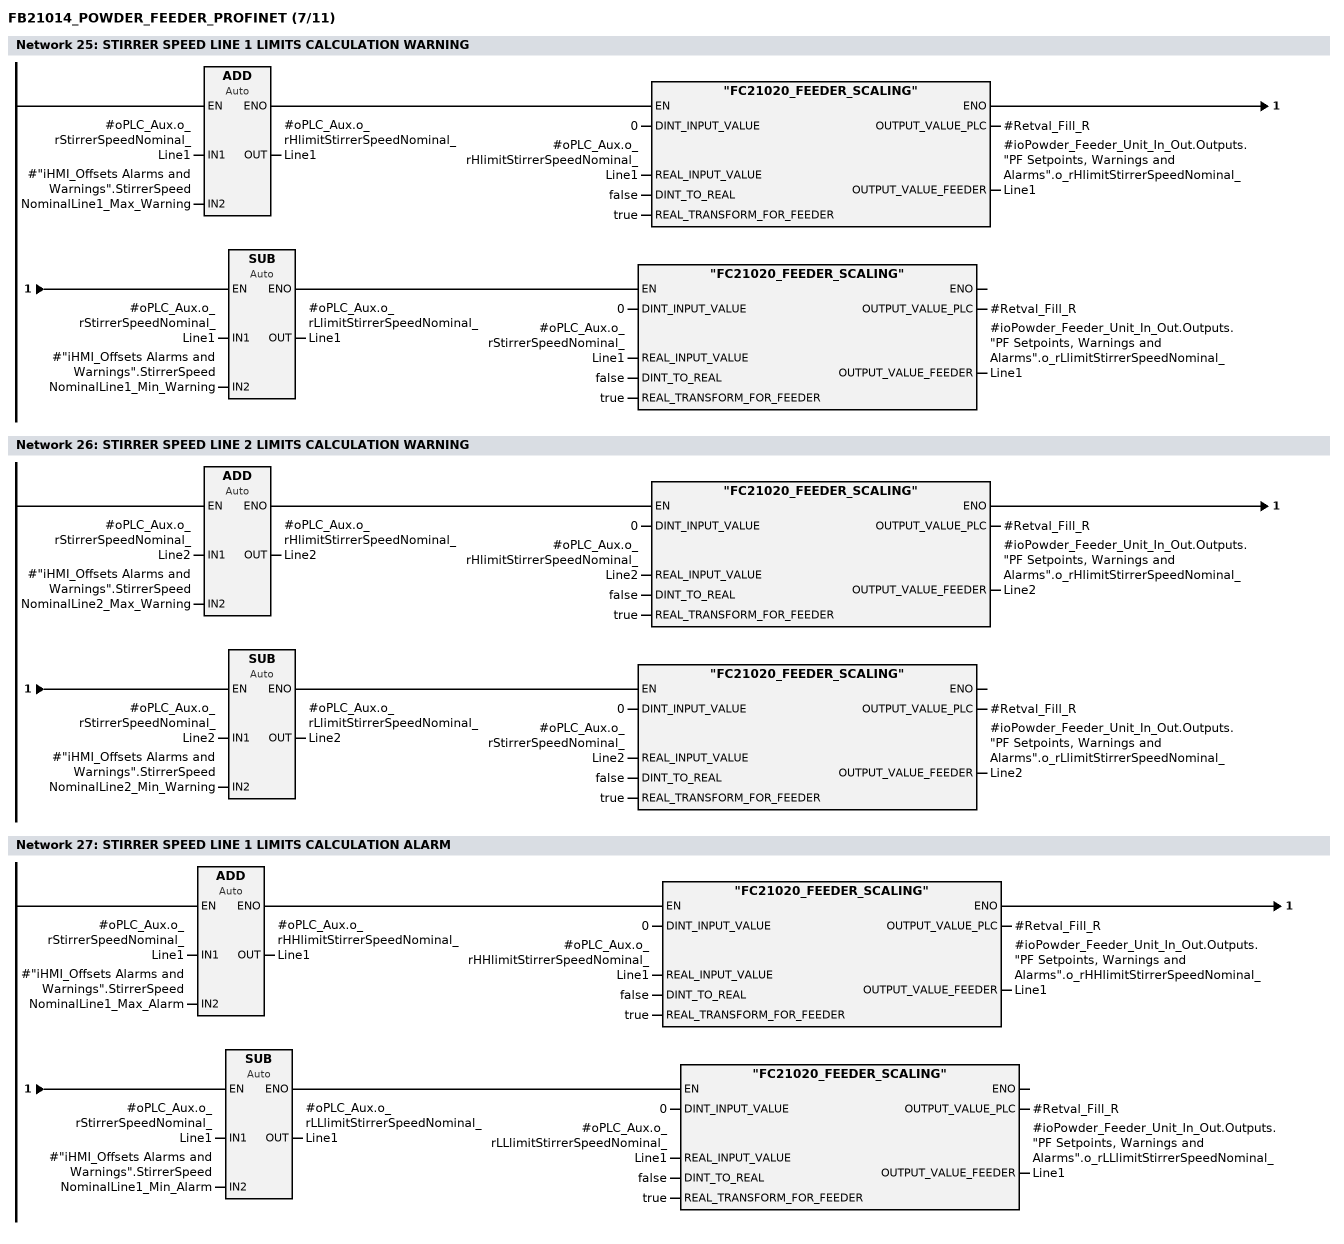
   RUNG wire#powerrail
      Add(in1 := #oPLC_Aux.o_rStirrerSpeedNominal_Line1, in2 := #"iHMI_Offsets Alarms and Warnings".StirrerSpeedNominalLine1_Max_Warning, out => #oPLC_Aux.o_rHlimitStirrerSpeedNominal_Line1)
      "FC21020_FEEDER_SCALING"(DINT_INPUT_VALUE := 0, REAL_INPUT_VALUE := #oPLC_Aux.o_rHlimitStirrerSpeedNominal_Line1, DINT_TO_REAL := false, REAL_TRANSFORM_FOR_FEEDER := true, OUTPUT_VALUE_PLC => #Retval_Fill_R, OUTPUT_VALUE_FEEDER => #ioPowder_Feeder_Unit_In_Out.Outputs."PF Setpoints, Warnings and Alarms".o_rHlimitStirrerSpeedNominal_Line1)
      Sub(in1 := #oPLC_Aux.o_rStirrerSpeedNominal_Line1, in2 := #"iHMI_Offsets Alarms and Warnings".StirrerSpeedNominalLine1_Min_Warning, out => #oPLC_Aux.o_rLlimitStirrerSpeedNominal_Line1)
      "FC21020_FEEDER_SCALING"(DINT_INPUT_VALUE := 0, REAL_INPUT_VALUE := #oPLC_Aux.o_rStirrerSpeedNominal_Line1, DINT_TO_REAL := false, REAL_TRANSFORM_FOR_FEEDER := true, OUTPUT_VALUE_PLC => #Retval_Fill_R, OUTPUT_VALUE_FEEDER => #ioPowder_Feeder_Unit_In_Out.Outputs."PF Setpoints, Warnings and Alarms".o_rLlimitStirrerSpeedNominal_Line1)
   END_RUNG
   // the same network as SCL:
   #oPLC_Aux.o_rHlimitStirrerSpeedNominal_Line1 := #oPLC_Aux.o_rStirrerSpeedNominal_Line1 + #"iHMI_Offsets Alarms and Warnings".StirrerSpeedNominalLine1_Max_Warning;
   "FC21020_FEEDER_SCALING"(DINT_INPUT_VALUE := 0,
                           REAL_INPUT_VALUE := #oPLC_Aux.o_rHlimitStirrerSpeedNominal_Line1,
                           DINT_TO_REAL := false,
                           REAL_TRANSFORM_FOR_FEEDER := true,
                           OUTPUT_VALUE_PLC => #Retval_Fill_R,
                           OUTPUT_VALUE_FEEDER => #ioPowder_Feeder_Unit_In_Out.Outputs."PF Setpoints, Warnings and Alarms".o_rHlimitStirrerSpeedNominal_Line1,
                           ENO => #_w1);
   IF #_w1 THEN
       #oPLC_Aux.o_rLlimitStirrerSpeedNominal_Line1 := #oPLC_Aux.o_rStirrerSpeedNominal_Line1 - #"iHMI_Offsets Alarms and Warnings".StirrerSpeedNominalLine1_Min_Warning;
       "FC21020_FEEDER_SCALING"(DINT_INPUT_VALUE := 0,
                               REAL_INPUT_VALUE := #oPLC_Aux.o_rStirrerSpeedNominal_Line1,
                               DINT_TO_REAL := false,
                               REAL_TRANSFORM_FOR_FEEDER := true,
                               OUTPUT_VALUE_PLC => #Retval_Fill_R,
                               OUTPUT_VALUE_FEEDER => #ioPowder_Feeder_Unit_In_Out.Outputs."PF Setpoints, Warnings and Alarms".o_rLlimitStirrerSpeedNominal_Line1);
   END_IF;
END_REGION

REGION Network 26: STIRRER SPEED LINE 2 LIMITS CALCULATION WARNING
   RUNG wire#powerrail
      Add(in1 := #oPLC_Aux.o_rStirrerSpeedNominal_Line2, in2 := #"iHMI_Offsets Alarms and Warnings".StirrerSpeedNominalLine2_Max_Warning, out => #oPLC_Aux.o_rHlimitStirrerSpeedNominal_Line2)
      "FC21020_FEEDER_SCALING"(DINT_INPUT_VALUE := 0, REAL_INPUT_VALUE := #oPLC_Aux.o_rHlimitStirrerSpeedNominal_Line2, DINT_TO_REAL := false, REAL_TRANSFORM_FOR_FEEDER := true, OUTPUT_VALUE_PLC => #Retval_Fill_R, OUTPUT_VALUE_FEEDER => #ioPowder_Feeder_Unit_In_Out.Outputs."PF Setpoints, Warnings and Alarms".o_rHlimitStirrerSpeedNominal_Line2)
      Sub(in1 := #oPLC_Aux.o_rStirrerSpeedNominal_Line2, in2 := #"iHMI_Offsets Alarms and Warnings".StirrerSpeedNominalLine2_Min_Warning, out => #oPLC_Aux.o_rLlimitStirrerSpeedNominal_Line2)
      "FC21020_FEEDER_SCALING"(DINT_INPUT_VALUE := 0, REAL_INPUT_VALUE := #oPLC_Aux.o_rStirrerSpeedNominal_Line2, DINT_TO_REAL := false, REAL_TRANSFORM_FOR_FEEDER := true, OUTPUT_VALUE_PLC => #Retval_Fill_R, OUTPUT_VALUE_FEEDER => #ioPowder_Feeder_Unit_In_Out.Outputs."PF Setpoints, Warnings and Alarms".o_rLlimitStirrerSpeedNominal_Line2)
   END_RUNG
   // the same network as SCL:
   #oPLC_Aux.o_rHlimitStirrerSpeedNominal_Line2 := #oPLC_Aux.o_rStirrerSpeedNominal_Line2 + #"iHMI_Offsets Alarms and Warnings".StirrerSpeedNominalLine2_Max_Warning;
   "FC21020_FEEDER_SCALING"(DINT_INPUT_VALUE := 0,
                           REAL_INPUT_VALUE := #oPLC_Aux.o_rHlimitStirrerSpeedNominal_Line2,
                           DINT_TO_REAL := false,
                           REAL_TRANSFORM_FOR_FEEDER := true,
                           OUTPUT_VALUE_PLC => #Retval_Fill_R,
                           OUTPUT_VALUE_FEEDER => #ioPowder_Feeder_Unit_In_Out.Outputs."PF Setpoints, Warnings and Alarms".o_rHlimitStirrerSpeedNominal_Line2,
                           ENO => #_w1);
   IF #_w1 THEN
       #oPLC_Aux.o_rLlimitStirrerSpeedNominal_Line2 := #oPLC_Aux.o_rStirrerSpeedNominal_Line2 - #"iHMI_Offsets Alarms and Warnings".StirrerSpeedNominalLine2_Min_Warning;
       "FC21020_FEEDER_SCALING"(DINT_INPUT_VALUE := 0,
                               REAL_INPUT_VALUE := #oPLC_Aux.o_rStirrerSpeedNominal_Line2,
                               DINT_TO_REAL := false,
                               REAL_TRANSFORM_FOR_FEEDER := true,
                               OUTPUT_VALUE_PLC => #Retval_Fill_R,
                               OUTPUT_VALUE_FEEDER => #ioPowder_Feeder_Unit_In_Out.Outputs."PF Setpoints, Warnings and Alarms".o_rLlimitStirrerSpeedNominal_Line2);
   END_IF;
END_REGION

